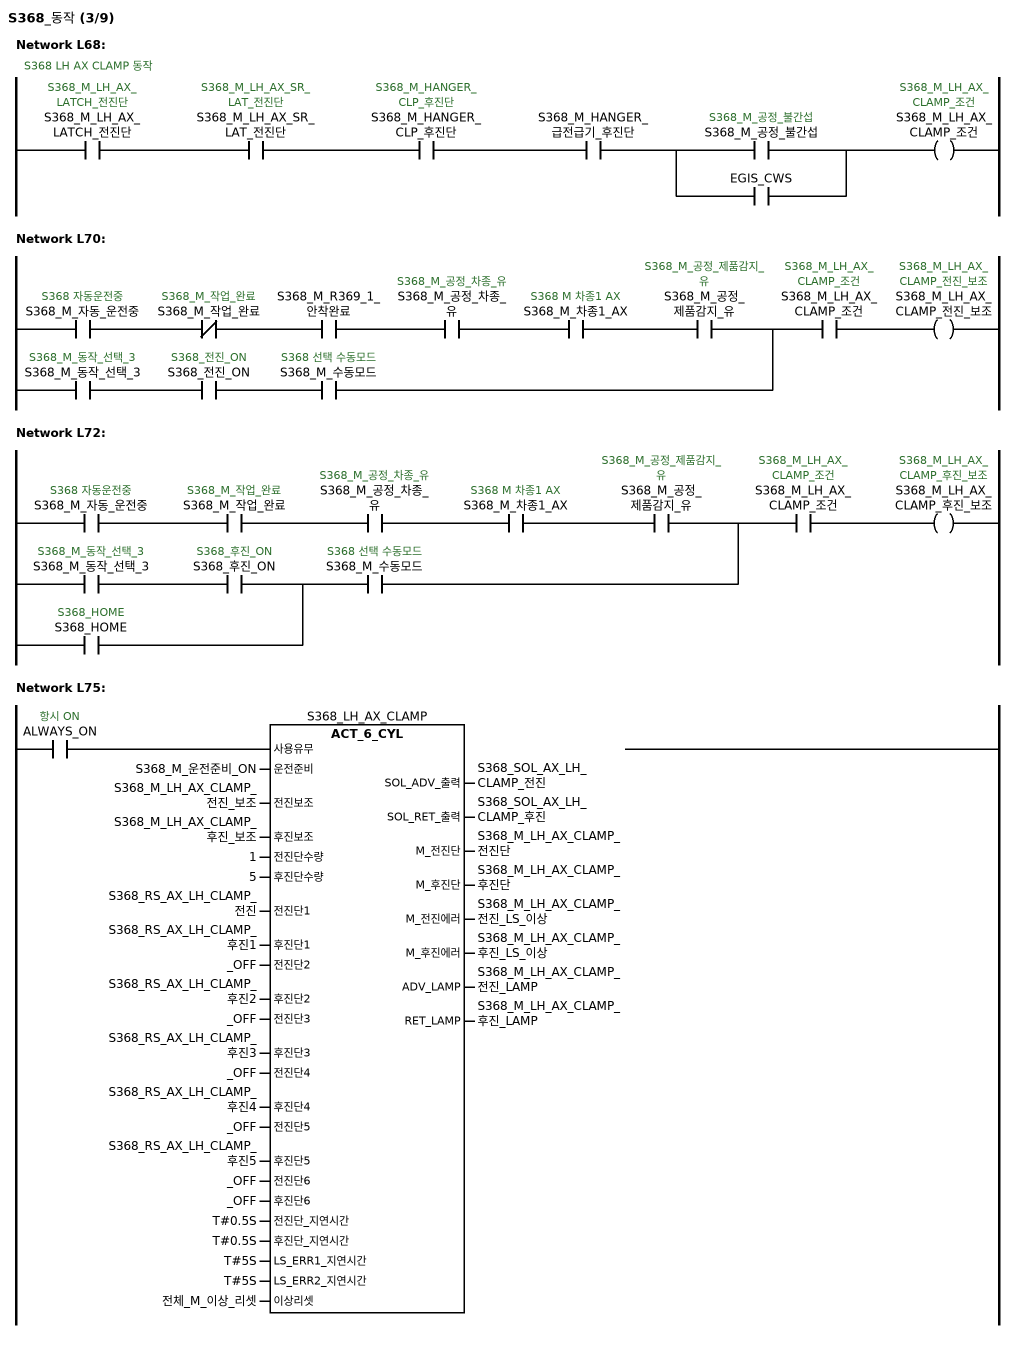
(* [picture p240: S368_동작 rungs L68-L75] *)
(* S368 LH AX CLAMP 동작 *)
(* Rung L68 *)
S368_M_LH_AX_CLAMP_조건 := S368_M_LH_AX_LATCH_전진단 AND S368_M_LH_AX_SR_LAT_전진단 AND S368_M_HANGER_CLP_후진단 AND S368_M_HANGER_급전급기_후진단 AND (S368_M_공정_불간섭 OR EGIS_CWS);
(* Rung L70 *)
S368_M_LH_AX_CLAMP_전진_보조 := ((S368_M_자동_운전중 AND NOT S368_M_작업_완료 AND S368_M_R369_1_안착완료 AND S368_M_공정_차종_유 AND S368_M_차종1_AX AND S368_M_공정_제품감지_유) OR (S368_M_동작_선택_3 AND S368_전진_ON AND S368_M_수동모드)) AND S368_M_LH_AX_CLAMP_조건;
(* Rung L72 *)
S368_M_LH_AX_CLAMP_후진_보조 := ((S368_M_자동_운전중 AND S368_M_작업_완료 AND S368_M_공정_차종_유 AND S368_M_차종1_AX AND S368_M_공정_제품감지_유) OR (((S368_M_동작_선택_3 AND S368_후진_ON) OR S368_HOME) AND S368_M_수동모드)) AND S368_M_LH_AX_CLAMP_조건;
(* Rung L75 *)
S368_LH_AX_CLAMP(사용유무 := ALWAYS_ON, 운전준비 := S368_M_운전준비_ON, 전진보조 := S368_M_LH_AX_CLAMP_전진_보조, 후진보조 := S368_M_LH_AX_CLAMP_후진_보조, 전진단수량 := 1, 후진단수량 := 5, 전진단1 := S368_RS_AX_LH_CLAMP_전진, 후진단1 := S368_RS_AX_LH_CLAMP_후진1, 전진단2 := _OFF, 후진단2 := S368_RS_AX_LH_CLAMP_후진2, 전진단3 := _OFF, 후진단3 := S368_RS_AX_LH_CLAMP_후진3, 전진단4 := _OFF, 후진단4 := S368_RS_AX_LH_CLAMP_후진4, 전진단5 := _OFF, 후진단5 := S368_RS_AX_LH_CLAMP_후진5, 전진단6 := _OFF, 후진단6 := _OFF, 전진단_지연시간 := T#0.5S, 후진단_지연시간 := T#0.5S, LS_ERR1_지연시간 := T#5S, LS_ERR2_지연시간 := T#5S, 이상리셋 := 전체_M_이상_리셋, SOL_ADV_출력 => S368_SOL_AX_LH_CLAMP_전진, SOL_RET_출력 => S368_SOL_AX_LH_CLAMP_후진, M_전진단 => S368_M_LH_AX_CLAMP_전진단, M_후진단 => S368_M_LH_AX_CLAMP_후진단, M_전진에러 => S368_M_LH_AX_CLAMP_전진_LS_이상, M_후진에러 => S368_M_LH_AX_CLAMP_후진_LS_이상, ADV_LAMP => S368_M_LH_AX_CLAMP_전진_LAMP, RET_LAMP => S368_M_LH_AX_CLAMP_후진_LAMP);

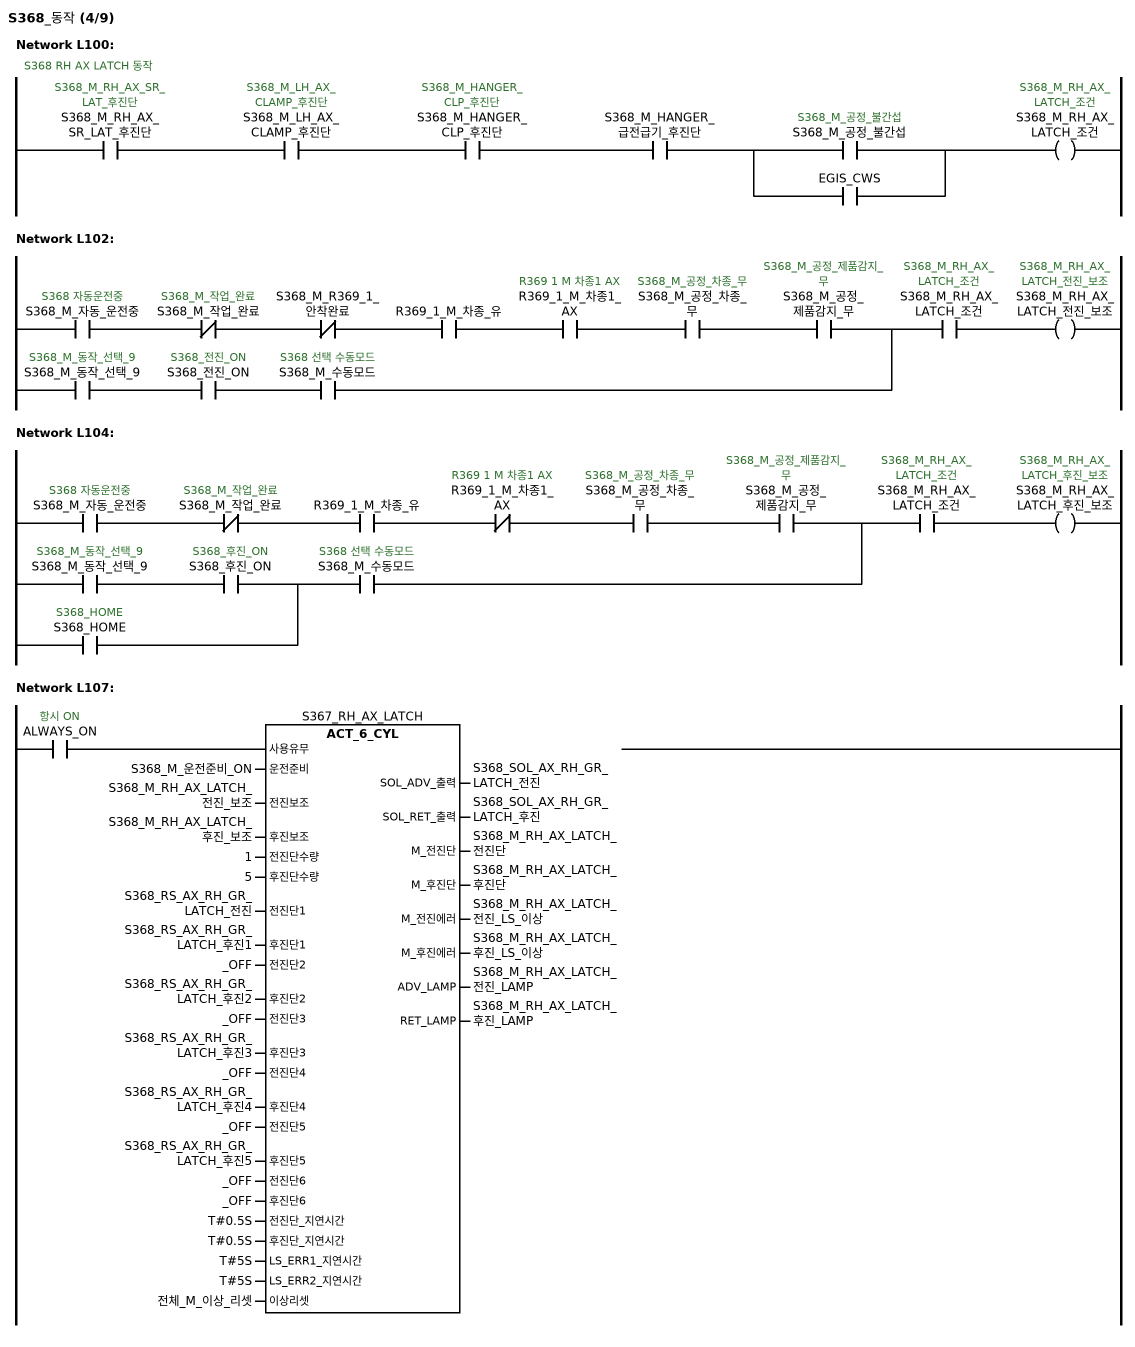
(* S368 RH AX LATCH 동작 *)
(* Rung L100 *)
S368_M_RH_AX_LATCH_조건 := S368_M_RH_AX_SR_LAT_후진단 AND S368_M_LH_AX_CLAMP_후진단 AND S368_M_HANGER_CLP_후진단 AND S368_M_HANGER_급전급기_후진단 AND (S368_M_공정_불간섭 OR EGIS_CWS);
(* Rung L102 *)
S368_M_RH_AX_LATCH_전진_보조 := ((S368_M_자동_운전중 AND NOT S368_M_작업_완료 AND NOT S368_M_R369_1_안착완료 AND R369_1_M_차종_유 AND R369_1_M_차종1_AX AND S368_M_공정_차종_무 AND S368_M_공정_제품감지_무) OR (S368_M_동작_선택_9 AND S368_전진_ON AND S368_M_수동모드)) AND S368_M_RH_AX_LATCH_조건;
(* Rung L104 *)
S368_M_RH_AX_LATCH_후진_보조 := ((S368_M_자동_운전중 AND NOT S368_M_작업_완료 AND R369_1_M_차종_유 AND NOT R369_1_M_차종1_AX AND S368_M_공정_차종_무 AND S368_M_공정_제품감지_무) OR (((S368_M_동작_선택_9 AND S368_후진_ON) OR S368_HOME) AND S368_M_수동모드)) AND S368_M_RH_AX_LATCH_조건;
(* Rung L107 *)
S367_RH_AX_LATCH(사용유무 := ALWAYS_ON, 운전준비 := S368_M_운전준비_ON, 전진보조 := S368_M_RH_AX_LATCH_전진_보조, 후진보조 := S368_M_RH_AX_LATCH_후진_보조, 전진단수량 := 1, 후진단수량 := 5, 전진단1 := S368_RS_AX_RH_GR_LATCH_전진, 후진단1 := S368_RS_AX_RH_GR_LATCH_후진1, 전진단2 := _OFF, 후진단2 := S368_RS_AX_RH_GR_LATCH_후진2, 전진단3 := _OFF, 후진단3 := S368_RS_AX_RH_GR_LATCH_후진3, 전진단4 := _OFF, 후진단4 := S368_RS_AX_RH_GR_LATCH_후진4, 전진단5 := _OFF, 후진단5 := S368_RS_AX_RH_GR_LATCH_후진5, 전진단6 := _OFF, 후진단6 := _OFF, 전진단_지연시간 := T#0.5S, 후진단_지연시간 := T#0.5S, LS_ERR1_지연시간 := T#5S, LS_ERR2_지연시간 := T#5S, 이상리셋 := 전체_M_이상_리셋, SOL_ADV_출력 => S368_SOL_AX_RH_GR_LATCH_전진, SOL_RET_출력 => S368_SOL_AX_RH_GR_LATCH_후진, M_전진단 => S368_M_RH_AX_LATCH_전진단, M_후진단 => S368_M_RH_AX_LATCH_후진단, M_전진에러 => S368_M_RH_AX_LATCH_전진_LS_이상, M_후진에러 => S368_M_RH_AX_LATCH_후진_LS_이상, ADV_LAMP => S368_M_RH_AX_LATCH_전진_LAMP, RET_LAMP => S368_M_RH_AX_LATCH_후진_LAMP);

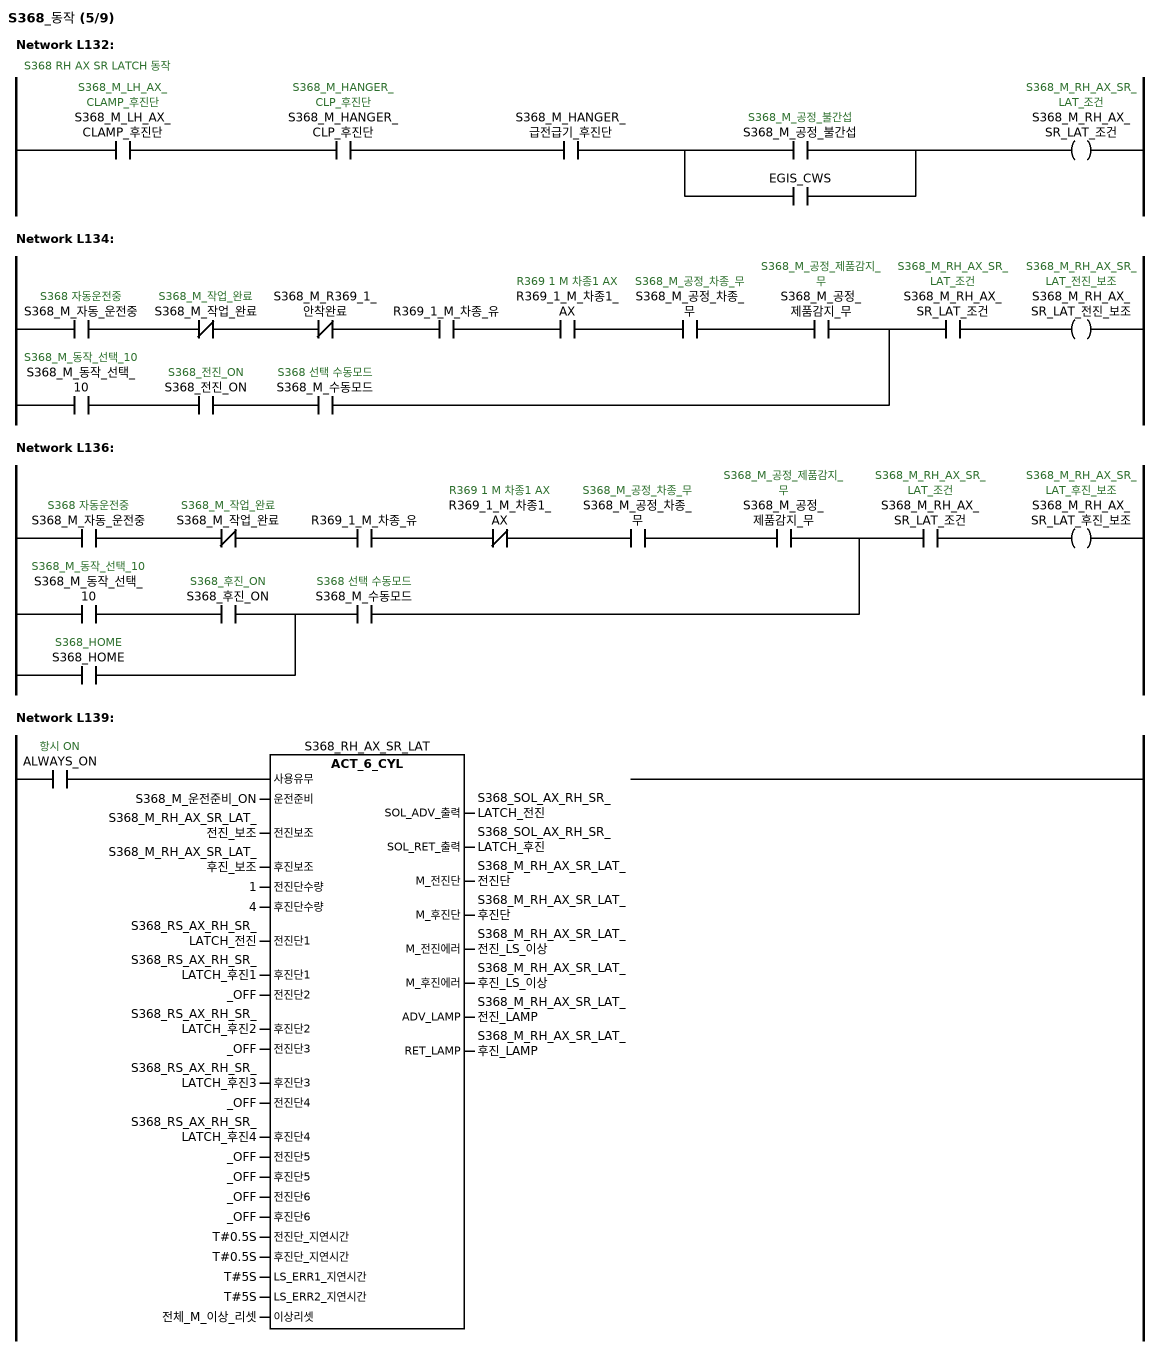
(* S368 RH AX SR LATCH 동작 *)
(* Rung L132 *)
S368_M_RH_AX_SR_LAT_조건 := S368_M_LH_AX_CLAMP_후진단 AND S368_M_HANGER_CLP_후진단 AND S368_M_HANGER_급전급기_후진단 AND (S368_M_공정_불간섭 OR EGIS_CWS);
(* Rung L134 *)
S368_M_RH_AX_SR_LAT_전진_보조 := ((S368_M_자동_운전중 AND NOT S368_M_작업_완료 AND NOT S368_M_R369_1_안착완료 AND R369_1_M_차종_유 AND R369_1_M_차종1_AX AND S368_M_공정_차종_무 AND S368_M_공정_제품감지_무) OR (S368_M_동작_선택_10 AND S368_전진_ON AND S368_M_수동모드)) AND S368_M_RH_AX_SR_LAT_조건;
(* Rung L136 *)
S368_M_RH_AX_SR_LAT_후진_보조 := ((S368_M_자동_운전중 AND NOT S368_M_작업_완료 AND R369_1_M_차종_유 AND NOT R369_1_M_차종1_AX AND S368_M_공정_차종_무 AND S368_M_공정_제품감지_무) OR (((S368_M_동작_선택_10 AND S368_후진_ON) OR S368_HOME) AND S368_M_수동모드)) AND S368_M_RH_AX_SR_LAT_조건;
(* Rung L139 *)
S368_RH_AX_SR_LAT(사용유무 := ALWAYS_ON, 운전준비 := S368_M_운전준비_ON, 전진보조 := S368_M_RH_AX_SR_LAT_전진_보조, 후진보조 := S368_M_RH_AX_SR_LAT_후진_보조, 전진단수량 := 1, 후진단수량 := 4, 전진단1 := S368_RS_AX_RH_SR_LATCH_전진, 후진단1 := S368_RS_AX_RH_SR_LATCH_후진1, 전진단2 := _OFF, 후진단2 := S368_RS_AX_RH_SR_LATCH_후진2, 전진단3 := _OFF, 후진단3 := S368_RS_AX_RH_SR_LATCH_후진3, 전진단4 := _OFF, 후진단4 := S368_RS_AX_RH_SR_LATCH_후진4, 전진단5 := _OFF, 후진단5 := _OFF, 전진단6 := _OFF, 후진단6 := _OFF, 전진단_지연시간 := T#0.5S, 후진단_지연시간 := T#0.5S, LS_ERR1_지연시간 := T#5S, LS_ERR2_지연시간 := T#5S, 이상리셋 := 전체_M_이상_리셋, SOL_ADV_출력 => S368_SOL_AX_RH_SR_LATCH_전진, SOL_RET_출력 => S368_SOL_AX_RH_SR_LATCH_후진, M_전진단 => S368_M_RH_AX_SR_LAT_전진단, M_후진단 => S368_M_RH_AX_SR_LAT_후진단, M_전진에러 => S368_M_RH_AX_SR_LAT_전진_LS_이상, M_후진에러 => S368_M_RH_AX_SR_LAT_후진_LS_이상, ADV_LAMP => S368_M_RH_AX_SR_LAT_전진_LAMP, RET_LAMP => S368_M_RH_AX_SR_LAT_후진_LAMP);

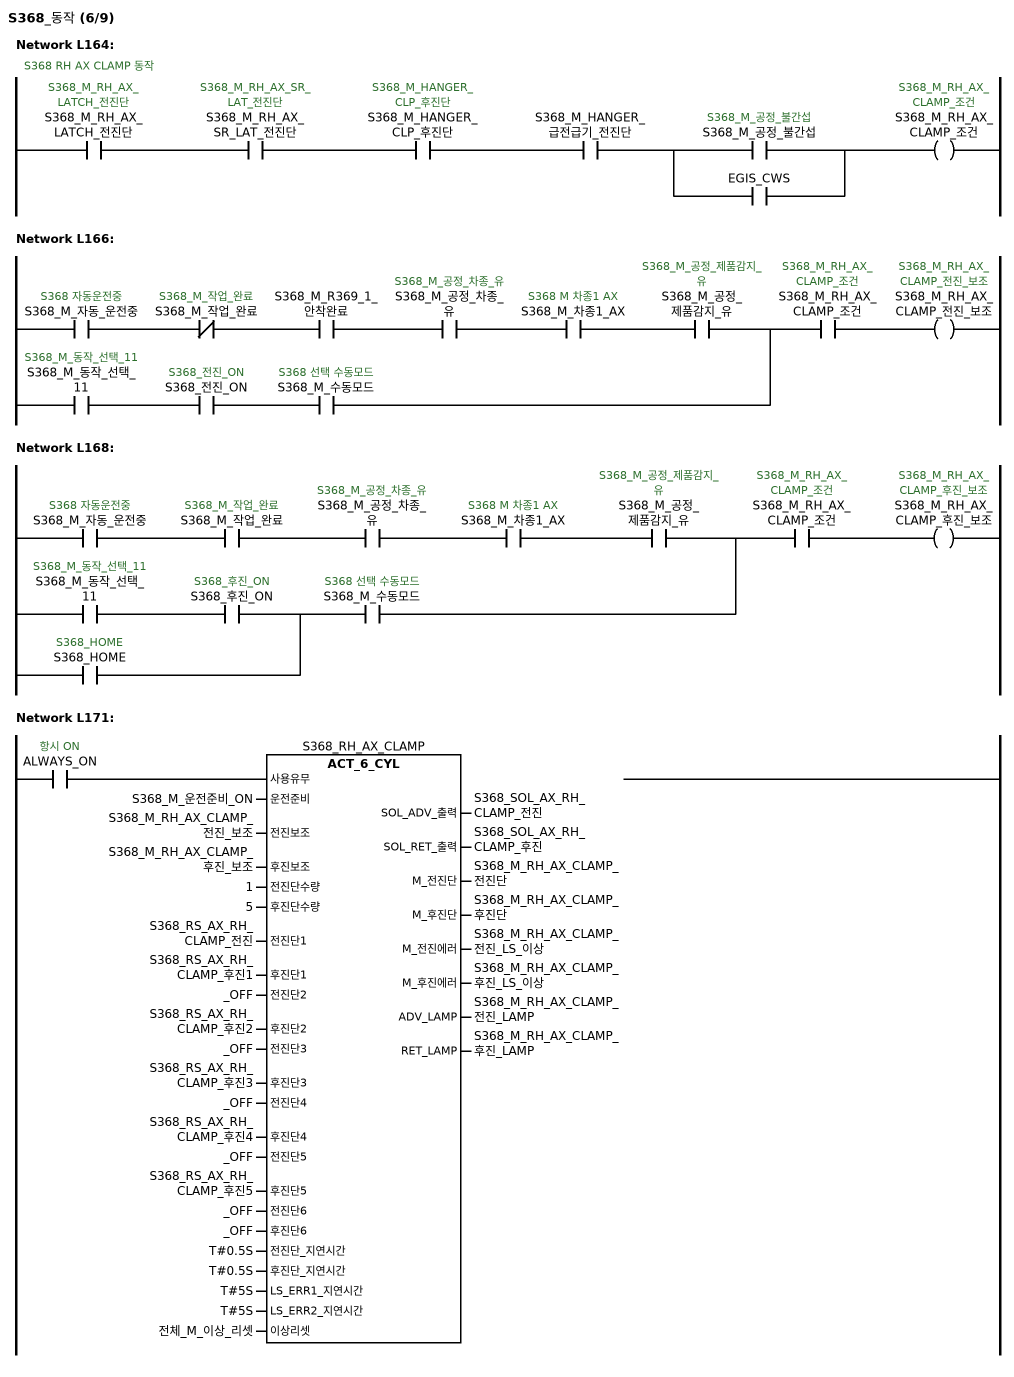
(* S368 RH AX CLAMP 동작 *)
(* Rung L164 *)
S368_M_RH_AX_CLAMP_조건 := S368_M_RH_AX_LATCH_전진단 AND S368_M_RH_AX_SR_LAT_전진단 AND S368_M_HANGER_CLP_후진단 AND S368_M_HANGER_급전급기_전진단 AND (S368_M_공정_불간섭 OR EGIS_CWS);
(* Rung L166 *)
S368_M_RH_AX_CLAMP_전진_보조 := ((S368_M_자동_운전중 AND NOT S368_M_작업_완료 AND S368_M_R369_1_안착완료 AND S368_M_공정_차종_유 AND S368_M_차종1_AX AND S368_M_공정_제품감지_유) OR (S368_M_동작_선택_11 AND S368_전진_ON AND S368_M_수동모드)) AND S368_M_RH_AX_CLAMP_조건;
(* Rung L168 *)
S368_M_RH_AX_CLAMP_후진_보조 := ((S368_M_자동_운전중 AND S368_M_작업_완료 AND S368_M_공정_차종_유 AND S368_M_차종1_AX AND S368_M_공정_제품감지_유) OR (((S368_M_동작_선택_11 AND S368_후진_ON) OR S368_HOME) AND S368_M_수동모드)) AND S368_M_RH_AX_CLAMP_조건;
(* Rung L171 *)
S368_RH_AX_CLAMP(사용유무 := ALWAYS_ON, 운전준비 := S368_M_운전준비_ON, 전진보조 := S368_M_RH_AX_CLAMP_전진_보조, 후진보조 := S368_M_RH_AX_CLAMP_후진_보조, 전진단수량 := 1, 후진단수량 := 5, 전진단1 := S368_RS_AX_RH_CLAMP_전진, 후진단1 := S368_RS_AX_RH_CLAMP_후진1, 전진단2 := _OFF, 후진단2 := S368_RS_AX_RH_CLAMP_후진2, 전진단3 := _OFF, 후진단3 := S368_RS_AX_RH_CLAMP_후진3, 전진단4 := _OFF, 후진단4 := S368_RS_AX_RH_CLAMP_후진4, 전진단5 := _OFF, 후진단5 := S368_RS_AX_RH_CLAMP_후진5, 전진단6 := _OFF, 후진단6 := _OFF, 전진단_지연시간 := T#0.5S, 후진단_지연시간 := T#0.5S, LS_ERR1_지연시간 := T#5S, LS_ERR2_지연시간 := T#5S, 이상리셋 := 전체_M_이상_리셋, SOL_ADV_출력 => S368_SOL_AX_RH_CLAMP_전진, SOL_RET_출력 => S368_SOL_AX_RH_CLAMP_후진, M_전진단 => S368_M_RH_AX_CLAMP_전진단, M_후진단 => S368_M_RH_AX_CLAMP_후진단, M_전진에러 => S368_M_RH_AX_CLAMP_전진_LS_이상, M_후진에러 => S368_M_RH_AX_CLAMP_후진_LS_이상, ADV_LAMP => S368_M_RH_AX_CLAMP_전진_LAMP, RET_LAMP => S368_M_RH_AX_CLAMP_후진_LAMP);

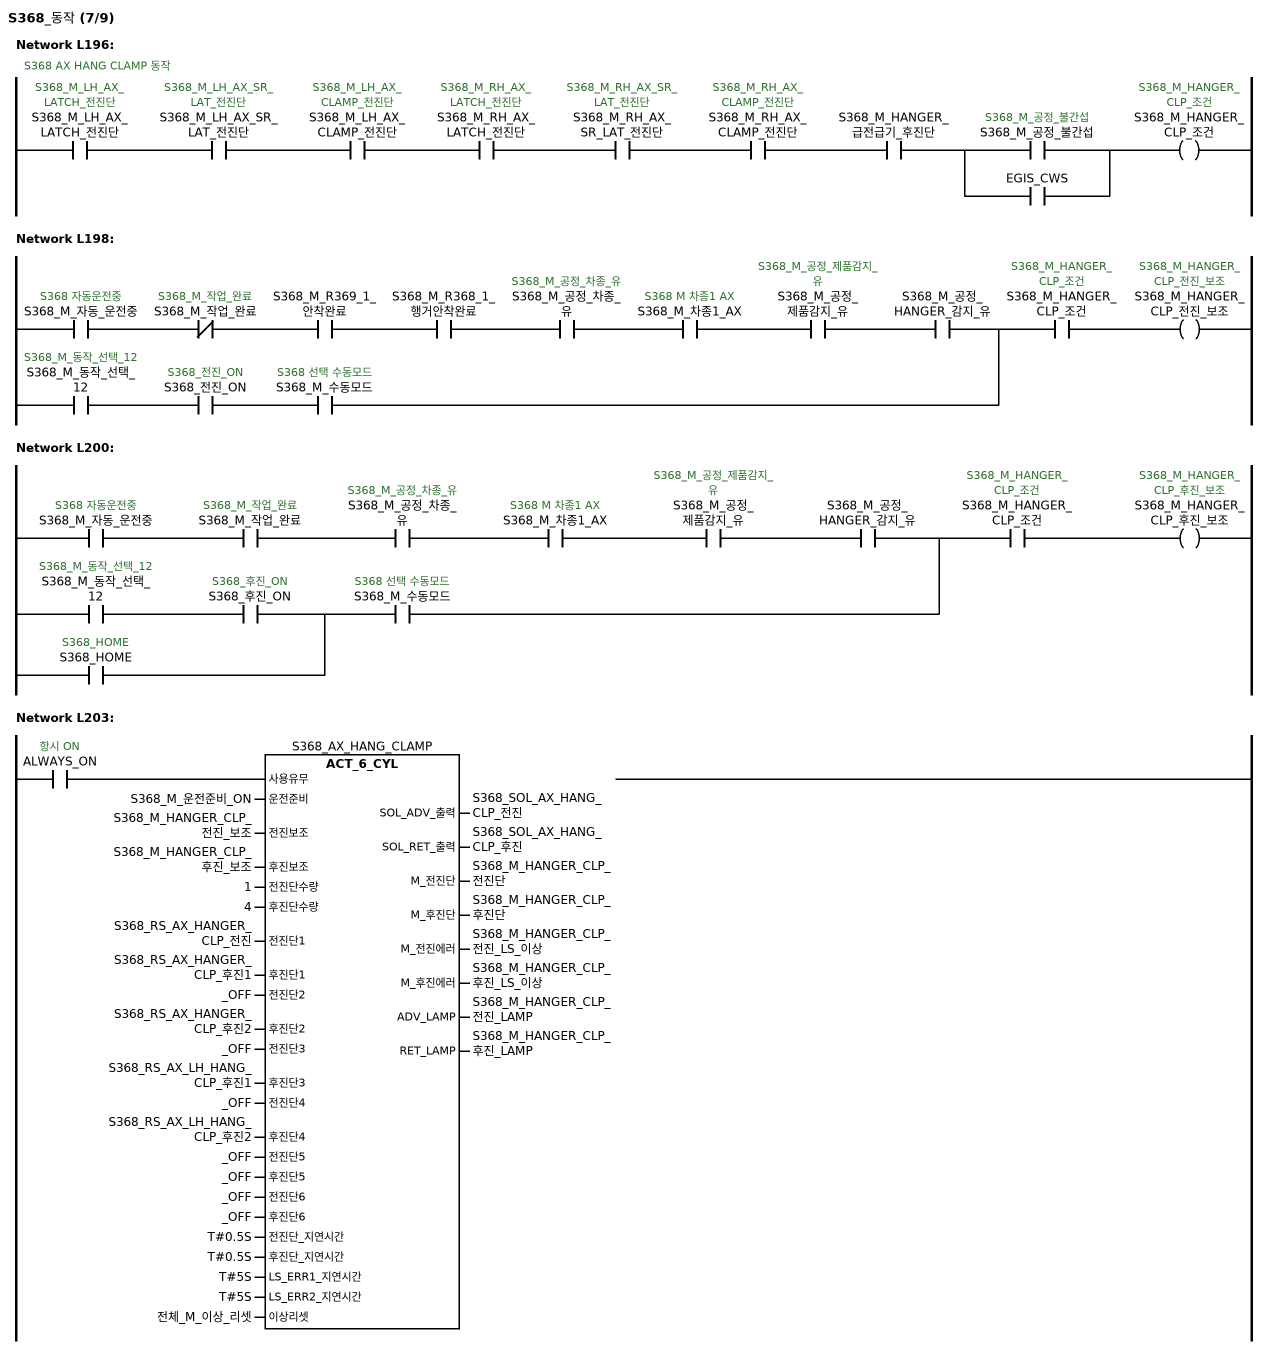
(* S368 AX HANG CLAMP 동작 *)
(* Rung L196 *)
S368_M_HANGER_CLP_조건 := S368_M_LH_AX_LATCH_전진단 AND S368_M_LH_AX_SR_LAT_전진단 AND S368_M_LH_AX_CLAMP_전진단 AND S368_M_RH_AX_LATCH_전진단 AND S368_M_RH_AX_SR_LAT_전진단 AND S368_M_RH_AX_CLAMP_전진단 AND S368_M_HANGER_급전급기_후진단 AND (S368_M_공정_불간섭 OR EGIS_CWS);
(* Rung L198 *)
S368_M_HANGER_CLP_전진_보조 := ((S368_M_자동_운전중 AND NOT S368_M_작업_완료 AND S368_M_R369_1_안착완료 AND S368_M_R368_1_행거안착완료 AND S368_M_공정_차종_유 AND S368_M_차종1_AX AND S368_M_공정_제품감지_유 AND S368_M_공정_HANGER_감지_유) OR (S368_M_동작_선택_12 AND S368_전진_ON AND S368_M_수동모드)) AND S368_M_HANGER_CLP_조건;
(* Rung L200 *)
S368_M_HANGER_CLP_후진_보조 := ((S368_M_자동_운전중 AND S368_M_작업_완료 AND S368_M_공정_차종_유 AND S368_M_차종1_AX AND S368_M_공정_제품감지_유 AND S368_M_공정_HANGER_감지_유) OR (((S368_M_동작_선택_12 AND S368_후진_ON) OR S368_HOME) AND S368_M_수동모드)) AND S368_M_HANGER_CLP_조건;
(* Rung L203 *)
S368_AX_HANG_CLAMP(사용유무 := ALWAYS_ON, 운전준비 := S368_M_운전준비_ON, 전진보조 := S368_M_HANGER_CLP_전진_보조, 후진보조 := S368_M_HANGER_CLP_후진_보조, 전진단수량 := 1, 후진단수량 := 4, 전진단1 := S368_RS_AX_HANGER_CLP_전진, 후진단1 := S368_RS_AX_HANGER_CLP_후진1, 전진단2 := _OFF, 후진단2 := S368_RS_AX_HANGER_CLP_후진2, 전진단3 := _OFF, 후진단3 := S368_RS_AX_LH_HANG_CLP_후진1, 전진단4 := _OFF, 후진단4 := S368_RS_AX_LH_HANG_CLP_후진2, 전진단5 := _OFF, 후진단5 := _OFF, 전진단6 := _OFF, 후진단6 := _OFF, 전진단_지연시간 := T#0.5S, 후진단_지연시간 := T#0.5S, LS_ERR1_지연시간 := T#5S, LS_ERR2_지연시간 := T#5S, 이상리셋 := 전체_M_이상_리셋, SOL_ADV_출력 => S368_SOL_AX_HANG_CLP_전진, SOL_RET_출력 => S368_SOL_AX_HANG_CLP_후진, M_전진단 => S368_M_HANGER_CLP_전진단, M_후진단 => S368_M_HANGER_CLP_후진단, M_전진에러 => S368_M_HANGER_CLP_전진_LS_이상, M_후진에러 => S368_M_HANGER_CLP_후진_LS_이상, ADV_LAMP => S368_M_HANGER_CLP_전진_LAMP, RET_LAMP => S368_M_HANGER_CLP_후진_LAMP);

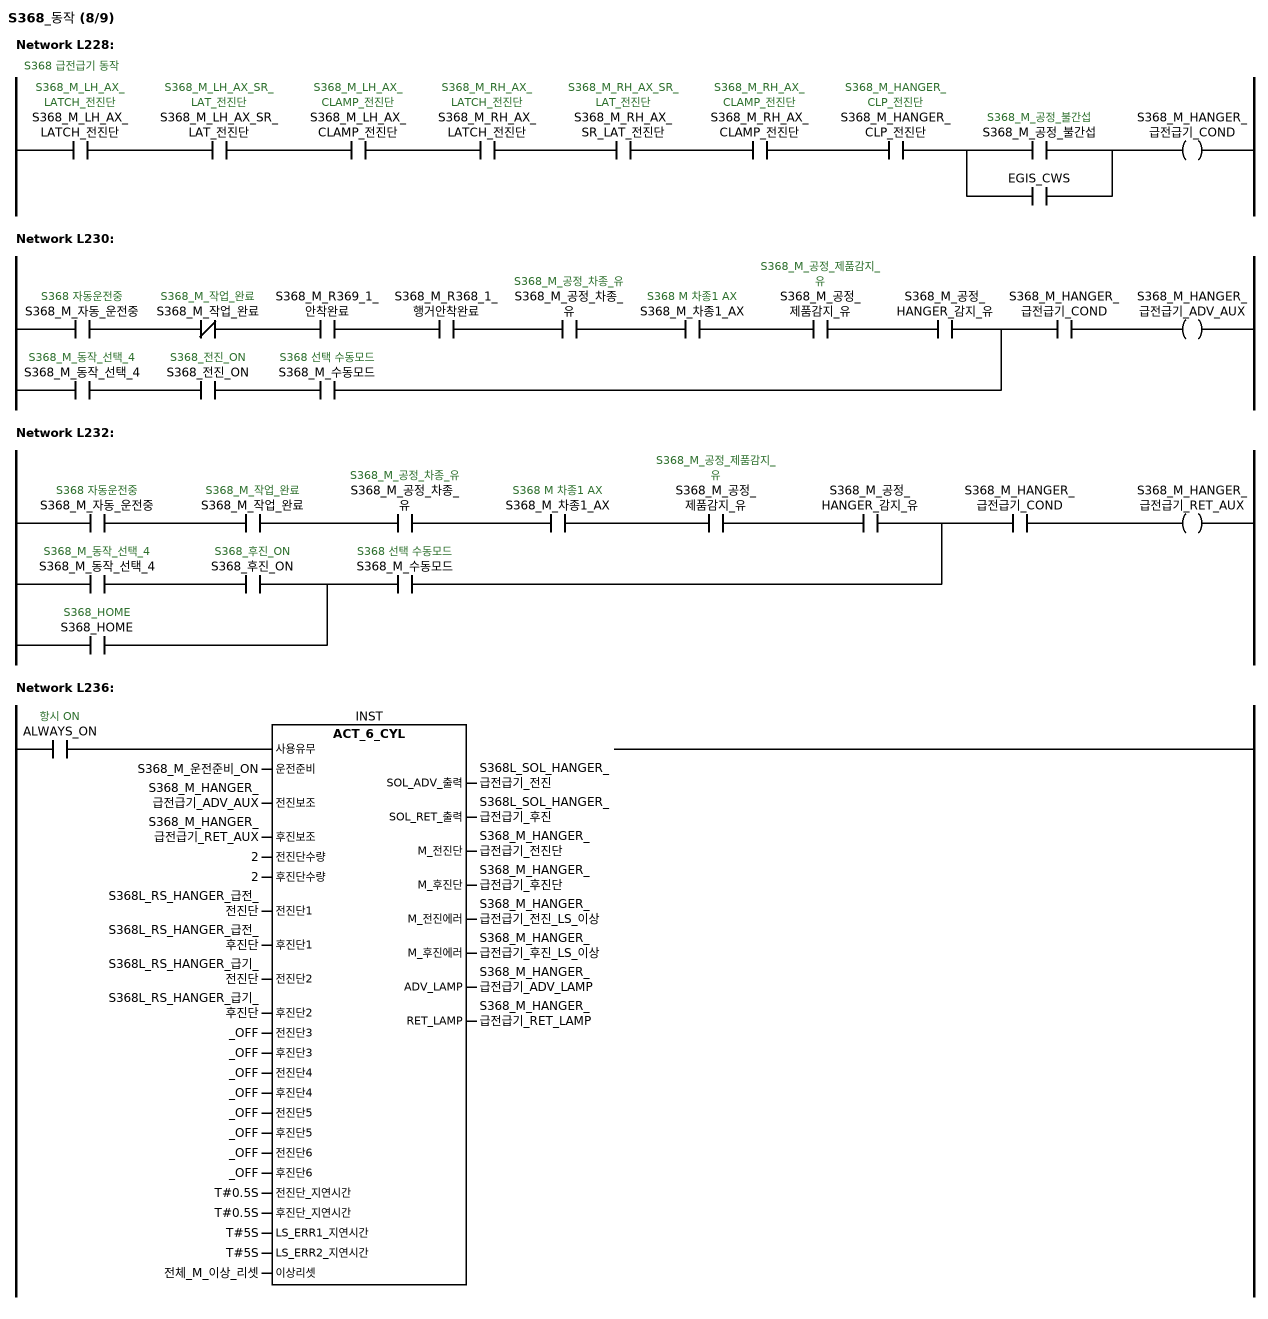
(* S368 급전급기 동작 *)
(* Rung L228 *)
S368_M_HANGER_급전급기_COND := S368_M_LH_AX_LATCH_전진단 AND S368_M_LH_AX_SR_LAT_전진단 AND S368_M_LH_AX_CLAMP_전진단 AND S368_M_RH_AX_LATCH_전진단 AND S368_M_RH_AX_SR_LAT_전진단 AND S368_M_RH_AX_CLAMP_전진단 AND S368_M_HANGER_CLP_전진단 AND (S368_M_공정_불간섭 OR EGIS_CWS);
(* Rung L230 *)
S368_M_HANGER_급전급기_ADV_AUX := ((S368_M_자동_운전중 AND NOT S368_M_작업_완료 AND S368_M_R369_1_안착완료 AND S368_M_R368_1_행거안착완료 AND S368_M_공정_차종_유 AND S368_M_차종1_AX AND S368_M_공정_제품감지_유 AND S368_M_공정_HANGER_감지_유) OR (S368_M_동작_선택_4 AND S368_전진_ON AND S368_M_수동모드)) AND S368_M_HANGER_급전급기_COND;
(* Rung L232 *)
S368_M_HANGER_급전급기_RET_AUX := ((S368_M_자동_운전중 AND S368_M_작업_완료 AND S368_M_공정_차종_유 AND S368_M_차종1_AX AND S368_M_공정_제품감지_유 AND S368_M_공정_HANGER_감지_유) OR (((S368_M_동작_선택_4 AND S368_후진_ON) OR S368_HOME) AND S368_M_수동모드)) AND S368_M_HANGER_급전급기_COND;
(* Rung L236 *)
INST(사용유무 := ALWAYS_ON, 운전준비 := S368_M_운전준비_ON, 전진보조 := S368_M_HANGER_급전급기_ADV_AUX, 후진보조 := S368_M_HANGER_급전급기_RET_AUX, 전진단수량 := 2, 후진단수량 := 2, 전진단1 := S368L_RS_HANGER_급전_전진단, 후진단1 := S368L_RS_HANGER_급전_후진단, 전진단2 := S368L_RS_HANGER_급기_전진단, 후진단2 := S368L_RS_HANGER_급기_후진단, 전진단3 := _OFF, 후진단3 := _OFF, 전진단4 := _OFF, 후진단4 := _OFF, 전진단5 := _OFF, 후진단5 := _OFF, 전진단6 := _OFF, 후진단6 := _OFF, 전진단_지연시간 := T#0.5S, 후진단_지연시간 := T#0.5S, LS_ERR1_지연시간 := T#5S, LS_ERR2_지연시간 := T#5S, 이상리셋 := 전체_M_이상_리셋, SOL_ADV_출력 => S368L_SOL_HANGER_급전급기_전진, SOL_RET_출력 => S368L_SOL_HANGER_급전급기_후진, M_전진단 => S368_M_HANGER_급전급기_전진단, M_후진단 => S368_M_HANGER_급전급기_후진단, M_전진에러 => S368_M_HANGER_급전급기_전진_LS_이상, M_후진에러 => S368_M_HANGER_급전급기_후진_LS_이상, ADV_LAMP => S368_M_HANGER_급전급기_ADV_LAMP, RET_LAMP => S368_M_HANGER_급전급기_RET_LAMP);

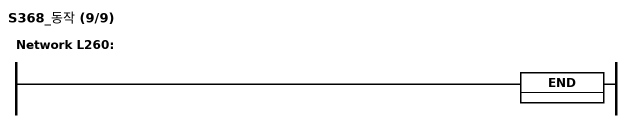
(* Rung L260 *)
END();
END_PROGRAM

PROGRAM S368_로보트 (* task: 스캔 프로그램 *)
VAR_EXTERNAL RETAIN
    ALWAYS_ON : BOOL; (* AT %MW3.1 *) (* 항시 ON *)
    MCP_M_부저_정지 : BOOL; (* AT %MW350.5 *) (* MCP 부저정지 *)
    MCP_M_비상정지 : BOOL; (* AT %MW350.7 *) (* MCP 비상정지 이상 *)
    S366_M_수동모드 : BOOL; (* AT %MW3000.3 *) (* S366 선택 수동모드 *)
    S366_M_자동_운전중 : BOOL; (* AT %MW3000.4 *) (* S366 자동운전중 *)
    S366_M_작업완료_SET_PLS : BOOL; (* AT %MW3000.8 *) (* S366 M 작업완료 SET PLS *)
    S366_M_작업완료_리셋_PLS : BOOL; (* AT %MW3000.9 *) (* S366 M 작업완료 리셋 PLS *)
    S368_M_R368_1_해밍가능 : BOOL; (* AT %MW4004.10 *)
    S368_M_R368_1_행거안착가능 : BOOL; (* AT %MW4004.9 *)
    S368_M_R368_1_행거안착완료 : BOOL; (* AT %MW4001.2 *)
    S368_M_R368_1_헤밍완료 : BOOL; (* AT %MW4001.3 *)
    S368_M_공정_HANGER_감지_무 : BOOL; (* AT %MW4001.12 *)
    S368_M_공정_HANGER_감지_유 : BOOL; (* AT %MW4001.11 *)
    S368_M_공정_제품감지_유 : BOOL; (* AT %MW4001.5 *) (* S368_M_공정_제품감지_유 *)
    S368_M_공정_차종_유 : BOOL; (* AT %MW4002.0 *) (* S368_M_공정_차종_유 *)
    S368_M_수동모드 : BOOL; (* AT %MW4000.3 *) (* S368 선택 수동모드 *)
    S368_M_자동_START : BOOL; (* AT %MW4000.5 *) (* S368 자동운전중 *)
    S368_M_자동_운전중 : BOOL; (* AT %MW4000.4 *) (* S368 자동운전중 *)
    S368_M_작업_완료 : BOOL; (* AT %MW4001.0 *) (* S368_M_작업_완료 *)
    S368_M_작업완료_SET_PLS : BOOL; (* AT %MW4000.8 *) (* S368 M 작업완료 SET PLS *)
    S368_M_작업완료_리셋_PLS : BOOL; (* AT %MW4000.9 *) (* S368 M 작업완료 리셋 PLS *)
    S368_M_차종1_AX : BOOL; (* AT %MW10201.0 *) (* S368 M 차종1 AX *)
    S368_M_총괄_이상 : BOOL; (* AT %MW4009.0 *) (* S368_M_총괄_이상 *)
    전체_M_GATE_비상정지_정상 : BOOL; (* AT %MW308.4 *) (* 전체 M GATE 비상정지 정상 *)
    전체_M_GATE_자동기동 : BOOL; (* AT %MW308.1 *) (* 전체_M_자동_운전 *)
    전체_M_운전준비_보조 : BOOL; (* AT %MW308.5 *)
    전체_M_이상_리셋 : BOOL; (* AT %MW308.2 *) (* ALL공정 PB 이상리셋 *)
    전체_공정_M_총괄_비상정지_정상 : BOOL; (* AT %MW304.1 *)
END_VAR
VAR
    INST1 : FB494_Robot_Hyundai_HMMI_v1;
    R368_1_M_RB_PROG_NO : INT;
    로보트제외 : BOOL;
END_VAR
VAR_EXTERNAL
    MCP_PBL_운전준비_ON : BOOL; (* AT %MW87630.0 *) (* MCP_PBL_운전준비_ON *)
    R366_1_M_I_RB_원위치 : BOOL; (* AT %MW20060.3 *) (* R366_1_M_I_RB_원위치 *)
    R366_1_M_O_RB_1_CYCLE_SET : BOOL; (* AT %MW21060.3 *) (* R366_1_M_O_RB_1_CYCLE_SET *)
    R366_1_M_O_RB_1차_작업완료_리셋 : BOOL; (* AT %MW21062.0 *) (* R366_1_M_O_RB_1차_작업완료_리셋 *)
    R366_1_M_O_RB_2차_작업완료_리셋 : BOOL; (* AT %MW21062.1 *) (* R366_1_M_O_RB_2차_작업완료_리셋 *)
    R366_1_M_O_RB_3차_작업완료_리셋 : BOOL; (* AT %MW21062.2 *) (* R366_1_M_O_RB_3차_작업완료_리셋 *)
    R366_1_M_O_RB_최종_작업완료_리셋 : BOOL; (* AT %MW21060.5 *) (* R366_1_M_O_RB_최종_작업완료_리셋 *)
    R368_1_I_RB_INPUT : ARRAY[0..3] OF WORD; (* AT %MW84070 *) (* R368_1_I_RB_INPUT *)
    R368_1_M_I_RB_1차_작업완료 : BOOL; (* AT %MW20071.2 *) (* R368_1_M_I_RB_1차_작업완료 *)
    R368_1_M_I_RB_2차_작업완료 : BOOL; (* AT %MW20071.3 *) (* R368_1_M_I_RB_2차_작업완료 *)
    R368_1_M_I_RB_3차_작업완료 : BOOL; (* AT %MW20071.4 *) (* R368_1_M_I_RB_3차_작업완료 *)
    R368_1_M_I_RB_4차_작업완료 : BOOL; (* AT %MW20071.5 *) (* R368_1_M_I_RB_4차_작업완료 *)
    R368_1_M_I_RB_5차_작업완료 : BOOL; (* AT %MW20071.6 *) (* R368_1_M_I_RB_5차_작업완료 *)
    R368_1_M_I_RB_6차_작업완료 : BOOL; (* AT %MW20071.7 *) (* R368_1_M_I_RB_6차_작업완료 *)
    R368_1_M_I_RB_7차_작업완료 : BOOL; (* AT %MW20071.8 *) (* R368_1_M_I_RB_7차_작업완료 *)
    R368_1_M_I_RB_PAUSE_보조 : BOOL; (* AT %MW20070.5 *) (* R368_1_M_I_RB_PAUSE_보조 *)
    R368_1_M_I_RB_PLC_RUN_CHK_이상 : BOOL; (* AT %MW20070.7 *) (* R368_1_M_I_RB_PLC_RUN_CHK_이상 *)
    R368_1_M_I_RB_간섭무_1 : BOOL; (* AT %MW20072.0 *) (* R368_1_M_I_RB_간섭무_1 *)
    R368_1_M_I_RB_간섭무_10 : BOOL; (* AT %MW20072.9 *) (* R368_1_M_I_RB_간섭무_10 *)
    R368_1_M_I_RB_간섭무_11 : BOOL; (* AT %MW20072.10 *) (* R368_1_M_I_RB_간섭무_11 *)
    R368_1_M_I_RB_간섭무_12 : BOOL; (* AT %MW20072.11 *) (* R368_1_M_I_RB_간섭무_12 *)
    R368_1_M_I_RB_간섭무_2 : BOOL; (* AT %MW20072.1 *) (* R368_1_M_I_RB_간섭무_2 *)
    R368_1_M_I_RB_간섭무_3 : BOOL; (* AT %MW20072.2 *) (* R368_1_M_I_RB_간섭무_3 *)
    R368_1_M_I_RB_간섭무_4 : BOOL; (* AT %MW20072.3 *) (* R368_1_M_I_RB_간섭무_4 *)
    R368_1_M_I_RB_간섭무_5 : BOOL; (* AT %MW20072.4 *) (* R368_1_M_I_RB_간섭무_5 *)
    R368_1_M_I_RB_간섭무_6 : BOOL; (* AT %MW20072.5 *) (* R368_1_M_I_RB_간섭무_6 *)
    R368_1_M_I_RB_간섭무_7 : BOOL; (* AT %MW20072.6 *) (* R368_1_M_I_RB_간섭무_7 *)
    R368_1_M_I_RB_간섭무_8 : BOOL; (* AT %MW20072.7 *) (* R368_1_M_I_RB_간섭무_8 *)
    R368_1_M_I_RB_간섭무_9 : BOOL; (* AT %MW20072.8 *) (* R368_1_M_I_RB_간섭무_9 *)
    R368_1_M_I_RB_비상정지 : BOOL; (* AT %MW20070.4 *) (* R368_1_M_I_RB_비상정지 *)
    R368_1_M_I_RB_운전준비 : BOOL; (* AT %MW20070.0 *) (* R368_1_M_I_RB_운전준비 *)
    R368_1_M_I_RB_원위치 : BOOL; (* AT %MW20070.3 *) (* R368_1_M_I_RB_원위치 *)
    R368_1_M_I_RB_이상 : BOOL; (* AT %MW20070.2 *) (* R368_1_M_I_RB_이상 *)
    R368_1_M_I_RB_자동 : BOOL; (* AT %MW20070.1 *) (* R368_1_M_I_RB_자동 *)
    R368_1_M_I_RB_최종작업완료 : BOOL; (* AT %MW20071.0 *) (* R368_1_M_I_RB_최종작업완료 *)
    R368_1_M_I_RB_프로그램_이상 : BOOL; (* AT %MW20070.6 *) (* R368_1_M_I_RB_프로그램_이상 *)
    R368_1_M_O_RB_1_CYCLE_SET : BOOL; (* AT %MW21070.3 *) (* R368_1_M_O_RB_1_CYCLE_SET *)
    R368_1_M_O_RB_1차_작업완료_리셋 : BOOL; (* AT %MW21072.0 *) (* R368_1_M_O_RB_1차_작업완료_리셋 *)
    R368_1_M_O_RB_2차_작업완료_리셋 : BOOL; (* AT %MW21072.1 *) (* R368_1_M_O_RB_2차_작업완료_리셋 *)
    R368_1_M_O_RB_2차_진입OK : BOOL; (* AT %MW21071.8 *) (* R368_1_M_O_RB_2차_진입OK *)
    R368_1_M_O_RB_3차_작업완료_리셋 : BOOL; (* AT %MW21072.2 *) (* R368_1_M_O_RB_3차_작업완료_리셋 *)
    R368_1_M_O_RB_3차_진입OK : BOOL; (* AT %MW21071.9 *) (* R368_1_M_O_RB_3차_진입OK *)
    R368_1_M_O_RB_4차_작업완료_리셋 : BOOL; (* AT %MW21072.3 *) (* R368_1_M_O_RB_4차_작업완료_리셋 *)
    R368_1_M_O_RB_4차_진입OK : BOOL; (* AT %MW21071.10 *) (* R368_1_M_O_RB_4차_진입OK *)
    R368_1_M_O_RB_5차_작업완료_리셋 : BOOL; (* AT %MW21072.4 *) (* R368_1_M_O_RB_5차_작업완료_리셋 *)
    R368_1_M_O_RB_5차_진입OK : BOOL; (* AT %MW21071.11 *) (* R368_1_M_O_RB_5차_진입OK *)
    R368_1_M_O_RB_6차_작업완료_리셋 : BOOL; (* AT %MW21072.5 *) (* R368_1_M_O_RB_6차_작업완료_리셋 *)
    R368_1_M_O_RB_6차_진입OK : BOOL; (* AT %MW21071.12 *) (* R368_1_M_O_RB_6차_진입OK *)
    R368_1_M_O_RB_7차_작업완료_리셋 : BOOL; (* AT %MW21072.6 *) (* R368_1_M_O_RB_7차_작업완료_리셋 *)
    R368_1_M_O_RB_7차_진입OK : BOOL; (* AT %MW21071.13 *) (* R368_1_M_O_RB_7차_진입OK *)
    R368_1_M_O_RB_ATD_OK : BOOL; (* AT %MW21070.6 *) (* R368_1_M_O_RB_ATD_OK *)
    R368_1_M_O_RB_PLT_10_진입OK : BOOL; (* AT %MW21073.10 *) (* R368_1_M_O_RB_PLT_10_진입OK *)
    R368_1_M_O_RB_PLT_11_진입OK : BOOL; (* AT %MW21073.11 *) (* R368_1_M_O_RB_PLT_11_진입OK *)
    R368_1_M_O_RB_PLT_12_진입OK : BOOL; (* AT %MW21073.12 *) (* R368_1_M_O_RB_PLT_12_진입OK *)
    R368_1_M_O_RB_PLT_1_진입OK : BOOL; (* AT %MW21073.1 *) (* R368_1_M_O_RB_PLT_1_진입OK *)
    R368_1_M_O_RB_PLT_2_진입OK : BOOL; (* AT %MW21073.2 *) (* R368_1_M_O_RB_PLT_2_진입OK *)
    R368_1_M_O_RB_PLT_3_진입OK : BOOL; (* AT %MW21073.3 *) (* R368_1_M_O_RB_PLT_3_진입OK *)
    R368_1_M_O_RB_PLT_4_진입OK : BOOL; (* AT %MW21073.4 *) (* R368_1_M_O_RB_PLT_4_진입OK *)
    R368_1_M_O_RB_PLT_5_진입OK : BOOL; (* AT %MW21073.5 *) (* R368_1_M_O_RB_PLT_5_진입OK *)
    R368_1_M_O_RB_PLT_6_진입OK : BOOL; (* AT %MW21073.6 *) (* R368_1_M_O_RB_PLT_6_진입OK *)
    R368_1_M_O_RB_PLT_7_진입OK : BOOL; (* AT %MW21073.7 *) (* R368_1_M_O_RB_PLT_7_진입OK *)
    R368_1_M_O_RB_PLT_8_진입OK : BOOL; (* AT %MW21073.8 *) (* R368_1_M_O_RB_PLT_8_진입OK *)
    R368_1_M_O_RB_PLT_9_진입OK : BOOL; (* AT %MW21073.9 *) (* R368_1_M_O_RB_PLT_9_진입OK *)
    R368_1_M_O_RB_PLT_카운터리셋_보조 : BOOL; (* AT %MW21070.10 *) (* R368_1_M_O_RB_PLT_카운터리셋_보조 *)
    R368_1_M_O_RB_PROG_NO : WORD; (* AT %MW21074 *)
    R368_1_M_O_RB_RESTART_OK : BOOL; (* AT %MW21070.2 *) (* R368_1_M_O_RB_RESTART_OK *)
    R368_1_M_O_RB_START_OK : BOOL; (* AT %MW21070.0 *) (* R368_1_M_O_RB_START_OK *)
    R368_1_M_O_RB_TEST_MODE_5000회 : BOOL; (* AT %MW21070.12 *) (* R368_1_M_O_RB_TEST_MODE_5000회 *)
    R368_1_M_O_RB_TIP_교체_시작 : BOOL; (* AT %MW21070.7 *) (* R368_1_M_O_RB_TIP_교체_시작 *)
    R368_1_M_O_RB_TIP_교체_완료 : BOOL; (* AT %MW21070.8 *) (* R368_1_M_O_RB_TIP_교체_완료 *)
    R368_1_M_O_RB_VIP_MODE : BOOL; (* AT %MW21070.11 *) (* R368_1_M_O_RB_VIP_MODE *)
    R368_1_M_O_RB_냉각수_차단_요청 : BOOL; (* AT %MW21070.9 *) (* R368_1_M_O_RB_냉각수_차단_요청 *)
    R368_1_M_O_RB_진입OK_AX차종 : BOOL; (* AT %MW21071.0 *) (* R368_1_M_O_RB_진입OK_AX차종 *)
    R368_1_M_O_RB_진입OK_B차종 : BOOL; (* AT %MW21071.1 *) (* R368_1_M_O_RB_진입OK_B차종 *)
    R368_1_M_O_RB_진입OK_C차종 : BOOL; (* AT %MW21071.2 *) (* R368_1_M_O_RB_진입OK_C차종 *)
    R368_1_M_O_RB_진입OK_D차종 : BOOL; (* AT %MW21071.3 *) (* R368_1_M_O_RB_진입OK_D차종 *)
    R368_1_M_O_RB_진입OK_E차종 : BOOL; (* AT %MW21071.4 *) (* R368_1_M_O_RB_진입OK_E차종 *)
    R368_1_M_O_RB_진입OK_F차종 : BOOL; (* AT %MW21071.5 *) (* R368_1_M_O_RB_진입OK_F차종 *)
    R368_1_M_O_RB_진입OK_G차종 : BOOL; (* AT %MW21071.6 *) (* R368_1_M_O_RB_진입OK_G차종 *)
    R368_1_M_O_RB_진입OK_H차종 : BOOL; (* AT %MW21071.7 *) (* R368_1_M_O_RB_진입OK_H차종 *)
    R368_1_M_O_RB_최종_작업완료_리셋 : BOOL; (* AT %MW21070.5 *) (* R368_1_M_O_RB_최종_작업완료_리셋 *)
    R368_1_M_O_RB_프로그램_OK : BOOL; (* AT %MW21070.1 *) (* R368_1_M_O_RB_프로그램_OK *)
    R368_1_O_RB_OUTPUT : ARRAY[0..3] OF WORD; (* AT %MW94070 *) (* R368_1_O_RB_OUTPUT *)
    R369_1_I_RB_상호인터록_INT1 : BOOL; (* AT %MW84083.0 *) (* R369_1_I_RB_상호인터록_INT1 *)
END_VAR
(* ladder body could not be read *)
END_PROGRAM

PROGRAM S368_이상 (* task: 스캔 프로그램 *)
VAR
    INST10 : TON;
    INST11 : TON;
    INST12 : TON;
    INST13 : TON;
    INST14 : TON;
    INST15 : TON;
    INST16 : TON;
    INST17 : TON;
    INST18 : TON;
    INST19 : TON;
    INST20 : TON;
    INST21 : TON;
    INST22 : TON;
    INST23 : TON;
    INST24 : TON;
    INST25 : TON;
    INST26 : TON;
    INST27 : TON;
    INST28 : TON;
    INST29 : TON;
    INST30 : TON;
    INST31 : TON;
    INST32 : TON;
    INST8 : TON;
    INST9 : TON;
END_VAR
VAR_EXTERNAL
    R366_1_M_I_RB_이상 : BOOL; (* AT %MW20060.2 *) (* R366_1_M_I_RB_이상 *)
    R366_1_M_I_RB_프로그램_이상 : BOOL; (* AT %MW20060.6 *) (* R366_1_M_I_RB_프로그램_이상 *)
    R368_1_M_I_RB_이상 : BOOL; (* AT %MW20070.2 *) (* R368_1_M_I_RB_이상 *)
    R368_1_M_I_RB_프로그램_이상 : BOOL; (* AT %MW20070.6 *) (* R368_1_M_I_RB_프로그램_이상 *)
    S368_6_30_PLC_BOX_CP_TRIP : BOOL; (* AT %MW86302.15 *) (* S368_6_30_PLC_BOX_CP_TRIP *)
    S368_6_31_PLC_BOX_CP_TRIP : BOOL; (* AT %MW86312.15 *) (* S368_6_31_PLC_BOX_CP_TRIP *)
    S368_PRS_AX_LH_HANGER_CHECK : BOOL; (* AT %MW86312.2 *) (* S368_PRS_AX_LH_HANGER_CHECK *)
    S368_PRS_AX_LH_ROOF_FRT_CHECK : BOOL; (* AT %MW86312.0 *) (* S368_PRS_AX_LH_ROOF_FRT_CHECK *)
    S368_PRS_AX_LH_ROOF_RR_CHECK : BOOL; (* AT %MW86312.1 *) (* S368_PRS_AX_LH_ROOF_RR_CHECK *)
    S368_PRS_AX_RH_HANGER_CHECK : BOOL; (* AT %MW86302.2 *) (* S368_PRS_AX_RH_HANGER_CHECK *)
    S368_PRS_AX_RH_ROOF_FRT_CHECK : BOOL; (* AT %MW86302.0 *) (* S368_PRS_AX_RH_ROOF_FRT_CHECK *)
    S368_PRS_AX_RH_ROOF_RR_CHECK : BOOL; (* AT %MW86302.1 *) (* S368_PRS_AX_RH_ROOF_RR_CHECK *)
    S368_공기압_AIR_CHECK : BOOL; (* AT %MW86302.14 *) (* S368_공기압_AIR_CHECK *)
    _0004_EB06_CFG_ER : BOOL; (* AT %MW184034.8 *) (* EB 구성 에러 *)
    _0004_EB06_DEER : BOOL; (* AT %MW184034.9 *) (* EB 운전 중 탈락 *)
    _0004_EB07_CFG_ER : BOOL; (* AT %MW184037.0 *) (* EB 구성 에러 *)
    _0004_EB07_DEER : BOOL; (* AT %MW184037.1 *) (* EB 운전 중 탈락 *)
    _0006_EB10_CFG_ER : BOOL; (* AT %MW186028.0 *) (* EB 구성 에러 *)
    _0006_EB10_DEER : BOOL; (* AT %MW186028.1 *) (* EB 운전 중 탈락 *)
    _0006_EB10_IO_DEER : BOOL; (* AT %MW186029.2 *) (* EB IO 탈락 에러 *)
    _0006_EB10_IO_TYER : BOOL; (* AT %MW186029.1 *) (* EB IO 타입 에러 *)
    _0006_EB30_CFG_ER : BOOL; (* AT %MW186046.0 *) (* EB 구성 에러 *)
    _0006_EB30_DEER : BOOL; (* AT %MW186046.1 *) (* EB 운전 중 탈락 *)
    _0006_EB30_IO_DEER : BOOL; (* AT %MW186047.2 *) (* EB IO 탈락 에러 *)
    _0006_EB30_IO_TYER : BOOL; (* AT %MW186047.1 *) (* EB IO 타입 에러 *)
    _0006_EB31_CFG_ER : BOOL; (* AT %MW186052.0 *) (* EB 구성 에러 *)
    _0006_EB31_DEER : BOOL; (* AT %MW186052.1 *) (* EB 운전 중 탈락 *)
    _0006_EB31_IO_DEER : BOOL; (* AT %MW186053.2 *) (* EB IO 탈락 에러 *)
    _0006_EB31_IO_TYER : BOOL; (* AT %MW186053.1 *) (* EB IO 타입 에러 *)
END_VAR
VAR_EXTERNAL RETAIN
    R368_1_M_NODE_4_07_통신_이상 : BOOL; (* AT %MW4024.8 *)
    S366_M_공정_불간섭 : BOOL; (* AT %MW3004.1 *) (* S366_M_공정_불간섭 *)
    S366_M_공정_제품감지_무 : BOOL; (* AT %MW3001.7 *) (* S366_M_공정_제품감지_무 *)
    S366_M_공정_차종_유 : BOOL; (* AT %MW3002.0 *) (* S366_M_공정_차종_유 *)
    S366_M_자동_운전중 : BOOL; (* AT %MW3000.4 *) (* S366 자동운전중 *)
    S368_LH_M_NODE_6_31_통신_이상 : BOOL; (* AT %MW4024.0 *)
    S368_M_HANGER_CLP_전진_LS_이상 : BOOL; (* AT %MW4111.5 *) (* S368_M_HANGER_CLP_전진_LS_이상 *)
    S368_M_HANGER_CLP_후진_LS_이상 : BOOL; (* AT %MW4111.6 *) (* S368_M_HANGER_CLP_후진_LS_이상 *)
    S368_M_HANGER_급전급기_전진_LS_이상 : BOOL; (* AT %MW4103.5 *)
    S368_M_HANGER_급전급기_후진_LS_이상 : BOOL; (* AT %MW4103.6 *)
    S368_M_LH_AX_CLAMP_전진_LS_이상 : BOOL; (* AT %MW4102.5 *) (* S368_M_LH_AX_CLAMP_전진_LS_이상 *)
    S368_M_LH_AX_CLAMP_후진_LS_이상 : BOOL; (* AT %MW4102.6 *) (* S368_M_LH_AX_CLAMP_후진_LS_이상 *)
    S368_M_LH_AX_LATCH_전진_LS_이상 : BOOL; (* AT %MW4100.5 *) (* S368_M_LH_AX_LATCH_전진_LS_이상 *)
    S368_M_LH_AX_LATCH_후진_LS_이상 : BOOL; (* AT %MW4100.6 *) (* S368_M_LH_AX_LATCH_후진_LS_이상 *)
    S368_M_LH_AX_SR_LAT_전진_LS_이상 : BOOL; (* AT %MW4101.5 *) (* S368_M_LH_AX_SR_LAT_전진_LS_이상 *)
    S368_M_LH_AX_SR_LAT_후진_LS_이상 : BOOL; (* AT %MW4101.6 *) (* S368_M_LH_AX_SR_LAT_후진_LS_이상 *)
    S368_M_LH_CP_OFF : BOOL; (* AT %MW4017.0 *) (* S368_M_LH_CP_OFF *)
    S368_M_R368_1_행거안착완료 : BOOL; (* AT %MW4001.2 *)
    S368_M_R369_1_안착완료 : BOOL; (* AT %MW4001.1 *)
    S368_M_RH_AX_CLAMP_전진_LS_이상 : BOOL; (* AT %MW4110.5 *) (* S368_M_RH_AX_CLAMP_전진_LS_이상 *)
    S368_M_RH_AX_CLAMP_후진_LS_이상 : BOOL; (* AT %MW4110.6 *) (* S368_M_RH_AX_CLAMP_후진_LS_이상 *)
    S368_M_RH_AX_LATCH_전진_LS_이상 : BOOL; (* AT %MW4108.5 *) (* S368_M_RH_AX_LATCH_전진_LS_이상 *)
    S368_M_RH_AX_LATCH_후진_LS_이상 : BOOL; (* AT %MW4108.6 *) (* S368_M_RH_AX_LATCH_후진_LS_이상 *)
    S368_M_RH_AX_SR_LAT_전진_LS_이상 : BOOL; (* AT %MW4109.5 *) (* S368_M_RH_AX_SR_LAT_전진_LS_이상 *)
    S368_M_RH_AX_SR_LAT_후진_LS_이상 : BOOL; (* AT %MW4109.6 *) (* S368_M_RH_AX_SR_LAT_후진_LS_이상 *)
    S368_M_RH_CP_OFF : BOOL; (* AT %MW4017.1 *) (* S368_M_RH_CP_OFF *)
    S368_M_공정_FRT_제품감지_무 : BOOL; (* AT %MW4001.8 *)
    S368_M_공정_FRT_제품감지_유 : BOOL; (* AT %MW4001.7 *)
    S368_M_공정_FRT_제품감지_이상 : BOOL; (* AT %MW4014.0 *)
    S368_M_공정_HANGER_감지_무 : BOOL; (* AT %MW4001.12 *)
    S368_M_공정_HANGER_감지_유 : BOOL; (* AT %MW4001.11 *)
    S368_M_공정_HANGER_감지_이상 : BOOL; (* AT %MW4014.2 *)
    S368_M_공정_RR_제품감지_무 : BOOL; (* AT %MW4001.10 *)
    S368_M_공정_RR_제품감지_유 : BOOL; (* AT %MW4001.9 *)
    S368_M_공정_RR_제품감지_이상 : BOOL; (* AT %MW4014.1 *)
    S368_M_공정_불간섭 : BOOL; (* AT %MW4004.1 *) (* S368_M_공정_불간섭 *)
    S368_M_공정_제품감지_무 : BOOL; (* AT %MW4001.6 *) (* S368_M_공정_제품감지_무 *)
    S368_M_공정_차종_유 : BOOL; (* AT %MW4002.0 *) (* S368_M_공정_차종_유 *)
    S368_M_자동_운전중 : BOOL; (* AT %MW4000.4 *) (* S368 자동운전중 *)
    S368_M_총괄_CP_이상 : BOOL; (* AT %MW4009.7 *) (* S368 CP OFF 이상 *)
    S368_M_총괄_CT_이상 : BOOL; (* AT %MW4010.4 *) (* S368   TACK TIME 이상 *)
    S368_M_총괄_EOCR_이상 : BOOL; (* AT %MW4009.8 *) (* S368_M_총괄_EOCR_이상 *)
    S368_M_총괄_INV_이상 : BOOL; (* AT %MW4009.9 *) (* S368_M_총괄_INV_이상 *)
    S368_M_총괄_LS_이상 : BOOL; (* AT %MW4009.15 *) (* S368 LS 이상 *)
    S368_M_총괄_MATCH_이상 : BOOL; (* AT %MW4010.0 *) (* S368 매트SW 이상 *)
    S368_M_총괄_MC_이상 : BOOL; (* AT %MW4009.13 *) (* S368_M_총괄_MC_이상 *)
    S368_M_총괄_NFB_이상 : BOOL; (* AT %MW4009.11 *) (* S368_M_총괄_NFB_이상 *)
    S368_M_총괄_ROBOT_이상 : BOOL; (* AT %MW4010.1 *) (* S368 ROBOT 이상 *)
    S368_M_총괄_SAFETY_이상 : BOOL; (* AT %MW4009.2 *) (* S368_M_총괄_SAFETY_이상 *)
    S368_M_총괄_공기압_이상 : BOOL; (* AT %MW4009.3 *) (* S368 공기압 이상 *)
    S368_M_총괄_사양_이상 : BOOL; (* AT %MW4009.6 *) (* S368 사양 이상 *)
    S368_M_총괄_오버런_이상 : BOOL; (* AT %MW4009.12 *) (* S368_M_총괄_오버런_이상 *)
    S368_M_총괄_용접타점수_이상 : BOOL; (* AT %MW4010.2 *) (* S368 용접타점수 이상 *)
    S368_M_총괄_이상 : BOOL; (* AT %MW4009.0 *) (* S368_M_총괄_이상 *)
    S368_M_총괄_제품감지_이상 : BOOL; (* AT %MW4009.4 *) (* S368 제품감지 이상 *)
    S368_M_총괄_차종_이상 : BOOL; (* AT %MW4009.5 *) (* S368 차종 이상 *)
    S368_M_총괄_통신_이상 : BOOL; (* AT %MW4009.14 *) (* S368 통신이상 *)
    S368_RH_M_NODE_6_30_통신_이상 : BOOL; (* AT %MW4024.1 *)
    전체_M_이상_리셋 : BOOL; (* AT %MW308.2 *) (* ALL공정 PB 이상리셋 *)
END_VAR

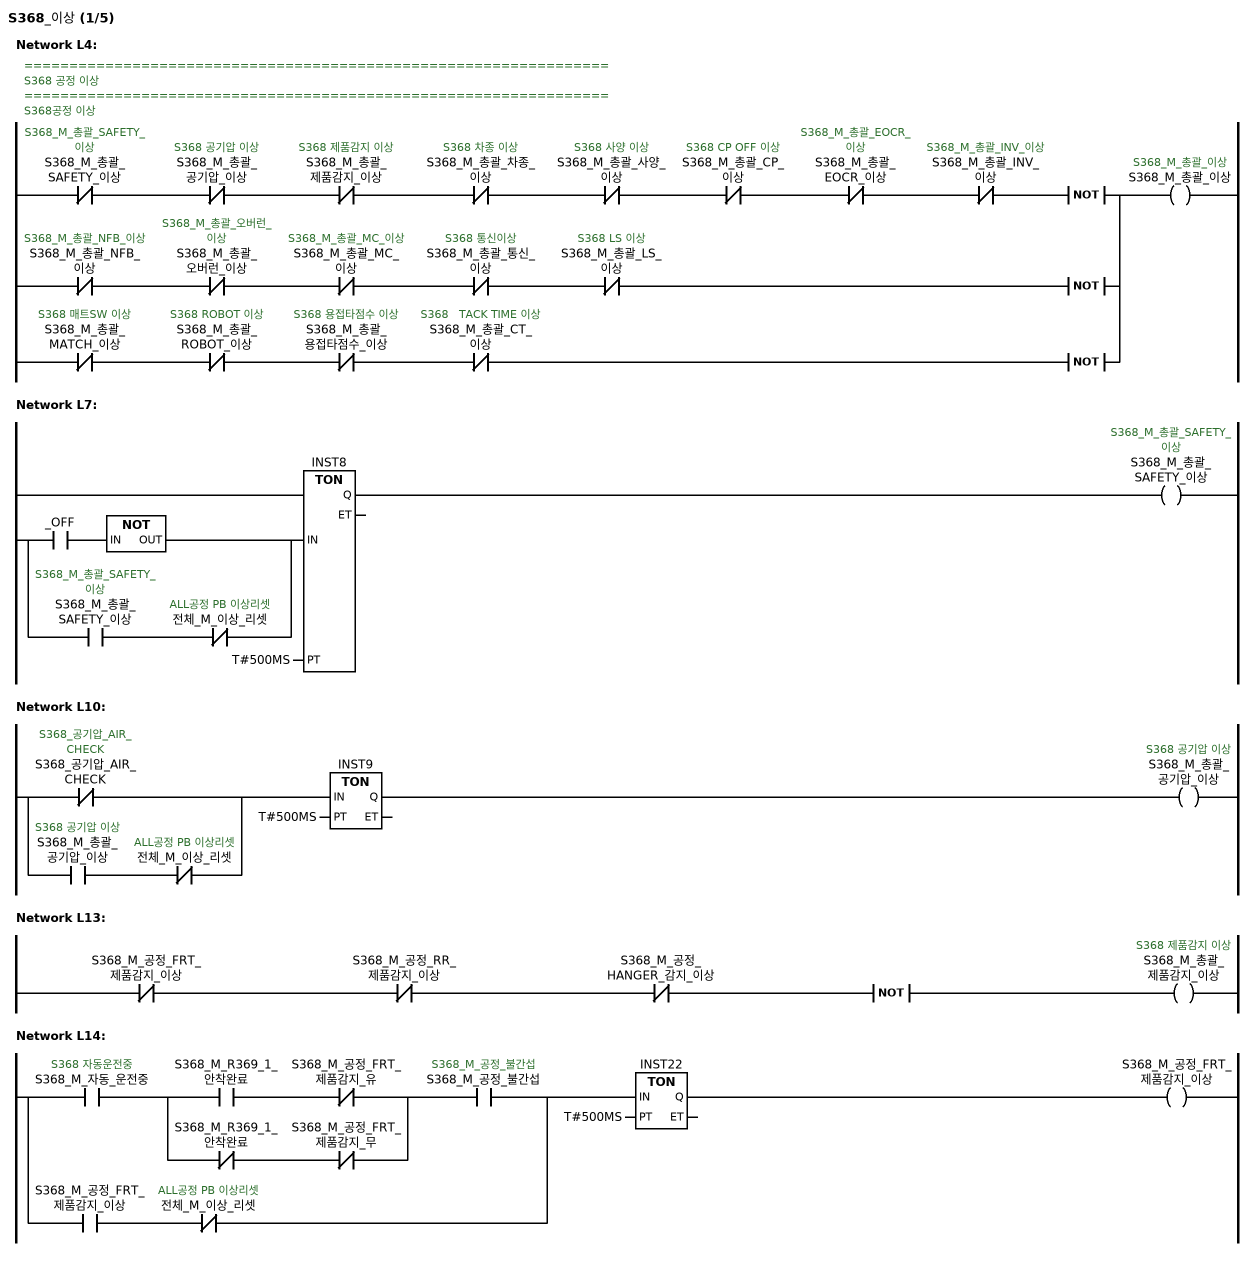
(* ================================================================= *)
(* S368 공정 이상 *)
(* ================================================================= *)
(* S368공정 이상 *)
(* Rung L4 *)
S368_M_총괄_이상 := NOT (NOT S368_M_총괄_SAFETY_이상 AND NOT S368_M_총괄_공기압_이상 AND NOT S368_M_총괄_제품감지_이상 AND NOT S368_M_총괄_차종_이상 AND NOT S368_M_총괄_사양_이상 AND NOT S368_M_총괄_CP_이상 AND NOT S368_M_총괄_EOCR_이상 AND NOT S368_M_총괄_INV_이상) OR NOT (NOT S368_M_총괄_NFB_이상 AND NOT S368_M_총괄_오버런_이상 AND NOT S368_M_총괄_MC_이상 AND NOT S368_M_총괄_통신_이상 AND NOT S368_M_총괄_LS_이상) OR NOT (NOT S368_M_총괄_MATCH_이상 AND NOT S368_M_총괄_ROBOT_이상 AND NOT S368_M_총괄_용접타점수_이상 AND NOT S368_M_총괄_CT_이상);
(* Rung L7 *)
INST8(IN := (NOT _OFF) OR (S368_M_총괄_SAFETY_이상 AND NOT 전체_M_이상_리셋), PT := T#500MS);
S368_M_총괄_SAFETY_이상 := INST8.Q;
(* Rung L10 *)
INST9(IN := NOT S368_공기압_AIR_CHECK OR (S368_M_총괄_공기압_이상 AND NOT 전체_M_이상_리셋), PT := T#500MS);
S368_M_총괄_공기압_이상 := INST9.Q;
(* Rung L13 *)
S368_M_총괄_제품감지_이상 := NOT (NOT S368_M_공정_FRT_제품감지_이상 AND NOT S368_M_공정_RR_제품감지_이상 AND NOT S368_M_공정_HANGER_감지_이상);
(* Rung L14 *)
INST22(IN := (S368_M_자동_운전중 AND ((S368_M_R369_1_안착완료 AND NOT S368_M_공정_FRT_제품감지_유) OR (NOT S368_M_R369_1_안착완료 AND NOT S368_M_공정_FRT_제품감지_무)) AND S368_M_공정_불간섭) OR (S368_M_공정_FRT_제품감지_이상 AND NOT 전체_M_이상_리셋), PT := T#500MS);
S368_M_공정_FRT_제품감지_이상 := INST22.Q;

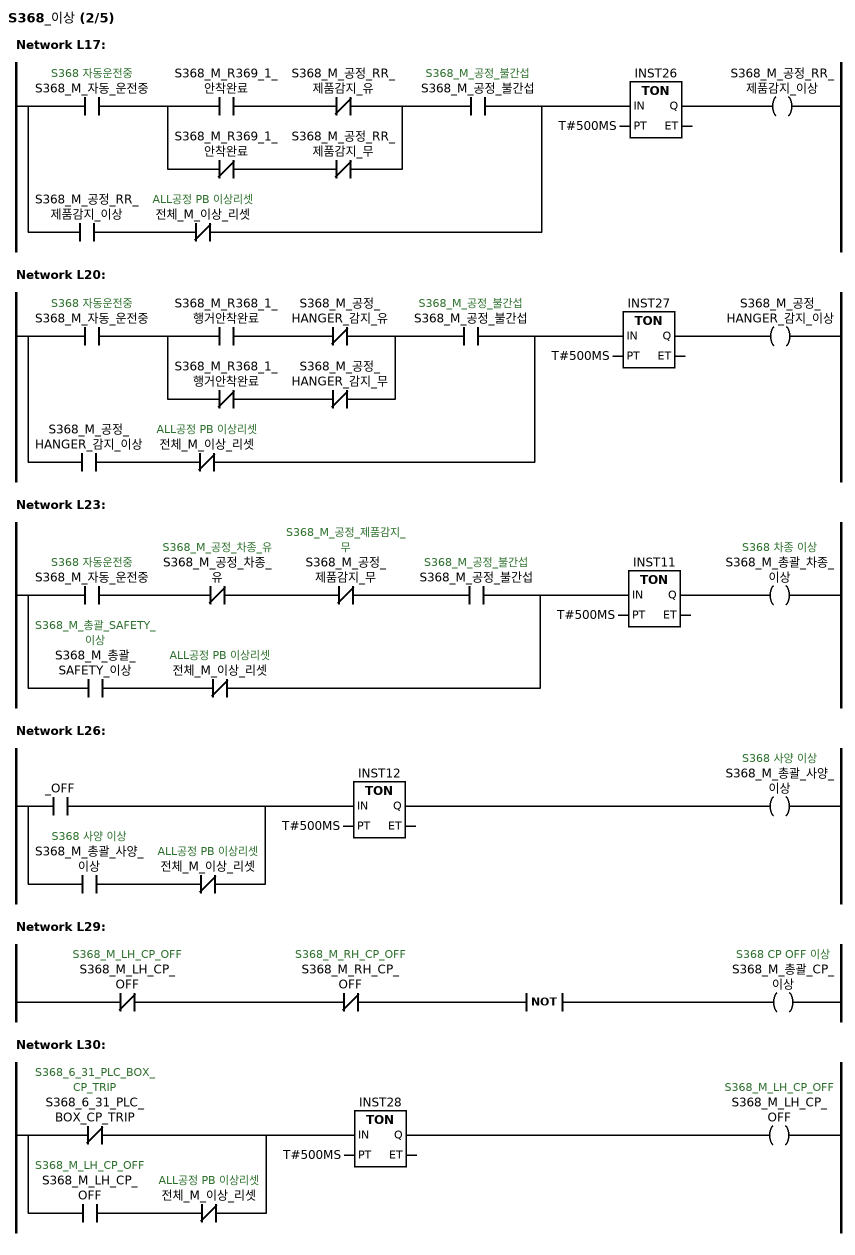
(* Rung L17 *)
INST26(IN := (S368_M_자동_운전중 AND ((S368_M_R369_1_안착완료 AND NOT S368_M_공정_RR_제품감지_유) OR (NOT S368_M_R369_1_안착완료 AND NOT S368_M_공정_RR_제품감지_무)) AND S368_M_공정_불간섭) OR (S368_M_공정_RR_제품감지_이상 AND NOT 전체_M_이상_리셋), PT := T#500MS);
S368_M_공정_RR_제품감지_이상 := INST26.Q;
(* Rung L20 *)
INST27(IN := (S368_M_자동_운전중 AND ((S368_M_R368_1_행거안착완료 AND NOT S368_M_공정_HANGER_감지_유) OR (NOT S368_M_R368_1_행거안착완료 AND NOT S368_M_공정_HANGER_감지_무)) AND S368_M_공정_불간섭) OR (S368_M_공정_HANGER_감지_이상 AND NOT 전체_M_이상_리셋), PT := T#500MS);
S368_M_공정_HANGER_감지_이상 := INST27.Q;
(* Rung L23 *)
INST11(IN := (S368_M_자동_운전중 AND NOT S368_M_공정_차종_유 AND NOT S368_M_공정_제품감지_무 AND S368_M_공정_불간섭) OR (S368_M_총괄_SAFETY_이상 AND NOT 전체_M_이상_리셋), PT := T#500MS);
S368_M_총괄_차종_이상 := INST11.Q;
(* Rung L26 *)
INST12(IN := _OFF OR (S368_M_총괄_사양_이상 AND NOT 전체_M_이상_리셋), PT := T#500MS);
S368_M_총괄_사양_이상 := INST12.Q;
(* Rung L29 *)
S368_M_총괄_CP_이상 := NOT (NOT S368_M_LH_CP_OFF AND NOT S368_M_RH_CP_OFF);
(* Rung L30 *)
INST28(IN := NOT S368_6_31_PLC_BOX_CP_TRIP OR (S368_M_LH_CP_OFF AND NOT 전체_M_이상_리셋), PT := T#500MS);
S368_M_LH_CP_OFF := INST28.Q;

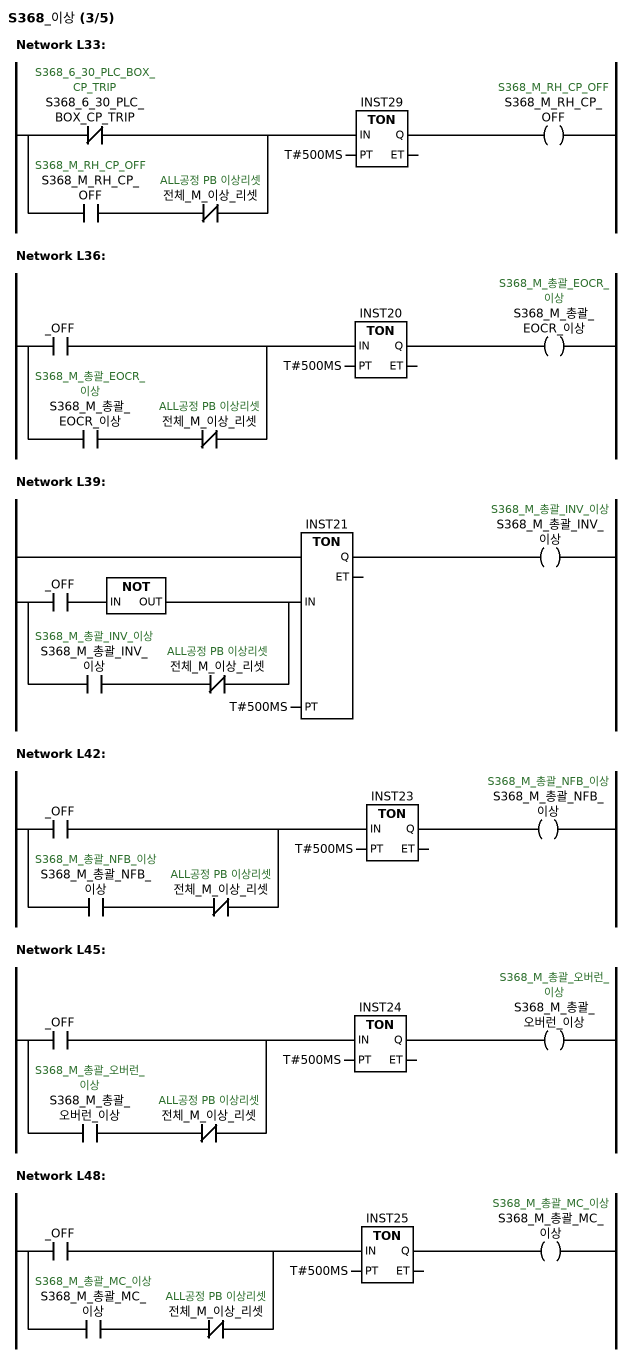
(* Rung L33 *)
INST29(IN := NOT S368_6_30_PLC_BOX_CP_TRIP OR (S368_M_RH_CP_OFF AND NOT 전체_M_이상_리셋), PT := T#500MS);
S368_M_RH_CP_OFF := INST29.Q;
(* Rung L36 *)
INST20(IN := _OFF OR (S368_M_총괄_EOCR_이상 AND NOT 전체_M_이상_리셋), PT := T#500MS);
S368_M_총괄_EOCR_이상 := INST20.Q;
(* Rung L39 *)
INST21(IN := (NOT _OFF) OR (S368_M_총괄_INV_이상 AND NOT 전체_M_이상_리셋), PT := T#500MS);
S368_M_총괄_INV_이상 := INST21.Q;
(* Rung L42 *)
INST23(IN := _OFF OR (S368_M_총괄_NFB_이상 AND NOT 전체_M_이상_리셋), PT := T#500MS);
S368_M_총괄_NFB_이상 := INST23.Q;
(* Rung L45 *)
INST24(IN := _OFF OR (S368_M_총괄_오버런_이상 AND NOT 전체_M_이상_리셋), PT := T#500MS);
S368_M_총괄_오버런_이상 := INST24.Q;
(* Rung L48 *)
INST25(IN := _OFF OR (S368_M_총괄_MC_이상 AND NOT 전체_M_이상_리셋), PT := T#500MS);
S368_M_총괄_MC_이상 := INST25.Q;

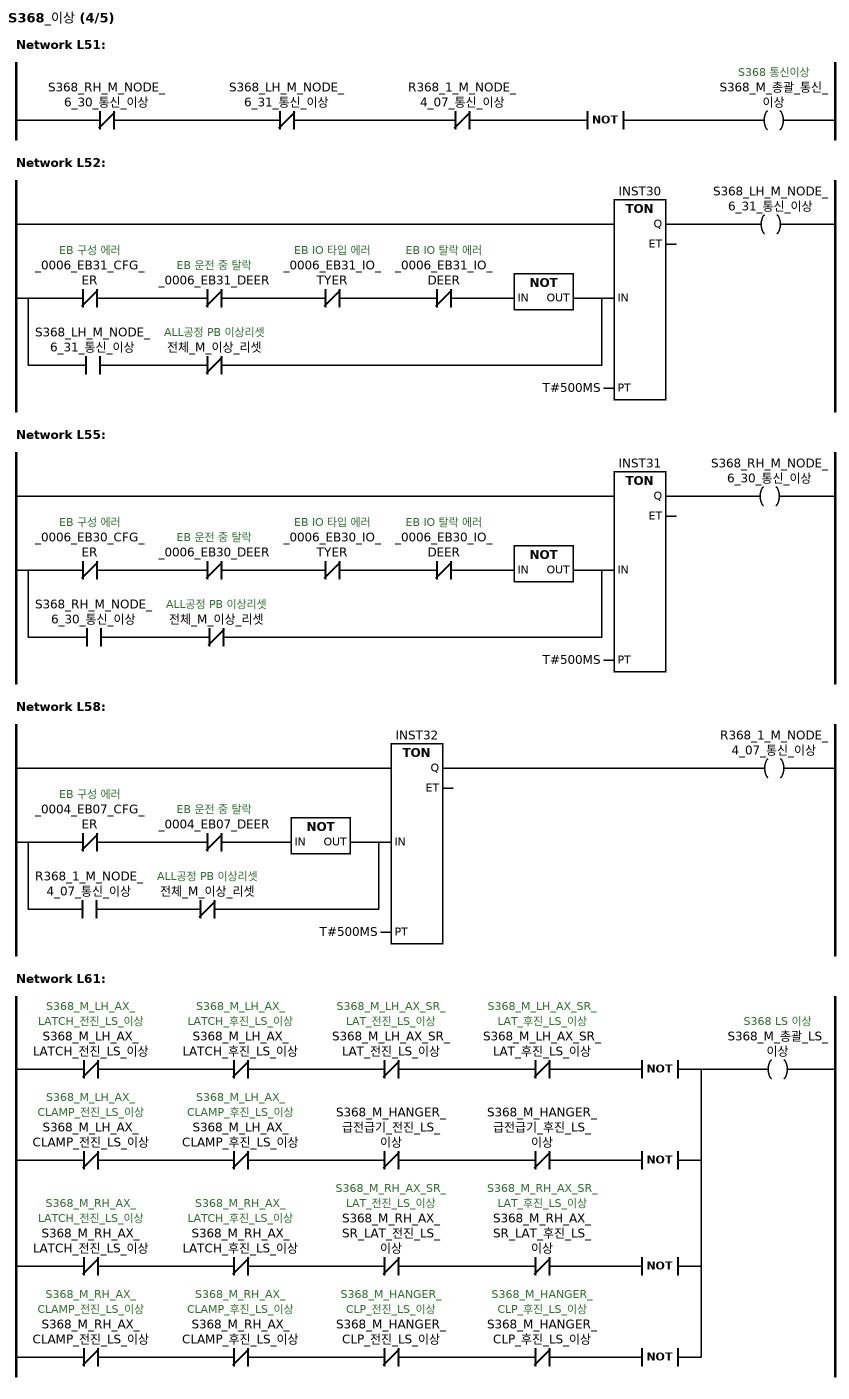
(* Rung L51 *)
S368_M_총괄_통신_이상 := NOT (NOT S368_RH_M_NODE_6_30_통신_이상 AND NOT S368_LH_M_NODE_6_31_통신_이상 AND NOT R368_1_M_NODE_4_07_통신_이상);
(* Rung L52 *)
INST30(IN := (NOT (NOT _0006_EB31_CFG_ER AND NOT _0006_EB31_DEER AND NOT _0006_EB31_IO_TYER AND NOT _0006_EB31_IO_DEER)) OR (S368_LH_M_NODE_6_31_통신_이상 AND NOT 전체_M_이상_리셋), PT := T#500MS);
S368_LH_M_NODE_6_31_통신_이상 := INST30.Q;
(* Rung L55 *)
INST31(IN := (NOT (NOT _0006_EB30_CFG_ER AND NOT _0006_EB30_DEER AND NOT _0006_EB30_IO_TYER AND NOT _0006_EB30_IO_DEER)) OR (S368_RH_M_NODE_6_30_통신_이상 AND NOT 전체_M_이상_리셋), PT := T#500MS);
S368_RH_M_NODE_6_30_통신_이상 := INST31.Q;
(* Rung L58 *)
INST32(IN := (NOT (NOT _0004_EB07_CFG_ER AND NOT _0004_EB07_DEER)) OR (R368_1_M_NODE_4_07_통신_이상 AND NOT 전체_M_이상_리셋), PT := T#500MS);
R368_1_M_NODE_4_07_통신_이상 := INST32.Q;
(* Rung L61 *)
S368_M_총괄_LS_이상 := NOT (NOT S368_M_LH_AX_LATCH_전진_LS_이상 AND NOT S368_M_LH_AX_LATCH_후진_LS_이상 AND NOT S368_M_LH_AX_SR_LAT_전진_LS_이상 AND NOT S368_M_LH_AX_SR_LAT_후진_LS_이상) OR NOT (NOT S368_M_LH_AX_CLAMP_전진_LS_이상 AND NOT S368_M_LH_AX_CLAMP_후진_LS_이상 AND NOT S368_M_HANGER_급전급기_전진_LS_이상 AND NOT S368_M_HANGER_급전급기_후진_LS_이상) OR NOT (NOT S368_M_RH_AX_LATCH_전진_LS_이상 AND NOT S368_M_RH_AX_LATCH_후진_LS_이상 AND NOT S368_M_RH_AX_SR_LAT_전진_LS_이상 AND NOT S368_M_RH_AX_SR_LAT_후진_LS_이상) OR NOT (NOT S368_M_RH_AX_CLAMP_전진_LS_이상 AND NOT S368_M_RH_AX_CLAMP_후진_LS_이상 AND NOT S368_M_HANGER_CLP_전진_LS_이상 AND NOT S368_M_HANGER_CLP_후진_LS_이상);

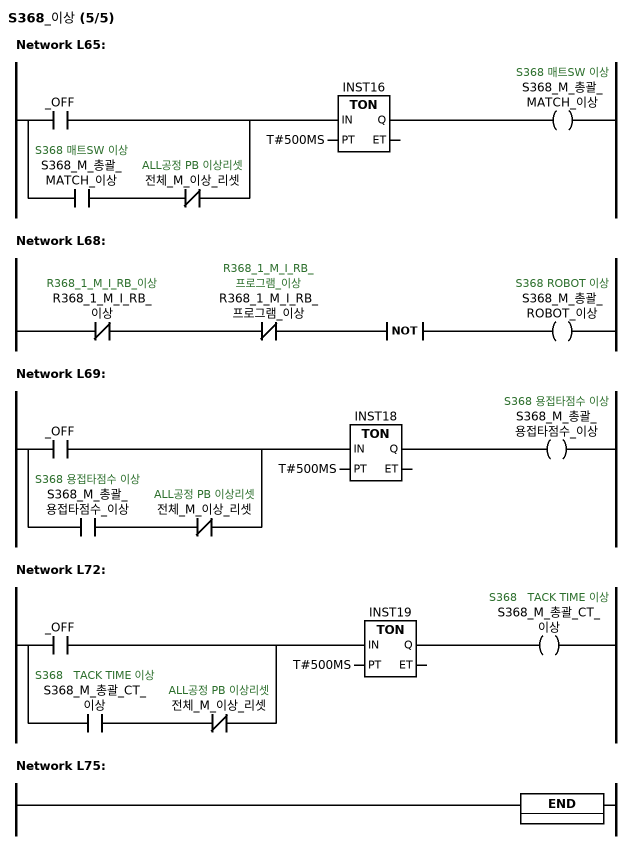
(* Rung L65 *)
INST16(IN := _OFF OR (S368_M_총괄_MATCH_이상 AND NOT 전체_M_이상_리셋), PT := T#500MS);
S368_M_총괄_MATCH_이상 := INST16.Q;
(* Rung L68 *)
S368_M_총괄_ROBOT_이상 := NOT (NOT R368_1_M_I_RB_이상 AND NOT R368_1_M_I_RB_프로그램_이상);
(* Rung L69 *)
INST18(IN := _OFF OR (S368_M_총괄_용접타점수_이상 AND NOT 전체_M_이상_리셋), PT := T#500MS);
S368_M_총괄_용접타점수_이상 := INST18.Q;
(* Rung L72 *)
INST19(IN := _OFF OR (S368_M_총괄_CT_이상 AND NOT 전체_M_이상_리셋), PT := T#500MS);
S368_M_총괄_CT_이상 := INST19.Q;
(* Rung L75 *)
END();
END_PROGRAM

PROGRAM S369_1_유틸리티 (* task: 스캔 프로그램 *)
VAR_EXTERNAL RETAIN
    ALWAYS_ON : BOOL; (* AT %MW3.1 *) (* 항시 ON *)
    HMI_M_선택_MOD_S368 : BOOL; (* AT %MW6.6 *) (* HMI M 선택 MOD S368 *)
    HMI_M_선택_MOD_S369_1 : BOOL; (* AT %MW6.7 *) (* HMI M 선택 MOD S369_1 *)
    R369_1_M_SEQ : WORD; (* AT %MW10060 *) (* R369 1 M SEQ *)
    R369_1_M_차종1_AX : BOOL; (* AT %MW10061.0 *) (* R369 1 M 차종1 AX *)
    R369_1_M_차종1_B : BOOL; (* AT %MW10061.1 *) (* R369 1 M 차종1 B *)
    R369_1_M_차종1_C : BOOL; (* AT %MW10061.2 *) (* R369 1 M 차종1 C *)
    R369_1_M_차종1_D : BOOL; (* AT %MW10061.3 *) (* R369 1 M 차종1 D *)
    R369_1_M_차종1_E : BOOL; (* AT %MW10061.4 *) (* R369 1 M 차종1 E *)
    R369_1_M_차종1_F : BOOL; (* AT %MW10061.5 *) (* R369 1 M 차종1 F *)
    R369_1_M_차종1_G : BOOL; (* AT %MW10061.6 *) (* R369 1 M 차종1 G *)
    R369_1_M_차종1_H : BOOL; (* AT %MW10061.7 *) (* R369 1 M 차종1 H *)
    R369_1_M_차종2_3DR : BOOL; (* AT %MW10061.8 *) (* R369 1 M 차종2 3DR *)
    R369_1_M_차종2_4DR : BOOL; (* AT %MW10061.9 *) (* R369 1 M 차종2 4DR *)
    R369_1_M_차종2_5DR : BOOL; (* AT %MW10061.10 *) (* R369 1 M 차종2 5DR *)
    R369_1_M_차종2_SP1 : BOOL; (* AT %MW10061.12 *) (* R369 1 M 차종2 SP1 *)
    R369_1_M_차종2_SP2 : BOOL; (* AT %MW10061.13 *) (* R369 1 M 차종2 SP2 *)
    R369_1_M_차종2_WGN : BOOL; (* AT %MW10061.11 *) (* R369 1 M 차종2 WGN *)
    R369_1_M_차종3_LHD : BOOL; (* AT %MW10061.14 *) (* R369 1 M 차종3 LHD *)
    R369_1_M_차종3_RHD : BOOL; (* AT %MW10061.15 *) (* R369 1 M 차종3 RHD *)
    R369_1_M_차종4_EEC : BOOL; (* AT %MW10062.3 *) (* R369 1 M 차종4 EEC *)
    R369_1_M_차종4_SP1 : BOOL; (* AT %MW10062.8 *) (* R369 1 M 차종4 SP1 *)
    R369_1_M_차종4_SP2 : BOOL; (* AT %MW10062.9 *) (* R369 1 M 차종4 SP2 *)
    R369_1_M_차종4_SP3 : BOOL; (* AT %MW10062.11 *) (* R369 1 M 차종4 SP3 *)
    R369_1_M_차종4_SP4 : BOOL; (* AT %MW10062.12 *) (* R369 1 M 차종4 SP4 *)
    R369_1_M_차종4_SP5 : BOOL; (* AT %MW10062.13 *) (* R369 1 M 차종4 SP5 *)
    R369_1_M_차종4_SP6 : BOOL; (* AT %MW10062.14 *) (* R369 1 M 차종4 SP6 *)
    R369_1_M_차종4_SP7 : BOOL; (* AT %MW10062.15 *) (* R369 1 M 차종4 SP7 *)
    R369_1_M_차종4_내수 : BOOL; (* AT %MW10062.0 *) (* R369 1 M 차종4 내수 *)
    R369_1_M_차종4_러시아 : BOOL; (* AT %MW10062.10 *) (* R369 1 M 차종4 러시아 *)
    R369_1_M_차종4_북미 : BOOL; (* AT %MW10062.2 *) (* R369 1 M 차종4 북미 *)
    R369_1_M_차종4_브라질 : BOOL; (* AT %MW10062.7 *) (* R369 1 M 차종4 브라질 *)
    R369_1_M_차종4_수출 : BOOL; (* AT %MW10062.1 *) (* R369 1 M 차종4 수출 *)
    R369_1_M_차종4_중국 : BOOL; (* AT %MW10062.6 *) (* R369 1 M 차종4 중국 *)
    R369_1_M_차종4_중동 : BOOL; (* AT %MW10062.5 *) (* R369 1 M 차종4 중동 *)
    R369_1_M_차종4_호주 : BOOL; (* AT %MW10062.4 *) (* R369 1 M 차종4 호주 *)
    R369_1_M_차종5_AT : BOOL; (* AT %MW10063.1 *) (* R369 1 M 차종5 AT *)
    R369_1_M_차종5_MT : BOOL; (* AT %MW10063.0 *) (* R369 1 M 차종5 MT *)
    R369_1_M_차종5_SP1 : BOOL; (* AT %MW10063.2 *) (* R369 1 M 차종5 SP1 *)
    R369_1_M_차종6_DSROOF : BOOL; (* AT %MW10063.6 *) (* R369 1 M 차종6 DSROOF *)
    R369_1_M_차종6_SP1 : BOOL; (* AT %MW10063.7 *) (* R369 1 M 차종6 SP1 *)
    R369_1_M_차종6_썬루프 : BOOL; (* AT %MW10063.4 *) (* R369 1 M 차종6 썬루프 *)
    R369_1_M_차종6_일반루프 : BOOL; (* AT %MW10063.3 *) (* R369 1 M 차종6 일반루프 *)
    R369_1_M_차종6_파노라마루프 : BOOL; (* AT %MW10063.5 *) (* R369 1 M 차종6 파노라마루프 *)
    R369_1_M_차종7_DSL : BOOL; (* AT %MW10063.9 *) (* R369 1 M 차종7 DSL *)
    R369_1_M_차종7_GSL : BOOL; (* AT %MW10063.8 *) (* R369 1 M 차종7 GSL *)
    R369_1_M_차종7_SP1 : BOOL; (* AT %MW10063.10 *) (* R369 1 M 차종7 SP1 *)
    R369_1_M_차종7_SP2 : BOOL; (* AT %MW10063.11 *) (* R369 1 M 차종7 SP2 *)
    R369_1_M_차종7_SP3 : BOOL; (* AT %MW10063.12 *) (* R369 1 M 차종7 SP3 *)
    R369_1_M_차종7_SP4 : BOOL; (* AT %MW10063.13 *) (* R369 1 M 차종7 SP4 *)
    R369_1_M_차종7_SP5 : BOOL; (* AT %MW10063.14 *) (* R369 1 M 차종7 SP5 *)
    R369_1_M_차종7_SP6 : BOOL; (* AT %MW10063.15 *) (* R369 1 M 차종7 SP6 *)
    R369_1_M_차종8_2WD : BOOL; (* AT %MW10064.0 *) (* R369 1 M 차종8 2WD *)
    R369_1_M_차종8_4WD : BOOL; (* AT %MW10064.1 *) (* R369 1 M 차종8 4WD *)
    R369_1_M_차종8_SP1 : BOOL; (* AT %MW10064.2 *) (* R369 1 M 차종8 SP1 *)
    R369_1_M_차종9_MPI : BOOL; (* AT %MW10064.3 *) (* R369 1 M 차종9 MPI *)
    R369_1_M_차종9_SP1 : BOOL; (* AT %MW10064.5 *) (* R369 1 M 차종9 SP1 *)
    R369_1_M_차종9_SP10 : BOOL; (* AT %MW10064.14 *) (* R369 1 M 차종9 SP10 *)
    R369_1_M_차종9_SP11 : BOOL; (* AT %MW10064.15 *) (* R369 1 M 차종9 SP11 *)
    R369_1_M_차종9_SP2 : BOOL; (* AT %MW10064.6 *) (* R369 1 M 차종9 SP2 *)
    R369_1_M_차종9_SP3 : BOOL; (* AT %MW10064.7 *) (* R369 1 M 차종9 SP3 *)
    R369_1_M_차종9_SP4 : BOOL; (* AT %MW10064.8 *) (* R369 1 M 차종9 SP4 *)
    R369_1_M_차종9_SP5 : BOOL; (* AT %MW10064.9 *) (* R369 1 M 차종9 SP5 *)
    R369_1_M_차종9_SP6 : BOOL; (* AT %MW10064.10 *) (* R369 1 M 차종9 SP6 *)
    R369_1_M_차종9_SP7 : BOOL; (* AT %MW10064.11 *) (* R369 1 M 차종9 SP7 *)
    R369_1_M_차종9_SP8 : BOOL; (* AT %MW10064.12 *) (* R369 1 M 차종9 SP8 *)
    R369_1_M_차종9_SP9 : BOOL; (* AT %MW10064.13 *) (* R369 1 M 차종9 SP9 *)
    R369_1_M_차종9_T_GDI : BOOL; (* AT %MW10064.4 *) (* R369 1 M 차종9 T GDI *)
    R369_1_M_차종_OPT1_R_RACK_무 : BOOL; (* AT %MW10065.3 *) (* R369 1 M 차종 OPT1 R RACK 무 *)
    R369_1_M_차종_OPT1_R_RACK_유 : BOOL; (* AT %MW10065.2 *) (* R369 1 M 차종 OPT1 R RACK 유 *)
    R369_1_M_차종_OPT1_S_REP_EATER_무 : BOOL; (* AT %MW10065.7 *) (* R369 1 M 차종 OPT1 S REP EATER 무 *)
    R369_1_M_차종_OPT1_S_REP_EATER_유 : BOOL; (* AT %MW10065.6 *) (* R369 1 M 차종 OPT1 S REP EATER 유 *)
    R369_1_M_차종_OPT1_VAN_무 : BOOL; (* AT %MW10065.9 *) (* R369 1 M 차종 OPT1 VAN 무 *)
    R369_1_M_차종_OPT1_VAN_유 : BOOL; (* AT %MW10065.8 *) (* R369 1 M 차종 OPT1 VAN 유 *)
    R369_1_M_차종_OPT1_슬라이딩_무 : BOOL; (* AT %MW10065.1 *) (* R369 1 M 차종 OPT1 슬라이딩 무 *)
    R369_1_M_차종_OPT1_슬라이딩_유 : BOOL; (* AT %MW10065.0 *) (* R369 1 M 차종 OPT1 슬라이딩 유 *)
    R369_1_M_차종_OPT1_폴딩_무 : BOOL; (* AT %MW10065.5 *) (* R369 1 M 차종 OPT1 폴딩 무 *)
    R369_1_M_차종_OPT1_폴딩_유 : BOOL; (* AT %MW10065.4 *) (* R369 1 M 차종 OPT1 폴딩 유 *)
    R369_1_M_차종_무 : BOOL; (* AT %MW4502.3 *)
    R369_1_M_차종_유 : BOOL; (* AT %MW4502.2 *)
    R369_2_M_SEQ : WORD; (* AT %MW10080 *) (* R369 2 M SEQ *)
    R369_2_M_차종1_AX : BOOL; (* AT %MW10081.0 *) (* R369 2 M 차종1 AX *)
    R369_2_M_차종1_B : BOOL; (* AT %MW10081.1 *) (* R369 2 M 차종1 B *)
    R369_2_M_차종1_C : BOOL; (* AT %MW10081.2 *) (* R369 2 M 차종1 C *)
    R369_2_M_차종1_D : BOOL; (* AT %MW10081.3 *) (* R369 2 M 차종1 D *)
    R369_2_M_차종1_E : BOOL; (* AT %MW10081.4 *) (* R369 2 M 차종1 E *)
    R369_2_M_차종1_F : BOOL; (* AT %MW10081.5 *) (* R369 2 M 차종1 F *)
    R369_2_M_차종1_G : BOOL; (* AT %MW10081.6 *) (* R369 2 M 차종1 G *)
    R369_2_M_차종1_H : BOOL; (* AT %MW10081.7 *) (* R369 2 M 차종1 H *)
    R369_2_M_차종2_3DR : BOOL; (* AT %MW10081.8 *) (* R369 2 M 차종2 3DR *)
    R369_2_M_차종2_4DR : BOOL; (* AT %MW10081.9 *) (* R369 2 M 차종2 4DR *)
    R369_2_M_차종2_5DR : BOOL; (* AT %MW10081.10 *) (* R369 2 M 차종2 5DR *)
    R369_2_M_차종2_SP1 : BOOL; (* AT %MW10081.12 *) (* R369 2 M 차종2 SP1 *)
    R369_2_M_차종2_SP2 : BOOL; (* AT %MW10081.13 *) (* R369 2 M 차종2 SP2 *)
    R369_2_M_차종2_WGN : BOOL; (* AT %MW10081.11 *) (* R369 2 M 차종2 WGN *)
    R369_2_M_차종3_LHD : BOOL; (* AT %MW10081.14 *) (* R369 2 M 차종3 LHD *)
    R369_2_M_차종3_RHD : BOOL; (* AT %MW10081.15 *) (* R369 2 M 차종3 RHD *)
    R369_2_M_차종4_EEC : BOOL; (* AT %MW10082.3 *) (* R369 2 M 차종4 EEC *)
    R369_2_M_차종4_SP1 : BOOL; (* AT %MW10082.8 *) (* R369 2 M 차종4 SP1 *)
    R369_2_M_차종4_SP2 : BOOL; (* AT %MW10082.9 *) (* R369 2 M 차종4 SP2 *)
    R369_2_M_차종4_SP3 : BOOL; (* AT %MW10082.11 *) (* R369 2 M 차종4 SP3 *)
    R369_2_M_차종4_SP4 : BOOL; (* AT %MW10082.12 *) (* R369 2 M 차종4 SP4 *)
    R369_2_M_차종4_SP5 : BOOL; (* AT %MW10082.13 *) (* R369 2 M 차종4 SP5 *)
    R369_2_M_차종4_SP6 : BOOL; (* AT %MW10082.14 *) (* R369 2 M 차종4 SP6 *)
    R369_2_M_차종4_SP7 : BOOL; (* AT %MW10082.15 *) (* R369 2 M 차종4 SP7 *)
    R369_2_M_차종4_내수 : BOOL; (* AT %MW10082.0 *) (* R369 2 M 차종4 내수 *)
    R369_2_M_차종4_러시아 : BOOL; (* AT %MW10082.10 *) (* R369 2 M 차종4 러시아 *)
    R369_2_M_차종4_북미 : BOOL; (* AT %MW10082.2 *) (* R369 2 M 차종4 북미 *)
    R369_2_M_차종4_브라질 : BOOL; (* AT %MW10082.7 *) (* R369 2 M 차종4 브라질 *)
    R369_2_M_차종4_수출 : BOOL; (* AT %MW10082.1 *) (* R369 2 M 차종4 수출 *)
    R369_2_M_차종4_중국 : BOOL; (* AT %MW10082.6 *) (* R369 2 M 차종4 중국 *)
    R369_2_M_차종4_중동 : BOOL; (* AT %MW10082.5 *) (* R369 2 M 차종4 중동 *)
    R369_2_M_차종4_호주 : BOOL; (* AT %MW10082.4 *) (* R369 2 M 차종4 호주 *)
    R369_2_M_차종5_AT : BOOL; (* AT %MW10083.1 *) (* R369 2 M 차종5 AT *)
    R369_2_M_차종5_MT : BOOL; (* AT %MW10083.0 *) (* R369 2 M 차종5 MT *)
    R369_2_M_차종5_SP1 : BOOL; (* AT %MW10083.2 *) (* R369 2 M 차종5 SP1 *)
    R369_2_M_차종6_DSROOF : BOOL; (* AT %MW10083.6 *) (* R369 2 M 차종6 DSROOF *)
    R369_2_M_차종6_SP1 : BOOL; (* AT %MW10083.7 *) (* R369 2 M 차종6 SP1 *)
    R369_2_M_차종6_썬루프 : BOOL; (* AT %MW10083.4 *) (* R369 2 M 차종6 썬루프 *)
    R369_2_M_차종6_일반루프 : BOOL; (* AT %MW10083.3 *) (* R369 2 M 차종6 일반루프 *)
    R369_2_M_차종6_파노라마루프 : BOOL; (* AT %MW10083.5 *) (* R369 2 M 차종6 파노라마루프 *)
    R369_2_M_차종7_DSL : BOOL; (* AT %MW10083.9 *) (* R369 2 M 차종7 DSL *)
    R369_2_M_차종7_GSL : BOOL; (* AT %MW10083.8 *) (* R369 2 M 차종7 GSL *)
    R369_2_M_차종7_SP1 : BOOL; (* AT %MW10083.10 *) (* R369 2 M 차종7 SP1 *)
    R369_2_M_차종7_SP2 : BOOL; (* AT %MW10083.11 *) (* R369 2 M 차종7 SP2 *)
    R369_2_M_차종7_SP3 : BOOL; (* AT %MW10083.12 *) (* R369 2 M 차종7 SP3 *)
    R369_2_M_차종7_SP4 : BOOL; (* AT %MW10083.13 *) (* R369 2 M 차종7 SP4 *)
    R369_2_M_차종7_SP5 : BOOL; (* AT %MW10083.14 *) (* R369 2 M 차종7 SP5 *)
    R369_2_M_차종7_SP6 : BOOL; (* AT %MW10083.15 *) (* R369 2 M 차종7 SP6 *)
    R369_2_M_차종8_2WD : BOOL; (* AT %MW10084.0 *) (* R369 2 M 차종8 2WD *)
    R369_2_M_차종8_4WD : BOOL; (* AT %MW10084.1 *) (* R369 2 M 차종8 4WD *)
    R369_2_M_차종8_SP1 : BOOL; (* AT %MW10084.2 *) (* R369 2 M 차종8 SP1 *)
    R369_2_M_차종9_MPI : BOOL; (* AT %MW10084.3 *) (* R369 2 M 차종9 MPI *)
    R369_2_M_차종9_SP1 : BOOL; (* AT %MW10084.5 *) (* R369 2 M 차종9 SP1 *)
    R369_2_M_차종9_SP10 : BOOL; (* AT %MW10084.14 *) (* R369 2 M 차종9 SP10 *)
    R369_2_M_차종9_SP11 : BOOL; (* AT %MW10084.15 *) (* R369 2 M 차종9 SP11 *)
    R369_2_M_차종9_SP2 : BOOL; (* AT %MW10084.6 *) (* R369 2 M 차종9 SP2 *)
    R369_2_M_차종9_SP3 : BOOL; (* AT %MW10084.7 *) (* R369 2 M 차종9 SP3 *)
    R369_2_M_차종9_SP4 : BOOL; (* AT %MW10084.8 *) (* R369 2 M 차종9 SP4 *)
    R369_2_M_차종9_SP5 : BOOL; (* AT %MW10084.9 *) (* R369 2 M 차종9 SP5 *)
    R369_2_M_차종9_SP6 : BOOL; (* AT %MW10084.10 *) (* R369 2 M 차종9 SP6 *)
    R369_2_M_차종9_SP7 : BOOL; (* AT %MW10084.11 *) (* R369 2 M 차종9 SP7 *)
    R369_2_M_차종9_SP8 : BOOL; (* AT %MW10084.12 *) (* R369 2 M 차종9 SP8 *)
    R369_2_M_차종9_SP9 : BOOL; (* AT %MW10084.13 *) (* R369 2 M 차종9 SP9 *)
    R369_2_M_차종9_T_GDI : BOOL; (* AT %MW10084.4 *) (* R369 2 M 차종9 T GDI *)
    R369_2_M_차종_OPT1_R_RACK_무 : BOOL; (* AT %MW10085.3 *) (* R369 2 M 차종 OPT1 R RACK 무 *)
    R369_2_M_차종_OPT1_R_RACK_유 : BOOL; (* AT %MW10085.2 *) (* R369 2 M 차종 OPT1 R RACK 유 *)
    R369_2_M_차종_OPT1_S_REP_EATER_무 : BOOL; (* AT %MW10085.7 *) (* R369 2 M 차종 OPT1 S REP EATER 무 *)
    R369_2_M_차종_OPT1_S_REP_EATER_유 : BOOL; (* AT %MW10085.6 *) (* R369 2 M 차종 OPT1 S REP EATER 유 *)
    R369_2_M_차종_OPT1_VAN_무 : BOOL; (* AT %MW10085.9 *) (* R369 2 M 차종 OPT1 VAN 무 *)
    R369_2_M_차종_OPT1_VAN_유 : BOOL; (* AT %MW10085.8 *) (* R369 2 M 차종 OPT1 VAN 유 *)
    R369_2_M_차종_OPT1_슬라이딩_무 : BOOL; (* AT %MW10085.1 *) (* R369 2 M 차종 OPT1 슬라이딩 무 *)
    R369_2_M_차종_OPT1_슬라이딩_유 : BOOL; (* AT %MW10085.0 *) (* R369 2 M 차종 OPT1 슬라이딩 유 *)
    R369_2_M_차종_OPT1_폴딩_무 : BOOL; (* AT %MW10085.5 *) (* R369 2 M 차종 OPT1 폴딩 무 *)
    R369_2_M_차종_OPT1_폴딩_유 : BOOL; (* AT %MW10085.4 *) (* R369 2 M 차종 OPT1 폴딩 유 *)
    R369_2_M_차종_무 : BOOL; (* AT %MW4502.5 *)
    R369_2_M_차종_유 : BOOL; (* AT %MW4502.4 *)
    S362_M_총괄_이상 : BOOL; (* AT %MW1009.0 *) (* S362_M_총괄_이상 *)
    S367_M_공정_차종_무 : BOOL; (* AT %MW3502.1 *) (* S367_M_공정_차종_무 *)
    S367_M_공정_차종_유 : BOOL; (* AT %MW3502.0 *) (* S367_M_공정_차종_유 *)
    S368_M_수동모드 : BOOL; (* AT %MW4000.3 *) (* S368 선택 수동모드 *)
    S368_M_작업완료_SET_PLS : BOOL; (* AT %MW4000.8 *) (* S368 M 작업완료 SET PLS *)
    S368_M_작업완료_리셋_PLS : BOOL; (* AT %MW4000.9 *) (* S368 M 작업완료 리셋 PLS *)
    S369_1_M_BYPASS_보조 : BOOL; (* AT %MW4503.15 *) (* S369 1 M BYPASS 보조 *)
    S369_1_M_R369_1_안착완료 : BOOL; (* AT %MW4501.1 *)
    S369_1_M_R369_2_ROOF_취출가능 : BOOL; (* AT %MW4504.9 *)
    S369_1_M_R369_2_언로딩완료 : BOOL; (* AT %MW4501.2 *)
    S369_1_M_ROOF_안착가능 : BOOL; (* AT %MW4504.8 *)
    S369_1_M_ROOF_제품감지_무 : BOOL; (* AT %MW4501.6 *)
    S369_1_M_ROOF_제품감지_유 : BOOL; (* AT %MW4501.5 *)
    S369_1_M_SEQ : WORD; (* AT %MW10220 *) (* S369 1 M SEQ *)
    S369_1_M_공정_불간섭 : BOOL; (* AT %MW4504.1 *) (* S369_1_M_공정_불간섭 *)
    S369_1_M_공정_원위치 : BOOL; (* AT %MW4504.0 *) (* S369_1_M_공정_원위치 *)
    S369_1_M_공정_제품감지_무 : BOOL; (* AT %MW4501.4 *) (* S369_1_M_공정_제품감지_무 *)
    S369_1_M_공정_제품감지_유 : BOOL; (* AT %MW4501.3 *) (* S369_1_M_공정_제품감지_유 *)
    S369_1_M_공정_차종_무 : BOOL; (* AT %MW4502.1 *) (* S369_1_M_공정_차종_무 *)
    S369_1_M_공정_차종_유 : BOOL; (* AT %MW4502.0 *) (* S369_1_M_공정_차종_유 *)
    S369_1_M_수동모드 : BOOL; (* AT %MW4500.3 *) (* S369-1 선택 수동모드 *)
    S369_1_M_썬루프_제품감지_무 : BOOL; (* AT %MW4501.8 *)
    S369_1_M_썬루프_제품감지_유 : BOOL; (* AT %MW4501.7 *)
    S369_1_M_운전준비_ON : BOOL; (* AT %MW4500.0 *) (* S369-1 운전준비 ON *)
    S369_1_M_자동_START : BOOL; (* AT %MW4500.5 *) (* S369-1 자동운전중 *)
    S369_1_M_자동_운전중 : BOOL; (* AT %MW4500.4 *) (* S369-1 자동운전중 *)
    S369_1_M_자동모드 : BOOL; (* AT %MW4500.1 *) (* S369-1 선택 자동모드 *)
    S369_1_M_작업_완료 : BOOL; (* AT %MW4501.0 *) (* S369_1_M_작업_완료 *)
    S369_1_M_작업완료_SET_PLS : BOOL; (* AT %MW4500.8 *) (* S369 1 M 작업완료 SET PLS *)
    S369_1_M_작업완료_리셋_PLS : BOOL; (* AT %MW4500.9 *) (* S369 1 M 작업완료 리셋 PLS *)
    S369_1_M_차종1_AX : BOOL; (* AT %MW10221.0 *) (* S369 1 M 차종1 AX *)
    S369_1_M_차종1_B : BOOL; (* AT %MW10221.1 *) (* S369 1 M 차종1 B *)
    S369_1_M_차종1_C : BOOL; (* AT %MW10221.2 *) (* S369 1 M 차종1 C *)
    S369_1_M_차종1_D : BOOL; (* AT %MW10221.3 *) (* S369 1 M 차종1 D *)
    S369_1_M_차종1_E : BOOL; (* AT %MW10221.4 *) (* S369 1 M 차종1 E *)
    S369_1_M_차종1_F : BOOL; (* AT %MW10221.5 *) (* S369 1 M 차종1 F *)
    S369_1_M_차종1_G : BOOL; (* AT %MW10221.6 *) (* S369 1 M 차종1 G *)
    S369_1_M_차종1_H : BOOL; (* AT %MW10221.7 *) (* S369 1 M 차종1 H *)
    S369_1_M_차종2_3DR : BOOL; (* AT %MW10221.8 *) (* S369 1 M 차종2 3DR *)
    S369_1_M_차종2_4DR : BOOL; (* AT %MW10221.9 *) (* S369 1 M 차종2 4DR *)
    S369_1_M_차종2_5DR : BOOL; (* AT %MW10221.10 *) (* S369 1 M 차종2 5DR *)
    S369_1_M_차종2_SP1 : BOOL; (* AT %MW10221.12 *) (* S369 1 M 차종2 SP1 *)
    S369_1_M_차종2_SP2 : BOOL; (* AT %MW10221.13 *) (* S369 1 M 차종2 SP2 *)
    S369_1_M_차종2_WGN : BOOL; (* AT %MW10221.11 *) (* S369 1 M 차종2 WGN *)
    S369_1_M_차종3_LHD : BOOL; (* AT %MW10221.14 *) (* S369 1 M 차종3 LHD *)
    S369_1_M_차종3_RHD : BOOL; (* AT %MW10221.15 *) (* S369 1 M 차종3 RHD *)
    S369_1_M_차종4_EEC : BOOL; (* AT %MW10222.3 *) (* S369 1 M 차종4 EEC *)
    S369_1_M_차종4_SP1 : BOOL; (* AT %MW10222.8 *) (* S369 1 M 차종4 SP1 *)
    S369_1_M_차종4_SP2 : BOOL; (* AT %MW10222.9 *) (* S369 1 M 차종4 SP2 *)
    S369_1_M_차종4_SP3 : BOOL; (* AT %MW10222.11 *) (* S369 1 M 차종4 SP3 *)
    S369_1_M_차종4_SP4 : BOOL; (* AT %MW10222.12 *) (* S369 1 M 차종4 SP4 *)
    S369_1_M_차종4_SP5 : BOOL; (* AT %MW10222.13 *) (* S369 1 M 차종4 SP5 *)
    S369_1_M_차종4_SP6 : BOOL; (* AT %MW10222.14 *) (* S369 1 M 차종4 SP6 *)
    S369_1_M_차종4_SP7 : BOOL; (* AT %MW10222.15 *) (* S369 1 M 차종4 SP7 *)
    S369_1_M_차종4_내수 : BOOL; (* AT %MW10222.0 *) (* S369 1 M 차종4 내수 *)
    S369_1_M_차종4_러시아 : BOOL; (* AT %MW10222.10 *) (* S369 1 M 차종4 러시아 *)
    S369_1_M_차종4_북미 : BOOL; (* AT %MW10222.2 *) (* S369 1 M 차종4 북미 *)
    S369_1_M_차종4_브라질 : BOOL; (* AT %MW10222.7 *) (* S369 1 M 차종4 브라질 *)
    S369_1_M_차종4_수출 : BOOL; (* AT %MW10222.1 *) (* S369 1 M 차종4 수출 *)
    S369_1_M_차종4_중국 : BOOL; (* AT %MW10222.6 *) (* S369 1 M 차종4 중국 *)
    S369_1_M_차종4_중동 : BOOL; (* AT %MW10222.5 *) (* S369 1 M 차종4 중동 *)
    S369_1_M_차종4_호주 : BOOL; (* AT %MW10222.4 *) (* S369 1 M 차종4 호주 *)
    S369_1_M_차종5_AT : BOOL; (* AT %MW10223.1 *) (* S369 1 M 차종5 AT *)
    S369_1_M_차종5_MT : BOOL; (* AT %MW10223.0 *) (* S369 1 M 차종5 MT *)
    S369_1_M_차종5_SP1 : BOOL; (* AT %MW10223.2 *) (* S369 1 M 차종5 SP1 *)
    S369_1_M_차종6_DSROOF : BOOL; (* AT %MW10223.6 *) (* S369 1 M 차종6 DSROOF *)
    S369_1_M_차종6_SP1 : BOOL; (* AT %MW10223.7 *) (* S369 1 M 차종6 SP1 *)
    S369_1_M_차종6_썬루프 : BOOL; (* AT %MW10223.4 *) (* S369 1 M 차종6 썬루프 *)
    S369_1_M_차종6_일반루프 : BOOL; (* AT %MW10223.3 *) (* S369 1 M 차종6 일반루프 *)
    S369_1_M_차종6_파노라마루프 : BOOL; (* AT %MW10223.5 *) (* S369 1 M 차종6 파노라마루프 *)
    S369_1_M_차종7_DSL : BOOL; (* AT %MW10223.9 *) (* S369 1 M 차종7 DSL *)
    S369_1_M_차종7_GSL : BOOL; (* AT %MW10223.8 *) (* S369 1 M 차종7 GSL *)
    S369_1_M_차종7_SP1 : BOOL; (* AT %MW10223.10 *) (* S369 1 M 차종7 SP1 *)
    S369_1_M_차종7_SP2 : BOOL; (* AT %MW10223.11 *) (* S369 1 M 차종7 SP2 *)
    S369_1_M_차종7_SP3 : BOOL; (* AT %MW10223.12 *) (* S369 1 M 차종7 SP3 *)
    S369_1_M_차종7_SP4 : BOOL; (* AT %MW10223.13 *) (* S369 1 M 차종7 SP4 *)
    S369_1_M_차종7_SP5 : BOOL; (* AT %MW10223.14 *) (* S369 1 M 차종7 SP5 *)
    S369_1_M_차종7_SP6 : BOOL; (* AT %MW10223.15 *) (* S369 1 M 차종7 SP6 *)
    S369_1_M_차종8_2WD : BOOL; (* AT %MW10224.0 *) (* S369 1 M 차종8 2WD *)
    S369_1_M_차종8_4WD : BOOL; (* AT %MW10224.1 *) (* S369 1 M 차종8 4WD *)
    S369_1_M_차종8_SP1 : BOOL; (* AT %MW10224.2 *) (* S369 1 M 차종8 SP1 *)
    S369_1_M_차종9_MPI : BOOL; (* AT %MW10224.3 *) (* S369 1 M 차종9 MPI *)
    S369_1_M_차종9_SP1 : BOOL; (* AT %MW10224.5 *) (* S369 1 M 차종9 SP1 *)
    S369_1_M_차종9_SP10 : BOOL; (* AT %MW10224.14 *) (* S369 1 M 차종9 SP10 *)
    S369_1_M_차종9_SP11 : BOOL; (* AT %MW10224.15 *) (* S369 1 M 차종9 SP11 *)
    S369_1_M_차종9_SP2 : BOOL; (* AT %MW10224.6 *) (* S369 1 M 차종9 SP2 *)
    S369_1_M_차종9_SP3 : BOOL; (* AT %MW10224.7 *) (* S369 1 M 차종9 SP3 *)
    S369_1_M_차종9_SP4 : BOOL; (* AT %MW10224.8 *) (* S369 1 M 차종9 SP4 *)
    S369_1_M_차종9_SP5 : BOOL; (* AT %MW10224.9 *) (* S369 1 M 차종9 SP5 *)
    S369_1_M_차종9_SP6 : BOOL; (* AT %MW10224.10 *) (* S369 1 M 차종9 SP6 *)
    S369_1_M_차종9_SP7 : BOOL; (* AT %MW10224.11 *) (* S369 1 M 차종9 SP7 *)
    S369_1_M_차종9_SP8 : BOOL; (* AT %MW10224.12 *) (* S369 1 M 차종9 SP8 *)
    S369_1_M_차종9_SP9 : BOOL; (* AT %MW10224.13 *) (* S369 1 M 차종9 SP9 *)
    S369_1_M_차종9_T_GDI : BOOL; (* AT %MW10224.4 *) (* S369 1 M 차종9 T GDI *)
    S369_1_M_차종_OPT1_R_RACK_무 : BOOL; (* AT %MW10225.3 *) (* S369 1 M 차종 OPT1 R RACK 무 *)
    S369_1_M_차종_OPT1_R_RACK_유 : BOOL; (* AT %MW10225.2 *) (* S369 1 M 차종 OPT1 R RACK 유 *)
    S369_1_M_차종_OPT1_S_REP_EATER_무 : BOOL; (* AT %MW10225.7 *) (* S369 1 M 차종 OPT1 S REP EATER 무 *)
    S369_1_M_차종_OPT1_S_REP_EATER_유 : BOOL; (* AT %MW10225.6 *) (* S369 1 M 차종 OPT1 S REP EATER 유 *)
    S369_1_M_차종_OPT1_VAN_무 : BOOL; (* AT %MW10225.9 *) (* S369 1 M 차종 OPT1 VAN 무 *)
    S369_1_M_차종_OPT1_VAN_유 : BOOL; (* AT %MW10225.8 *) (* S369 1 M 차종 OPT1 VAN 유 *)
    S369_1_M_차종_OPT1_슬라이딩_무 : BOOL; (* AT %MW10225.1 *) (* S369 1 M 차종 OPT1 슬라이딩 무 *)
    S369_1_M_차종_OPT1_슬라이딩_유 : BOOL; (* AT %MW10225.0 *) (* S369 1 M 차종 OPT1 슬라이딩 유 *)
    S369_1_M_차종_OPT1_폴딩_무 : BOOL; (* AT %MW10225.5 *) (* S369 1 M 차종 OPT1 폴딩 무 *)
    S369_1_M_차종_OPT1_폴딩_유 : BOOL; (* AT %MW10225.4 *) (* S369 1 M 차종 OPT1 폴딩 유 *)
    S369_1_M_차종_공대차 : BOOL; (* AT %MW10230.12 *) (* S369 1 M 차종 공대차 *)
    S369_1_M_차종_공차 : BOOL; (* AT %MW10230.10 *) (* S369 1 M 차종 공차 *)
    S369_1_M_차종_불량차 : BOOL; (* AT %MW10230.11 *) (* S369 1 M 차종 불량차 *)
    S369_1_M_총괄_이상 : BOOL; (* AT %MW4509.0 *) (* S369_1_M_총괄_이상 *)
    전체_M_GATE_자동기동 : BOOL; (* AT %MW308.1 *) (* 전체_M_자동_운전 *)
    전체_라인_M_총괄_SAFETY_이상 : BOOL; (* AT %MW300.2 *) (* ALL공정 SAFETY  이상총괄 *)
    전체_라인_M_총괄_공기압_이상 : BOOL; (* AT %MW300.3 *) (* ALL공정 공기압 이상총괄 *)
    전체_라인_M_총괄_비상정지_이상 : BOOL; (* AT %MW300.1 *) (* ALL공정 비상정지 이상총괄 *)
    전체_라인_M_총괄_이상 : BOOL; (* AT %MW300.0 *) (* ALL공정 총괄이상 *)
END_VAR
VAR_EXTERNAL
    HOP_PBL_369_자동_운전 : BOOL; (* AT %MW87500.10 *) (* HOP_PBL_369_자동_운전 *)
    HOP_PBL_운전준비_ON : BOOL; (* AT %MW87500.0 *) (* HOP_PBL_운전준비_ON *)
    HOP_SSP_369_수동_선택 : BOOL; (* AT %MW87500.9 *) (* HOP_SSP_369_수동_선택 *)
    HOP_SSP_369_자동_선택 : BOOL; (* AT %MW87500.8 *) (* HOP_SSP_369_자동_선택 *)
    MCP_PBL_369_자동_운전 : BOOL; (* AT %MW87630.10 *) (* MCP PBL 369~-1 자동기동 *)
    MCP_PBL_운전준비_ON : BOOL; (* AT %MW87630.0 *) (* MCP_PBL_운전준비_ON *)
    MCP_SPB_작업완료_RESET : BOOL; (* AT %MW87631.6 *) (* MCP_SPB_작업완료_RESET *)
    MCP_SPB_작업완료_SET : BOOL; (* AT %MW87631.7 *) (* MCP_SPB_작업완료_SET *)
    MCP_SSP_369_수동_선택 : BOOL; (* AT %MW87630.8 *) (* MCP_SSP_369_수동_선택 *)
    MCP_SSP_369_자동_선택 : BOOL; (* AT %MW87630.9 *) (* MCP_SSP_369_자동_선택 *)
    R368_1_M_I_RB_간섭무_1 : BOOL; (* AT %MW20072.0 *) (* R368_1_M_I_RB_간섭무_1 *)
    R368_1_M_I_RB_원위치 : BOOL; (* AT %MW20070.3 *) (* R368_1_M_I_RB_원위치 *)
    R369_1_M_I_RB_4차_작업완료 : BOOL; (* AT %MW20081.5 *) (* R369_1_M_I_RB_4차_작업완료 *)
    R369_1_M_I_RB_간섭무_1 : BOOL; (* AT %MW20082.0 *) (* R369_1_M_I_RB_간섭무_1 *)
    R369_1_M_I_RB_원위치 : BOOL; (* AT %MW20080.3 *) (* R369_1_M_I_RB_원위치 *)
    R369_2_M_I_RB_1차_작업완료 : BOOL; (* AT %MW20091.2 *) (* R369_2_M_I_RB_1차_작업완료 *)
    R369_2_M_I_RB_간섭무_1 : BOOL; (* AT %MW20092.0 *) (* R369_2_M_I_RB_간섭무_1 *)
    R369_2_M_I_RB_원위치 : BOOL; (* AT %MW20090.3 *) (* R369_2_M_I_RB_원위치 *)
    S369_1_PHS_ROOF_PNL_썬루프_감지 : BOOL; (* AT %MW86400.3 *)
    S369_1_PRS_ROOF_PNL_제품감지1 : BOOL; (* AT %MW86400.0 *)
    S369_1_PRS_ROOF_PNL_제품감지2 : BOOL; (* AT %MW86400.1 *)
    S369_1_PRS_ROOF_PNL_제품감지3 : BOOL; (* AT %MW86400.2 *)
END_VAR
VAR
    S369_1_READY : TON;
    T369_1_AUTO : TON;
END_VAR
VAR
    _t1 : BOOL;
    _t2 : BOOL;
    _t3 : BOOL;
END_VAR

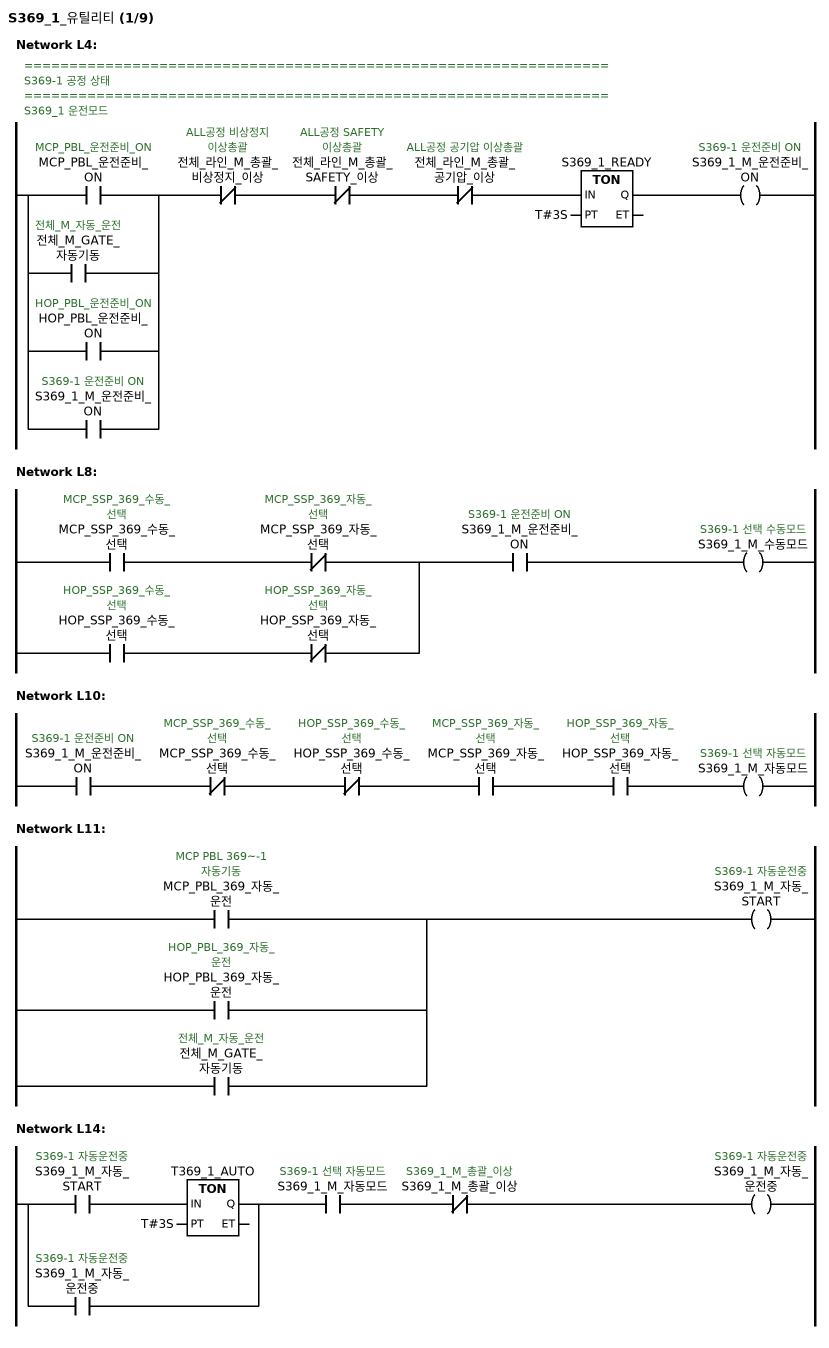
(* ================================================================= *)
(* S369-1 공정 상태 *)
(* ================================================================= *)
(* S369_1 운전모드 *)
(* Rung L4 *)
S369_1_READY(IN := (MCP_PBL_운전준비_ON OR 전체_M_GATE_자동기동 OR HOP_PBL_운전준비_ON OR S369_1_M_운전준비_ON) AND NOT 전체_라인_M_총괄_비상정지_이상 AND NOT 전체_라인_M_총괄_SAFETY_이상 AND NOT 전체_라인_M_총괄_공기압_이상, PT := T#3S);
S369_1_M_운전준비_ON := S369_1_READY.Q;
(* Rung L8 *)
S369_1_M_수동모드 := ((MCP_SSP_369_수동_선택 AND NOT MCP_SSP_369_자동_선택) OR (HOP_SSP_369_수동_선택 AND NOT HOP_SSP_369_자동_선택)) AND S369_1_M_운전준비_ON;
(* Rung L10 *)
S369_1_M_자동모드 := S369_1_M_운전준비_ON AND NOT MCP_SSP_369_수동_선택 AND NOT HOP_SSP_369_수동_선택 AND MCP_SSP_369_자동_선택 AND HOP_SSP_369_자동_선택;
(* Rung L11 *)
S369_1_M_자동_START := MCP_PBL_369_자동_운전 OR HOP_PBL_369_자동_운전 OR 전체_M_GATE_자동기동;
(* Rung L14 *)
T369_1_AUTO(IN := S369_1_M_자동_START, PT := T#3S);
S369_1_M_자동_운전중 := (T369_1_AUTO.Q OR S369_1_M_자동_운전중) AND S369_1_M_자동모드 AND NOT S369_1_M_총괄_이상;

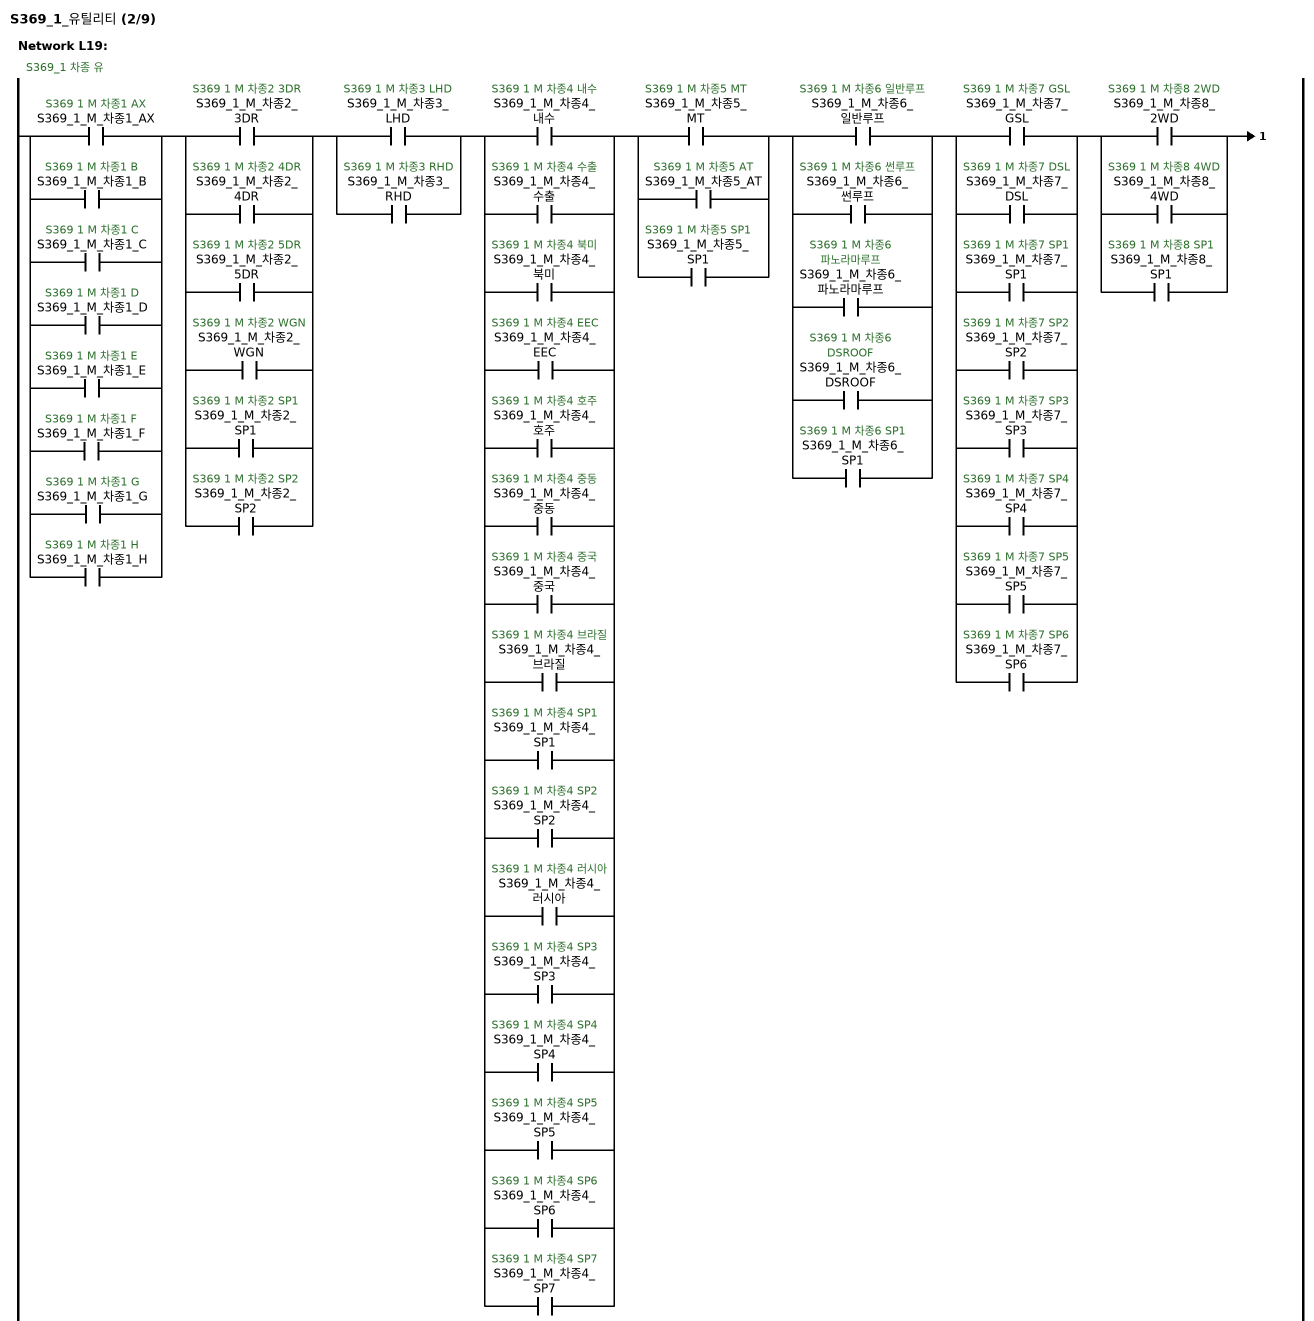

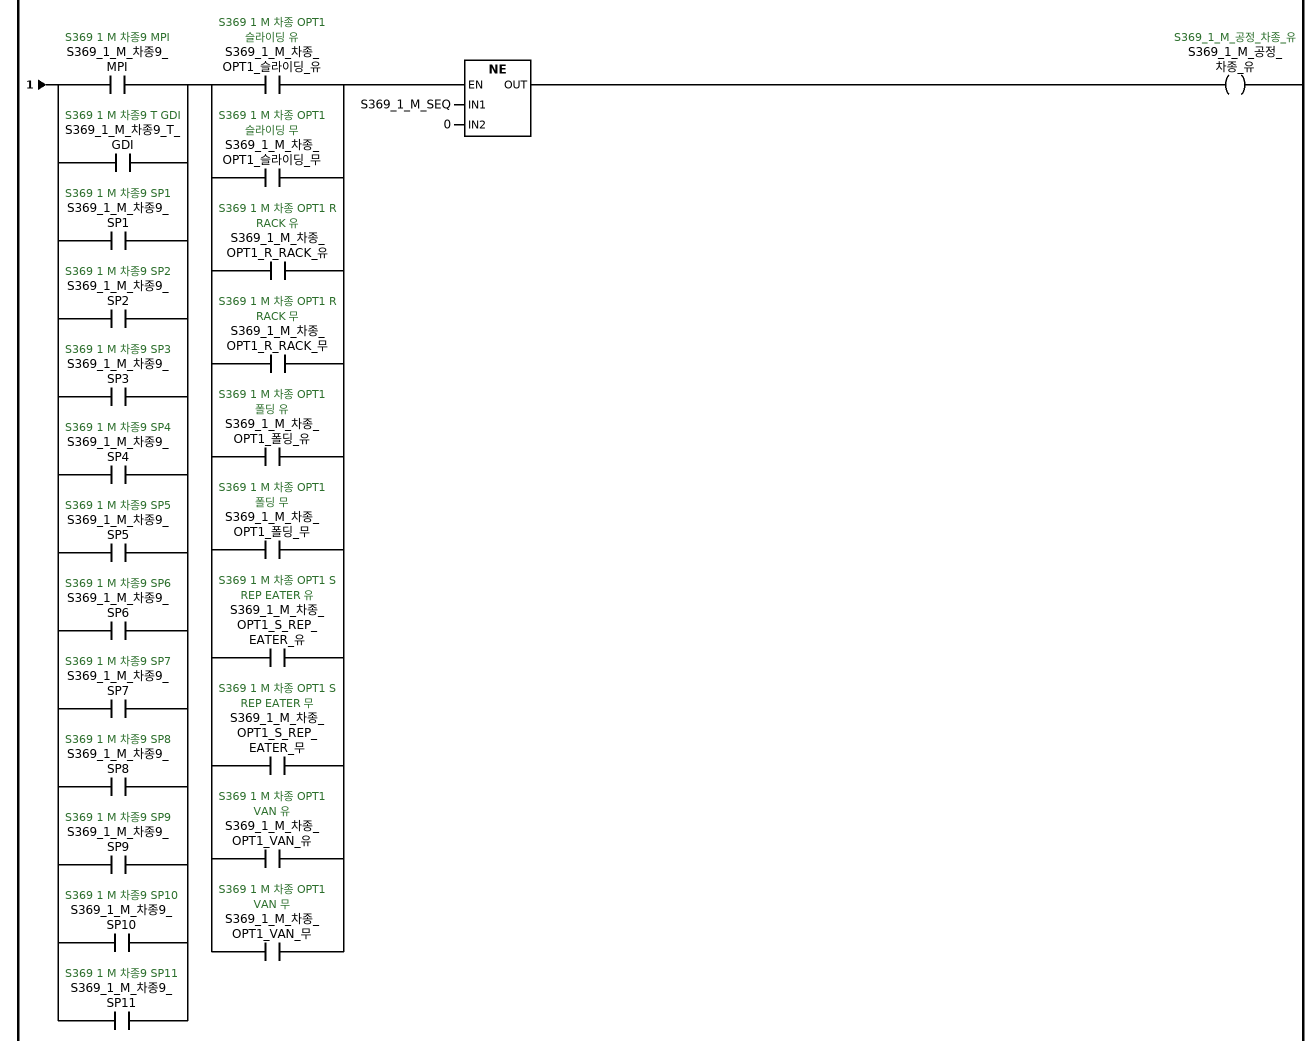
(* S369_1 차종 유 *)
(* Rung L19 *)
IF (S369_1_M_차종1_AX OR S369_1_M_차종1_B OR S369_1_M_차종1_C OR S369_1_M_차종1_D OR S369_1_M_차종1_E OR S369_1_M_차종1_F OR S369_1_M_차종1_G OR S369_1_M_차종1_H) AND (S369_1_M_차종2_3DR OR S369_1_M_차종2_4DR OR S369_1_M_차종2_5DR OR S369_1_M_차종2_WGN OR S369_1_M_차종2_SP1 OR S369_1_M_차종2_SP2) AND (S369_1_M_차종3_LHD OR S369_1_M_차종3_RHD) AND (S369_1_M_차종4_내수 OR S369_1_M_차종4_수출 OR S369_1_M_차종4_북미 OR S369_1_M_차종4_EEC OR S369_1_M_차종4_호주 OR S369_1_M_차종4_중동 OR S369_1_M_차종4_중국 OR S369_1_M_차종4_브라질 OR S369_1_M_차종4_SP1 OR S369_1_M_차종4_SP2 OR S369_1_M_차종4_러시아 OR S369_1_M_차종4_SP3 OR S369_1_M_차종4_SP4 OR S369_1_M_차종4_SP5 OR S369_1_M_차종4_SP6 OR S369_1_M_차종4_SP7) AND (S369_1_M_차종5_MT OR S369_1_M_차종5_AT OR S369_1_M_차종5_SP1) AND (S369_1_M_차종6_일반루프 OR S369_1_M_차종6_썬루프 OR S369_1_M_차종6_파노라마루프 OR S369_1_M_차종6_DSROOF OR S369_1_M_차종6_SP1) AND (S369_1_M_차종7_GSL OR S369_1_M_차종7_DSL OR S369_1_M_차종7_SP1 OR S369_1_M_차종7_SP2 OR S369_1_M_차종7_SP3 OR S369_1_M_차종7_SP4 OR S369_1_M_차종7_SP5 OR S369_1_M_차종7_SP6) AND (S369_1_M_차종8_2WD OR S369_1_M_차종8_4WD OR S369_1_M_차종8_SP1) AND (S369_1_M_차종9_MPI OR S369_1_M_차종9_T_GDI OR S369_1_M_차종9_SP1 OR S369_1_M_차종9_SP2 OR S369_1_M_차종9_SP3 OR S369_1_M_차종9_SP4 OR S369_1_M_차종9_SP5 OR S369_1_M_차종9_SP6 OR S369_1_M_차종9_SP7 OR S369_1_M_차종9_SP8 OR S369_1_M_차종9_SP9 OR S369_1_M_차종9_SP10 OR S369_1_M_차종9_SP11) AND (S369_1_M_차종_OPT1_슬라이딩_유 OR S369_1_M_차종_OPT1_슬라이딩_무 OR S369_1_M_차종_OPT1_R_RACK_유 OR S369_1_M_차종_OPT1_R_RACK_무 OR S369_1_M_차종_OPT1_폴딩_유 OR S369_1_M_차종_OPT1_폴딩_무 OR S369_1_M_차종_OPT1_S_REP_EATER_유 OR S369_1_M_차종_OPT1_S_REP_EATER_무 OR S369_1_M_차종_OPT1_VAN_유 OR S369_1_M_차종_OPT1_VAN_무) THEN
    _t1 := S369_1_M_SEQ <> 0;
END_IF;
S369_1_M_공정_차종_유 := _t1;

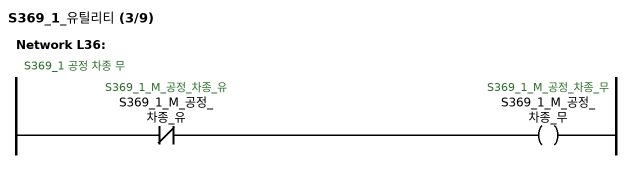
(* S369_1 공정 차종 무 *)
(* Rung L36 *)
S369_1_M_공정_차종_무 := NOT S369_1_M_공정_차종_유;

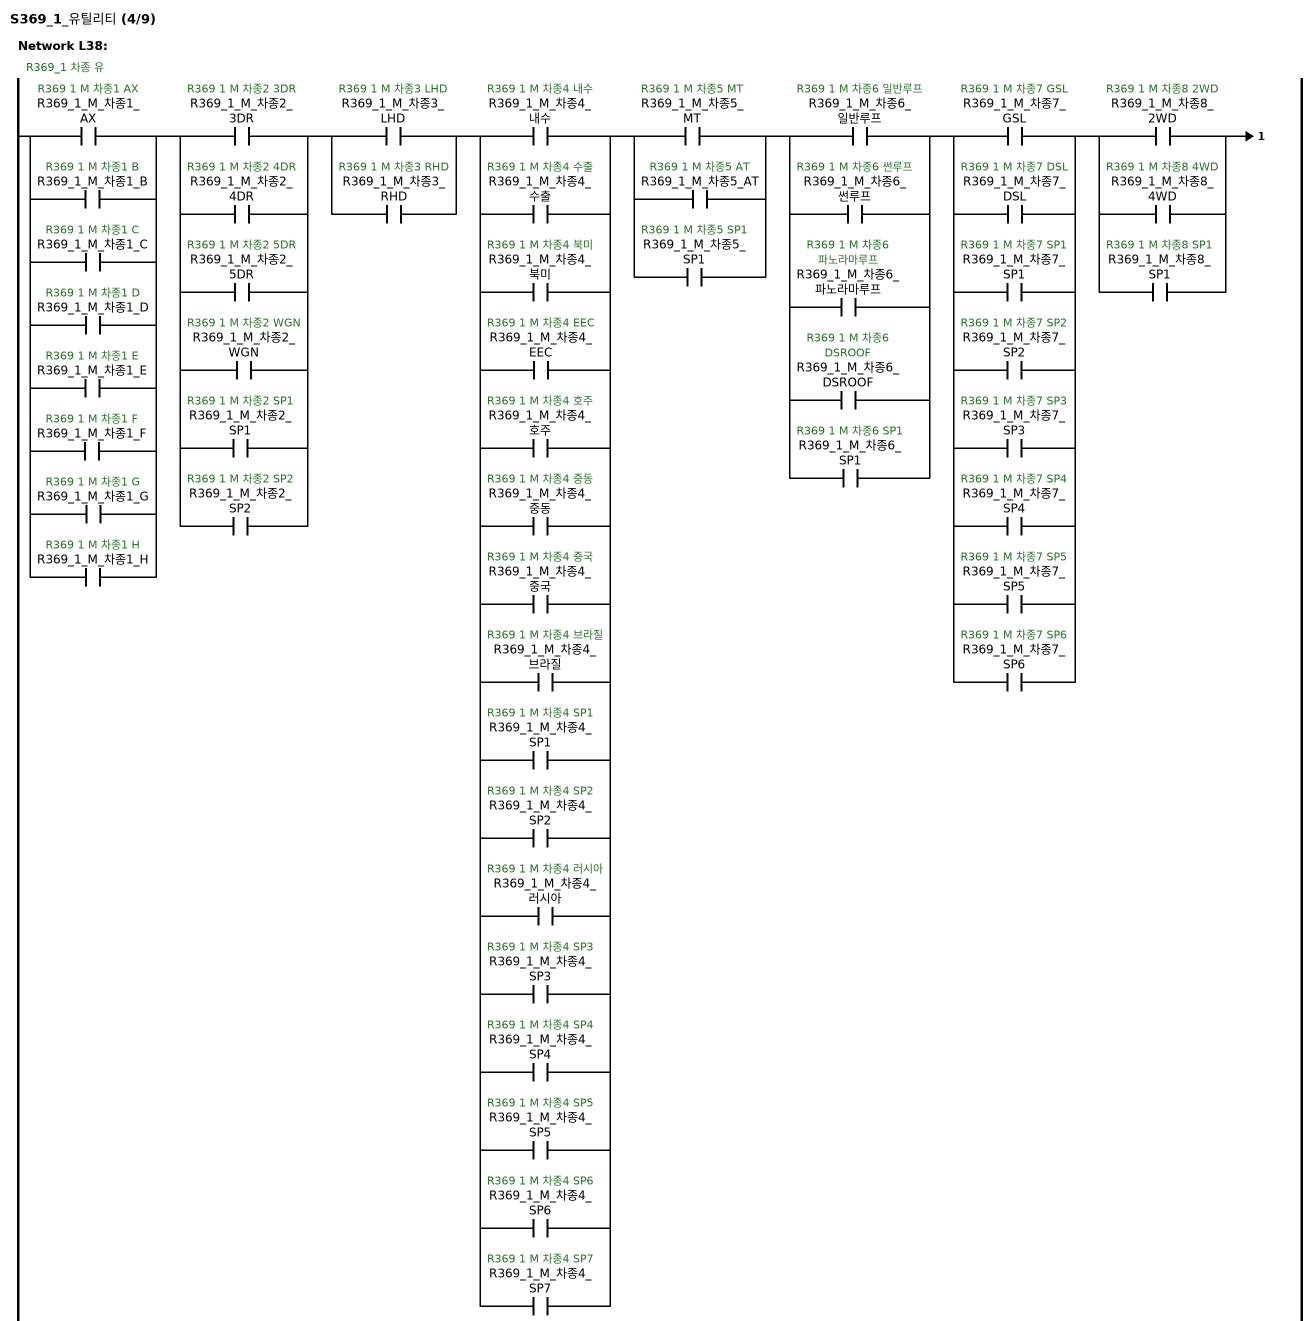

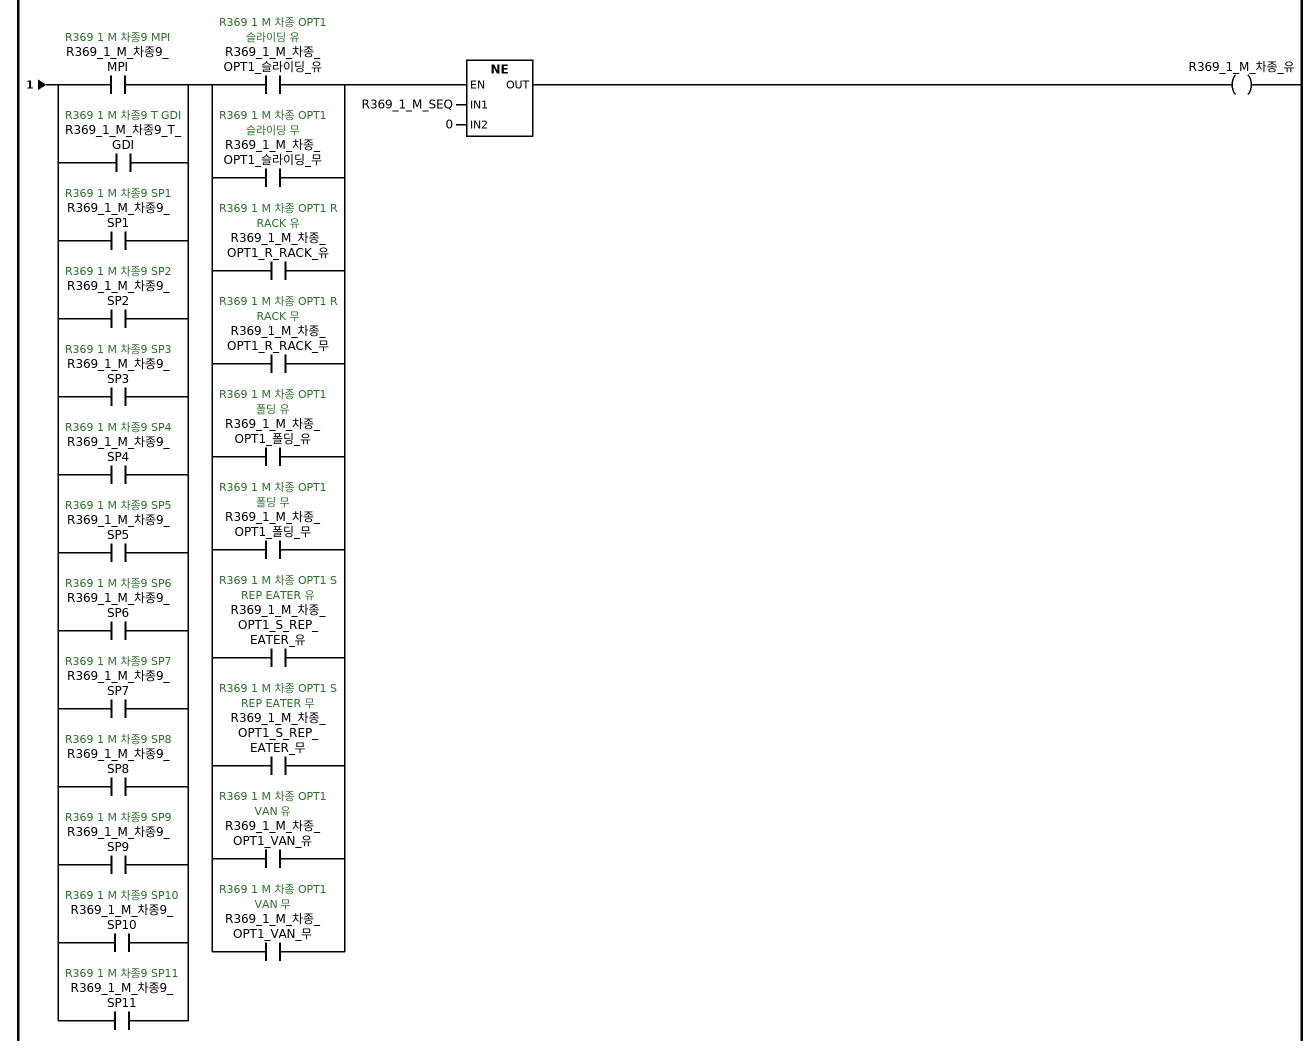
(* R369_1 차종 유 *)
(* Rung L38 *)
IF (R369_1_M_차종1_AX OR R369_1_M_차종1_B OR R369_1_M_차종1_C OR R369_1_M_차종1_D OR R369_1_M_차종1_E OR R369_1_M_차종1_F OR R369_1_M_차종1_G OR R369_1_M_차종1_H) AND (R369_1_M_차종2_3DR OR R369_1_M_차종2_4DR OR R369_1_M_차종2_5DR OR R369_1_M_차종2_WGN OR R369_1_M_차종2_SP1 OR R369_1_M_차종2_SP2) AND (R369_1_M_차종3_LHD OR R369_1_M_차종3_RHD) AND (R369_1_M_차종4_내수 OR R369_1_M_차종4_수출 OR R369_1_M_차종4_북미 OR R369_1_M_차종4_EEC OR R369_1_M_차종4_호주 OR R369_1_M_차종4_중동 OR R369_1_M_차종4_중국 OR R369_1_M_차종4_브라질 OR R369_1_M_차종4_SP1 OR R369_1_M_차종4_SP2 OR R369_1_M_차종4_러시아 OR R369_1_M_차종4_SP3 OR R369_1_M_차종4_SP4 OR R369_1_M_차종4_SP5 OR R369_1_M_차종4_SP6 OR R369_1_M_차종4_SP7) AND (R369_1_M_차종5_MT OR R369_1_M_차종5_AT OR R369_1_M_차종5_SP1) AND (R369_1_M_차종6_일반루프 OR R369_1_M_차종6_썬루프 OR R369_1_M_차종6_파노라마루프 OR R369_1_M_차종6_DSROOF OR R369_1_M_차종6_SP1) AND (R369_1_M_차종7_GSL OR R369_1_M_차종7_DSL OR R369_1_M_차종7_SP1 OR R369_1_M_차종7_SP2 OR R369_1_M_차종7_SP3 OR R369_1_M_차종7_SP4 OR R369_1_M_차종7_SP5 OR R369_1_M_차종7_SP6) AND (R369_1_M_차종8_2WD OR R369_1_M_차종8_4WD OR R369_1_M_차종8_SP1) AND (R369_1_M_차종9_MPI OR R369_1_M_차종9_T_GDI OR R369_1_M_차종9_SP1 OR R369_1_M_차종9_SP2 OR R369_1_M_차종9_SP3 OR R369_1_M_차종9_SP4 OR R369_1_M_차종9_SP5 OR R369_1_M_차종9_SP6 OR R369_1_M_차종9_SP7 OR R369_1_M_차종9_SP8 OR R369_1_M_차종9_SP9 OR R369_1_M_차종9_SP10 OR R369_1_M_차종9_SP11) AND (R369_1_M_차종_OPT1_슬라이딩_유 OR R369_1_M_차종_OPT1_슬라이딩_무 OR R369_1_M_차종_OPT1_R_RACK_유 OR R369_1_M_차종_OPT1_R_RACK_무 OR R369_1_M_차종_OPT1_폴딩_유 OR R369_1_M_차종_OPT1_폴딩_무 OR R369_1_M_차종_OPT1_S_REP_EATER_유 OR R369_1_M_차종_OPT1_S_REP_EATER_무 OR R369_1_M_차종_OPT1_VAN_유 OR R369_1_M_차종_OPT1_VAN_무) THEN
    _t2 := R369_1_M_SEQ <> 0;
END_IF;
R369_1_M_차종_유 := _t2;

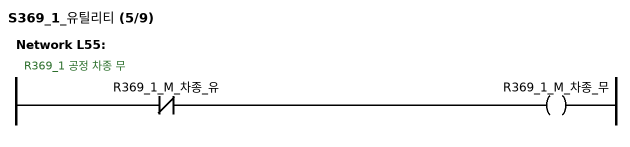
(* R369_1 공정 차종 무 *)
(* Rung L55 *)
R369_1_M_차종_무 := NOT R369_1_M_차종_유;

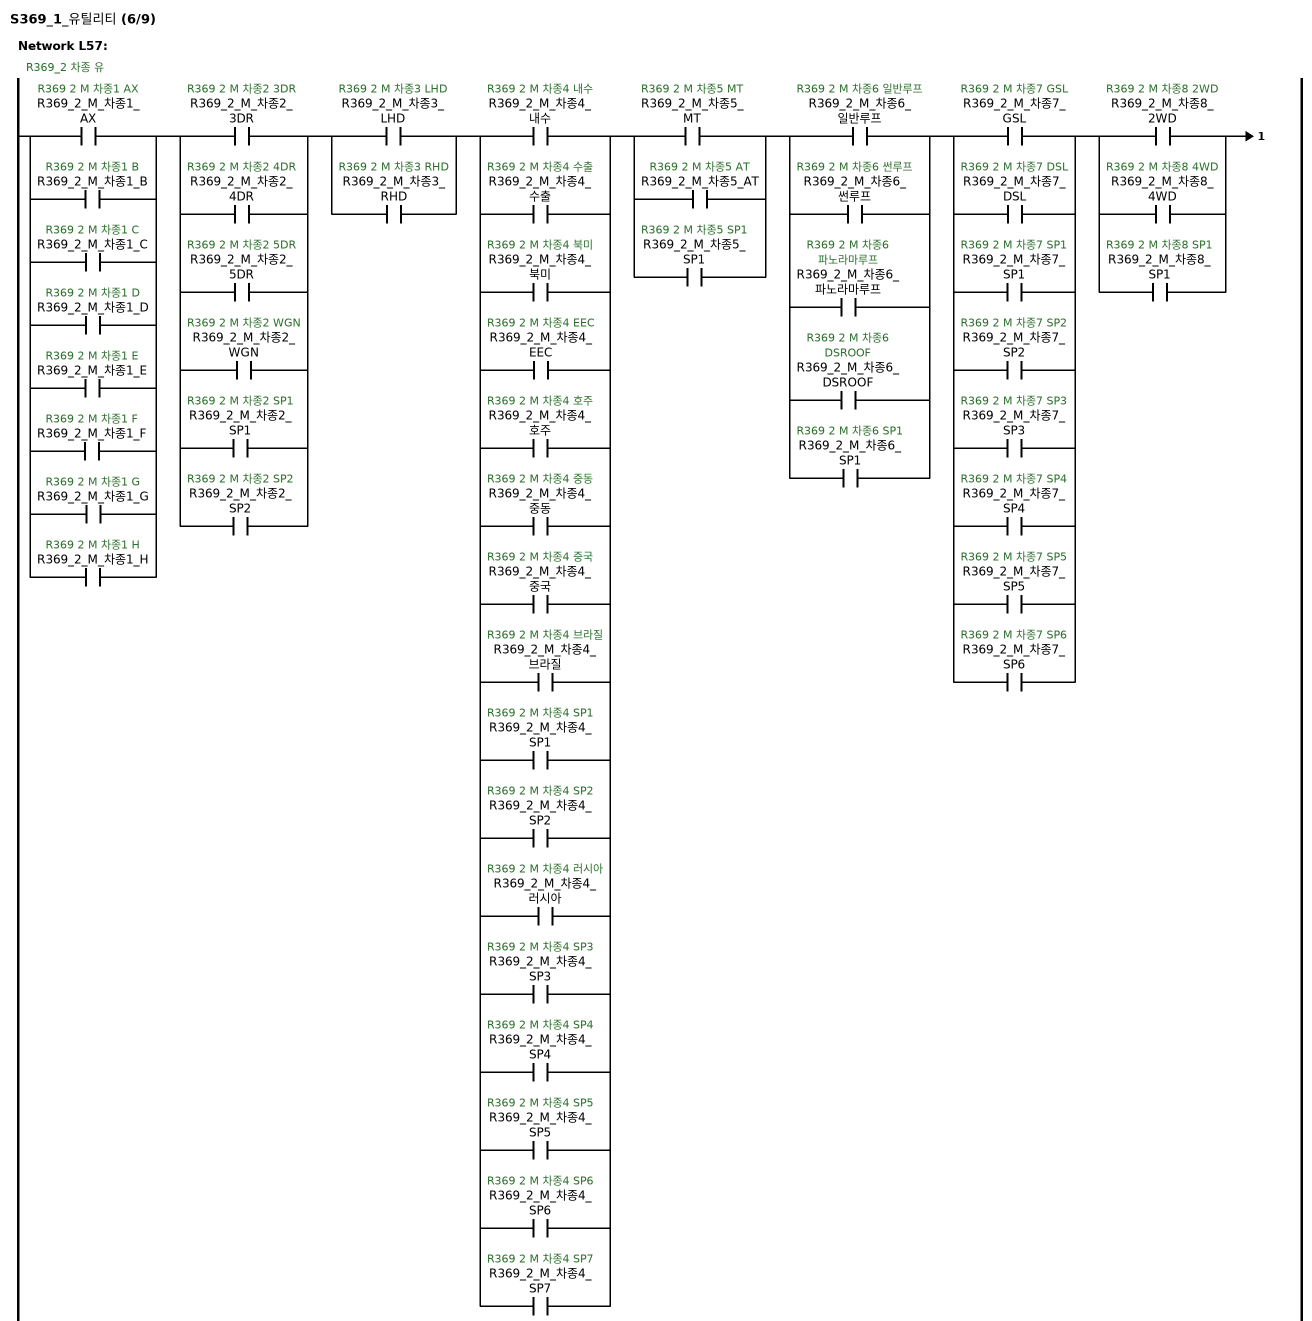

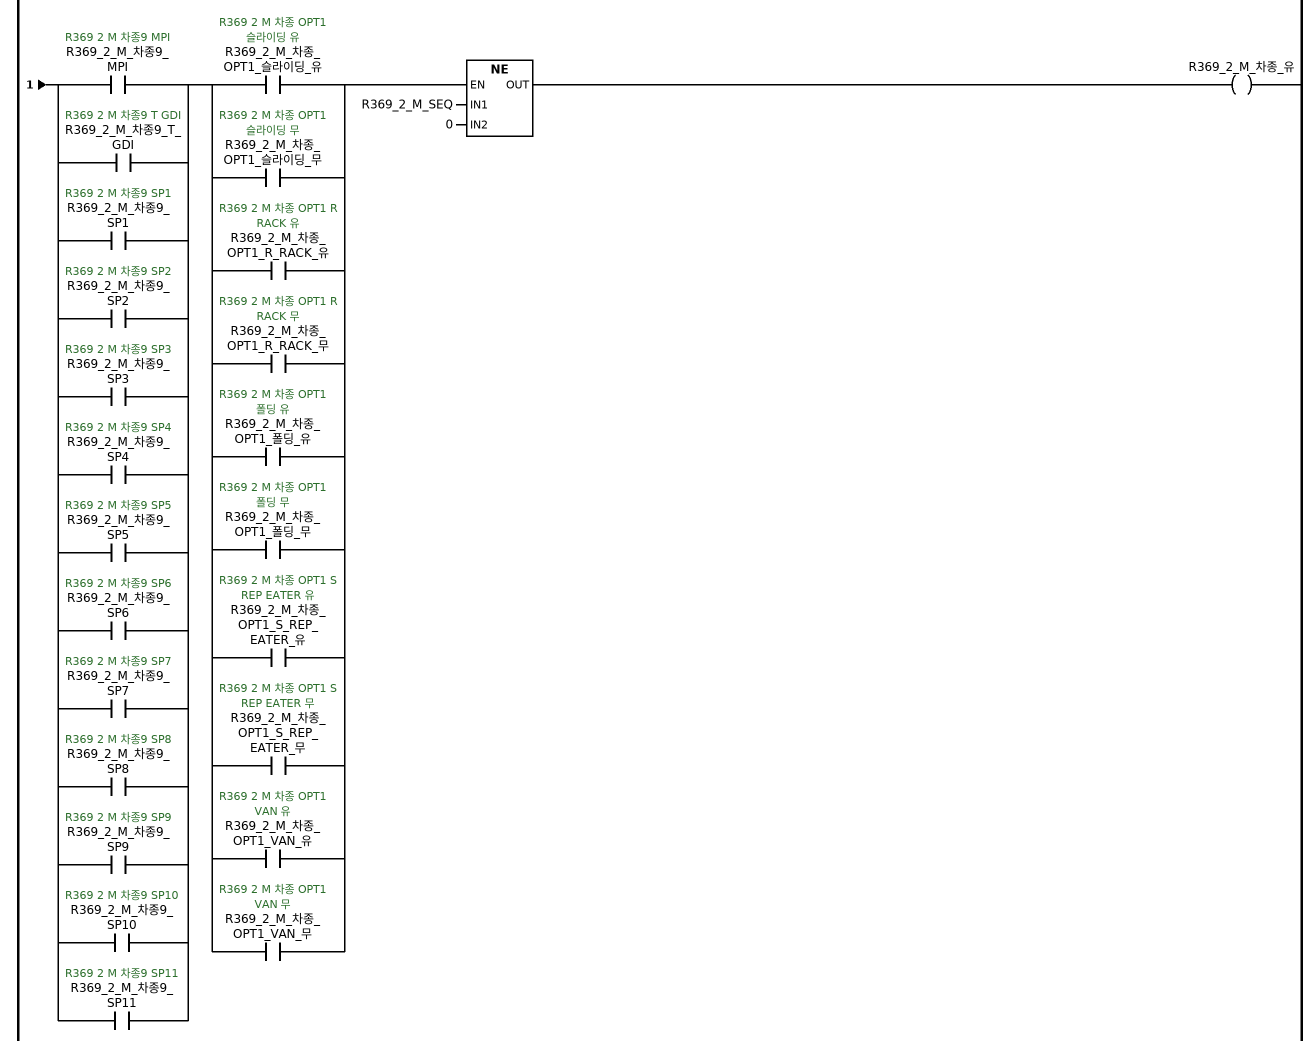
(* R369_2 차종 유 *)
(* Rung L57 *)
IF (R369_2_M_차종1_AX OR R369_2_M_차종1_B OR R369_2_M_차종1_C OR R369_2_M_차종1_D OR R369_2_M_차종1_E OR R369_2_M_차종1_F OR R369_2_M_차종1_G OR R369_2_M_차종1_H) AND (R369_2_M_차종2_3DR OR R369_2_M_차종2_4DR OR R369_2_M_차종2_5DR OR R369_2_M_차종2_WGN OR R369_2_M_차종2_SP1 OR R369_2_M_차종2_SP2) AND (R369_2_M_차종3_LHD OR R369_2_M_차종3_RHD) AND (R369_2_M_차종4_내수 OR R369_2_M_차종4_수출 OR R369_2_M_차종4_북미 OR R369_2_M_차종4_EEC OR R369_2_M_차종4_호주 OR R369_2_M_차종4_중동 OR R369_2_M_차종4_중국 OR R369_2_M_차종4_브라질 OR R369_2_M_차종4_SP1 OR R369_2_M_차종4_SP2 OR R369_2_M_차종4_러시아 OR R369_2_M_차종4_SP3 OR R369_2_M_차종4_SP4 OR R369_2_M_차종4_SP5 OR R369_2_M_차종4_SP6 OR R369_2_M_차종4_SP7) AND (R369_2_M_차종5_MT OR R369_2_M_차종5_AT OR R369_2_M_차종5_SP1) AND (R369_2_M_차종6_일반루프 OR R369_2_M_차종6_썬루프 OR R369_2_M_차종6_파노라마루프 OR R369_2_M_차종6_DSROOF OR R369_2_M_차종6_SP1) AND (R369_2_M_차종7_GSL OR R369_2_M_차종7_DSL OR R369_2_M_차종7_SP1 OR R369_2_M_차종7_SP2 OR R369_2_M_차종7_SP3 OR R369_2_M_차종7_SP4 OR R369_2_M_차종7_SP5 OR R369_2_M_차종7_SP6) AND (R369_2_M_차종8_2WD OR R369_2_M_차종8_4WD OR R369_2_M_차종8_SP1) AND (R369_2_M_차종9_MPI OR R369_2_M_차종9_T_GDI OR R369_2_M_차종9_SP1 OR R369_2_M_차종9_SP2 OR R369_2_M_차종9_SP3 OR R369_2_M_차종9_SP4 OR R369_2_M_차종9_SP5 OR R369_2_M_차종9_SP6 OR R369_2_M_차종9_SP7 OR R369_2_M_차종9_SP8 OR R369_2_M_차종9_SP9 OR R369_2_M_차종9_SP10 OR R369_2_M_차종9_SP11) AND (R369_2_M_차종_OPT1_슬라이딩_유 OR R369_2_M_차종_OPT1_슬라이딩_무 OR R369_2_M_차종_OPT1_R_RACK_유 OR R369_2_M_차종_OPT1_R_RACK_무 OR R369_2_M_차종_OPT1_폴딩_유 OR R369_2_M_차종_OPT1_폴딩_무 OR R369_2_M_차종_OPT1_S_REP_EATER_유 OR R369_2_M_차종_OPT1_S_REP_EATER_무 OR R369_2_M_차종_OPT1_VAN_유 OR R369_2_M_차종_OPT1_VAN_무) THEN
    _t3 := R369_2_M_SEQ <> 0;
END_IF;
R369_2_M_차종_유 := _t3;

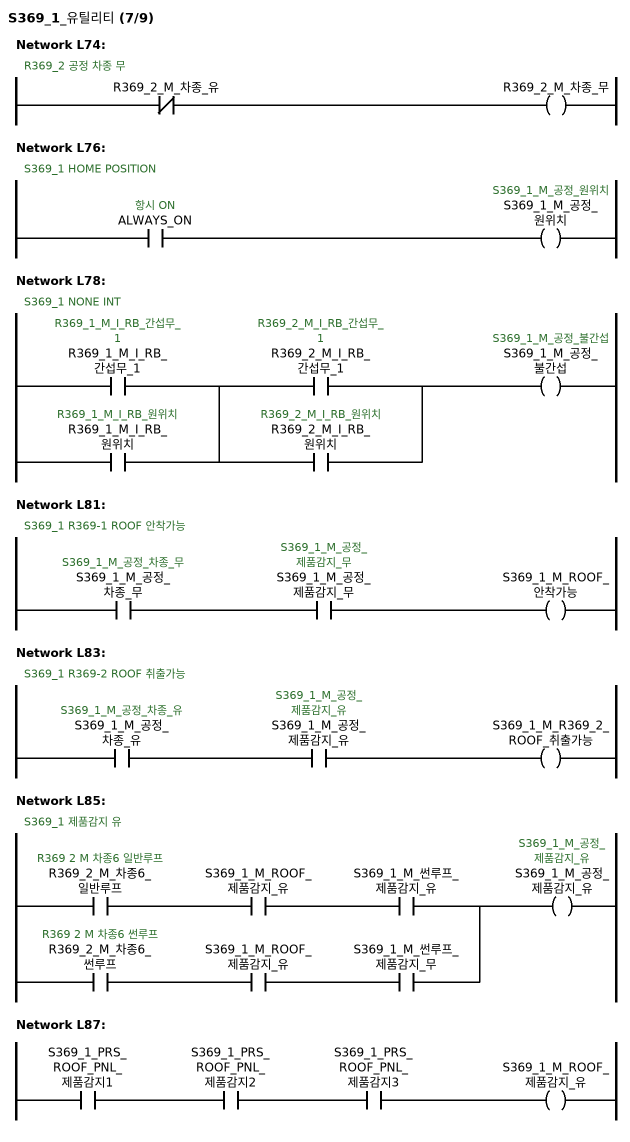
(* R369_2 공정 차종 무 *)
(* Rung L74 *)
R369_2_M_차종_무 := NOT R369_2_M_차종_유;
(* S369_1 HOME POSITION *)
(* Rung L76 *)
S369_1_M_공정_원위치 := ALWAYS_ON;
(* S369_1 NONE INT *)
(* Rung L78 *)
S369_1_M_공정_불간섭 := (R369_1_M_I_RB_간섭무_1 OR R369_1_M_I_RB_원위치) AND (R369_2_M_I_RB_간섭무_1 OR R369_2_M_I_RB_원위치);
(* S369_1 R369-1 ROOF 안착가능 *)
(* Rung L81 *)
S369_1_M_ROOF_안착가능 := S369_1_M_공정_차종_무 AND S369_1_M_공정_제품감지_무;
(* S369_1 R369-2 ROOF 취출가능 *)
(* Rung L83 *)
S369_1_M_R369_2_ROOF_취출가능 := S369_1_M_공정_차종_유 AND S369_1_M_공정_제품감지_유;
(* S369_1 제품감지 유 *)
(* Rung L85 *)
S369_1_M_공정_제품감지_유 := (R369_2_M_차종6_일반루프 AND S369_1_M_ROOF_제품감지_유 AND S369_1_M_썬루프_제품감지_유) OR (R369_2_M_차종6_썬루프 AND S369_1_M_ROOF_제품감지_유 AND S369_1_M_썬루프_제품감지_무);
(* Rung L87 *)
S369_1_M_ROOF_제품감지_유 := S369_1_PRS_ROOF_PNL_제품감지1 AND S369_1_PRS_ROOF_PNL_제품감지2 AND S369_1_PRS_ROOF_PNL_제품감지3;

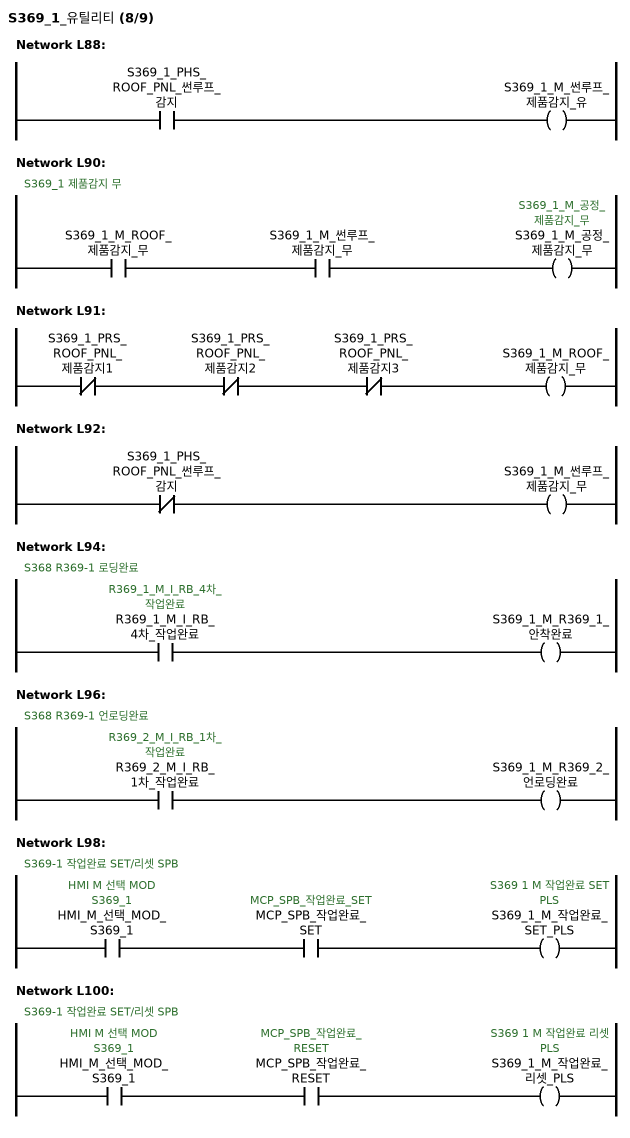
(* Rung L88 *)
S369_1_M_썬루프_제품감지_유 := S369_1_PHS_ROOF_PNL_썬루프_감지;
(* S369_1 제품감지 무 *)
(* Rung L90 *)
S369_1_M_공정_제품감지_무 := S369_1_M_ROOF_제품감지_무 AND S369_1_M_썬루프_제품감지_무;
(* Rung L91 *)
S369_1_M_ROOF_제품감지_무 := NOT S369_1_PRS_ROOF_PNL_제품감지1 AND NOT S369_1_PRS_ROOF_PNL_제품감지2 AND NOT S369_1_PRS_ROOF_PNL_제품감지3;
(* Rung L92 *)
S369_1_M_썬루프_제품감지_무 := NOT S369_1_PHS_ROOF_PNL_썬루프_감지;
(* S368 R369-1 로딩완료 *)
(* Rung L94 *)
S369_1_M_R369_1_안착완료 := R369_1_M_I_RB_4차_작업완료;
(* S368 R369-1 언로딩완료 *)
(* Rung L96 *)
S369_1_M_R369_2_언로딩완료 := R369_2_M_I_RB_1차_작업완료;
(* S369-1 작업완료 SET/리셋 SPB *)
(* Rung L98 *)
S369_1_M_작업완료_SET_PLS := HMI_M_선택_MOD_S369_1 AND MCP_SPB_작업완료_SET;
(* S369-1 작업완료 SET/리셋 SPB *)
(* Rung L100 *)
S369_1_M_작업완료_리셋_PLS := HMI_M_선택_MOD_S369_1 AND MCP_SPB_작업완료_RESET;

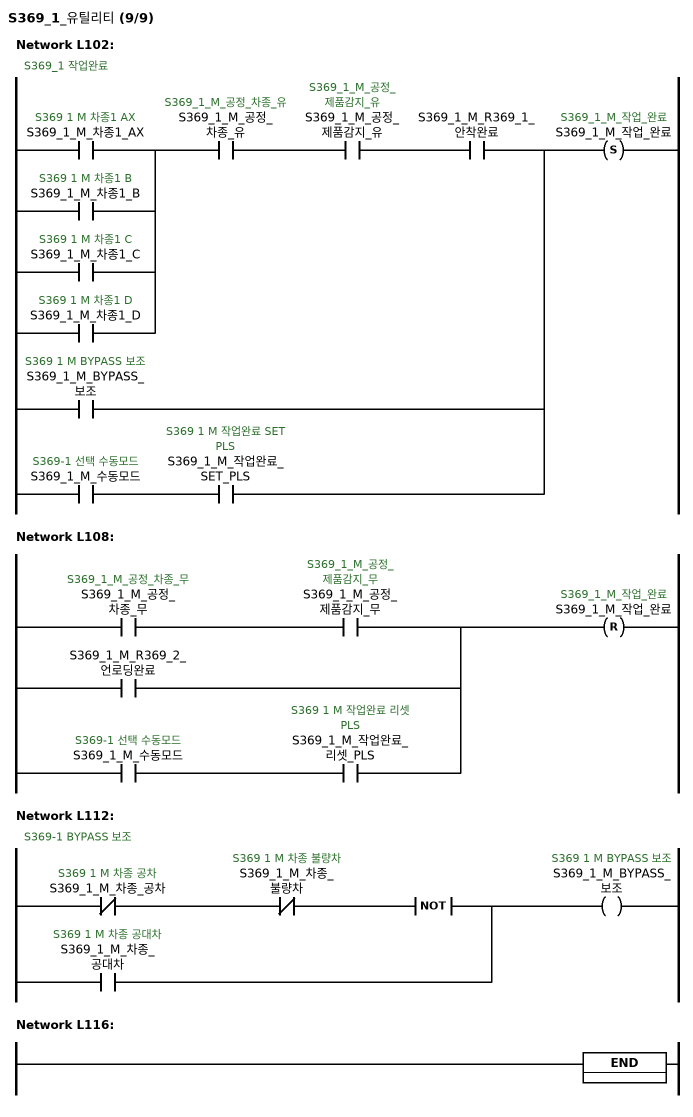
(* S369_1 작업완료 *)
(* Rung L102 *)
IF ((S369_1_M_차종1_AX OR S369_1_M_차종1_B OR S369_1_M_차종1_C OR S369_1_M_차종1_D) AND S369_1_M_공정_차종_유 AND S369_1_M_공정_제품감지_유 AND S369_1_M_R369_1_안착완료) OR S369_1_M_BYPASS_보조 OR (S369_1_M_수동모드 AND S369_1_M_작업완료_SET_PLS) THEN
    S369_1_M_작업_완료 := TRUE;
END_IF;
(* Rung L108 *)
IF (S369_1_M_공정_차종_무 AND S369_1_M_공정_제품감지_무) OR S369_1_M_R369_2_언로딩완료 OR (S369_1_M_수동모드 AND S369_1_M_작업완료_리셋_PLS) THEN
    S369_1_M_작업_완료 := FALSE;
END_IF;
(* S369-1 BYPASS 보조 *)
(* Rung L112 *)
S369_1_M_BYPASS_보조 := NOT (NOT S369_1_M_차종_공차 AND NOT S369_1_M_차종_불량차) OR S369_1_M_차종_공대차;
(* Rung L116 *)
END();
END_PROGRAM

PROGRAM S369_1_로보트(R369_1_&_R369_2) (* task: 스캔 프로그램 *)
VAR_EXTERNAL RETAIN
    ALWAYS_ON : BOOL; (* AT %MW3.1 *) (* 항시 ON *)
    MCP_M_부저_정지 : BOOL; (* AT %MW350.5 *) (* MCP 부저정지 *)
    MCP_M_비상정지 : BOOL; (* AT %MW350.7 *) (* MCP 비상정지 이상 *)
    R369_1_M_차종6_썬루프 : BOOL; (* AT %MW10063.4 *) (* R369 1 M 차종6 썬루프 *)
    R369_1_M_차종6_일반루프 : BOOL; (* AT %MW10063.3 *) (* R369 1 M 차종6 일반루프 *)
    R369_1_M_차종_유 : BOOL; (* AT %MW4502.2 *)
    S364_M_공정_차종_AX : BOOL; (* AT %MW2002.3 *) (* S364_M_공정_차종_AX *)
    S364_M_자동_START : BOOL; (* AT %MW2000.5 *) (* S364 자동운전중 *)
    S364_M_자동_운전중 : BOOL; (* AT %MW2000.4 *) (* S364 자동운전중 *)
    S364_M_작업_완료 : BOOL; (* AT %MW2001.0 *) (* S364_M_작업_완료 *)
    S364_M_총괄_이상 : BOOL; (* AT %MW2009.0 *) (* S364_M_총괄_이상 *)
    S367_M_369_1_언로딩가능 : BOOL; (* AT %MW3504.10 *)
    S367_M_공정_제품감지_유 : BOOL; (* AT %MW3501.5 *) (* S367_M_공정_제품감지_유 *)
    S367_M_공정_차종_유 : BOOL; (* AT %MW3502.0 *) (* S367_M_공정_차종_유 *)
    S367_M_작업_완료 : BOOL; (* AT %MW3501.0 *) (* S367_M_작업_완료 *)
    S367_M_차종1_AX : BOOL; (* AT %MW10181.0 *) (* S367 M 차종1 AX *)
    S367_M_차종6_썬루프 : BOOL; (* AT %MW10183.4 *) (* S367 M 차종6 썬루프 *)
    S367_M_차종6_일반루프 : BOOL; (* AT %MW10183.3 *) (* S367 M 차종6 일반루프 *)
    S368_M_R369_1_안착가능 : BOOL; (* AT %MW4004.8 *)
    S368_M_R369_1_안착완료 : BOOL; (* AT %MW4001.1 *)
    S368_M_공정_제품감지_무 : BOOL; (* AT %MW4001.6 *) (* S368_M_공정_제품감지_무 *)
    S368_M_공정_제품감지_유 : BOOL; (* AT %MW4001.5 *) (* S368_M_공정_제품감지_유 *)
    S368_M_공정_차종_무 : BOOL; (* AT %MW4002.1 *) (* S368_M_공정_차종_무 *)
    S368_M_공정_차종_유 : BOOL; (* AT %MW4002.0 *) (* S368_M_공정_차종_유 *)
    S368_M_작업_완료 : BOOL; (* AT %MW4001.0 *) (* S368_M_작업_완료 *)
    S369_1_M_R369_1_안착완료 : BOOL; (* AT %MW4501.1 *)
    S369_1_M_R369_2_ROOF_취출가능 : BOOL; (* AT %MW4504.9 *)
    S369_1_M_ROOF_안착가능 : BOOL; (* AT %MW4504.8 *)
    S369_1_M_공정_제품감지_무 : BOOL; (* AT %MW4501.4 *) (* S369_1_M_공정_제품감지_무 *)
    S369_1_M_공정_제품감지_유 : BOOL; (* AT %MW4501.3 *) (* S369_1_M_공정_제품감지_유 *)
    S369_1_M_공정_차종_무 : BOOL; (* AT %MW4502.1 *) (* S369_1_M_공정_차종_무 *)
    S369_1_M_공정_차종_유 : BOOL; (* AT %MW4502.0 *) (* S369_1_M_공정_차종_유 *)
    S369_1_M_수동모드 : BOOL; (* AT %MW4500.3 *) (* S369-1 선택 수동모드 *)
    S369_1_M_자동_운전중 : BOOL; (* AT %MW4500.4 *) (* S369-1 자동운전중 *)
    S369_1_M_작업_완료 : BOOL; (* AT %MW4501.0 *) (* S369_1_M_작업_완료 *)
    S369_1_M_작업완료_SET_PLS : BOOL; (* AT %MW4500.8 *) (* S369 1 M 작업완료 SET PLS *)
    S369_1_M_작업완료_리셋_PLS : BOOL; (* AT %MW4500.9 *) (* S369 1 M 작업완료 리셋 PLS *)
    S369_1_M_차종1_AX : BOOL; (* AT %MW10221.0 *) (* S369 1 M 차종1 AX *)
    S369_1_M_총괄_이상 : BOOL; (* AT %MW4509.0 *) (* S369_1_M_총괄_이상 *)
    S369_M_R369_2_로딩가능 : BOOL; (* AT %MW5004.8 *)
    S369_M_로딩_이젝터_제품감지_무 : BOOL; (* AT %MW5001.9 *)
    S369_M_로딩_작업_완료 : BOOL; (* AT %MW5001.0 *) (* S369_M_작업_완료 *)
    S369_M_로딩버퍼_제품감지_무 : BOOL; (* AT %MW5005.1 *) (* S369_로딩버퍼_제품감지_무 *)
    S369_M_로딩버퍼_차종_무 : BOOL; (* AT %MW5002.1 *)
    S369_M_자동_START : BOOL; (* AT %MW5000.5 *) (* S369 자동운전중 *)
    S369_M_자동_운전중 : BOOL; (* AT %MW5000.4 *) (* S369 자동운전중 *)
    S369_M_총괄_이상 : BOOL; (* AT %MW5009.0 *) (* S369_M_총괄_이상 *)
    전체_M_GATE_비상정지_정상 : BOOL; (* AT %MW308.4 *) (* 전체 M GATE 비상정지 정상 *)
    전체_M_GATE_자동기동 : BOOL; (* AT %MW308.1 *) (* 전체_M_자동_운전 *)
    전체_M_운전준비_보조 : BOOL; (* AT %MW308.5 *)
    전체_M_이상_리셋 : BOOL; (* AT %MW308.2 *) (* ALL공정 PB 이상리셋 *)
    전체_공정_M_총괄_비상정지_정상 : BOOL; (* AT %MW304.1 *)
END_VAR
VAR
    INST1 : FB494_Robot_Hyundai_HMMI_v1;
    INST2 : FB494_Robot_Hyundai_HMMI_v1;
    R361_1_M_RB_PROG_NO : INT;
    R369_1_M_RB_PROG_NO : INT;
    R369_2_M_RB_PROG_NO : INT;
    로보트제외 : BOOL;
END_VAR
VAR_EXTERNAL
    MCP_PBL_운전준비_ON : BOOL; (* AT %MW87630.0 *) (* MCP_PBL_운전준비_ON *)
    R361_1_I_RB_INPUT : ARRAY[0..3] OF WORD; (* AT %MW84010 *) (* R361_1_I_RB_INPUT *)
    R361_1_M_I_RB_1차_작업완료 : BOOL; (* AT %MW20011.2 *) (* R361_1_M_I_RB_1차_작업완료 *)
    R361_1_M_I_RB_2차_작업완료 : BOOL; (* AT %MW20011.3 *) (* R361_1_M_I_RB_2차_작업완료 *)
    R361_1_M_I_RB_3차_작업완료 : BOOL; (* AT %MW20011.4 *) (* R361_1_M_I_RB_3차_작업완료 *)
    R361_1_M_I_RB_4차_작업완료 : BOOL; (* AT %MW20011.5 *) (* R361_1_M_I_RB_4차_작업완료 *)
    R361_1_M_I_RB_5차_작업완료 : BOOL; (* AT %MW20011.6 *) (* R361_1_M_I_RB_5차_작업완료 *)
    R361_1_M_I_RB_6차_작업완료 : BOOL; (* AT %MW20011.7 *) (* R361_1_M_I_RB_6차_작업완료 *)
    R361_1_M_I_RB_7차_작업완료 : BOOL; (* AT %MW20011.8 *) (* R361_1_M_I_RB_7차_작업완료 *)
    R361_1_M_I_RB_PAUSE_보조 : BOOL; (* AT %MW20010.5 *) (* R361_1_M_I_RB_PAUSE_보조 *)
    R361_1_M_I_RB_PLC_RUN_CHK_이상 : BOOL; (* AT %MW20010.7 *) (* R361_1_M_I_RB_PLC_RUN_CHK_이상 *)
    R361_1_M_I_RB_간섭무_1 : BOOL; (* AT %MW20012.0 *) (* R361_1_M_I_RB_간섭무_1 *)
    R361_1_M_I_RB_간섭무_10 : BOOL; (* AT %MW20012.9 *) (* R361_1_M_I_RB_간섭무_10 *)
    R361_1_M_I_RB_간섭무_11 : BOOL; (* AT %MW20012.10 *) (* R361_1_M_I_RB_간섭무_11 *)
    R361_1_M_I_RB_간섭무_12 : BOOL; (* AT %MW20012.11 *) (* R361_1_M_I_RB_간섭무_12 *)
    R361_1_M_I_RB_간섭무_2 : BOOL; (* AT %MW20012.1 *) (* R361_1_M_I_RB_간섭무_2 *)
    R361_1_M_I_RB_간섭무_3 : BOOL; (* AT %MW20012.2 *) (* R361_1_M_I_RB_간섭무_3 *)
    R361_1_M_I_RB_간섭무_4 : BOOL; (* AT %MW20012.3 *) (* R361_1_M_I_RB_간섭무_4 *)
    R361_1_M_I_RB_간섭무_5 : BOOL; (* AT %MW20012.4 *) (* R361_1_M_I_RB_간섭무_5 *)
    R361_1_M_I_RB_간섭무_6 : BOOL; (* AT %MW20012.5 *) (* R361_1_M_I_RB_간섭무_6 *)
    R361_1_M_I_RB_간섭무_7 : BOOL; (* AT %MW20012.6 *) (* R361_1_M_I_RB_간섭무_7 *)
    R361_1_M_I_RB_간섭무_8 : BOOL; (* AT %MW20012.7 *) (* R361_1_M_I_RB_간섭무_8 *)
    R361_1_M_I_RB_간섭무_9 : BOOL; (* AT %MW20012.8 *) (* R361_1_M_I_RB_간섭무_9 *)
    R361_1_M_I_RB_비상정지 : BOOL; (* AT %MW20010.4 *) (* R361_1_M_I_RB_비상정지 *)
    R361_1_M_I_RB_운전준비 : BOOL; (* AT %MW20010.0 *) (* R361_1_M_I_RB_운전준비 *)
    R361_1_M_I_RB_원위치 : BOOL; (* AT %MW20010.3 *) (* R361_1_M_I_RB_원위치 *)
    R361_1_M_I_RB_이상 : BOOL; (* AT %MW20010.2 *) (* R361_1_M_I_RB_이상 *)
    R361_1_M_I_RB_자동 : BOOL; (* AT %MW20010.1 *) (* R361_1_M_I_RB_자동 *)
    R361_1_M_I_RB_최종작업완료 : BOOL; (* AT %MW20011.0 *) (* R361_1_M_I_RB_최종작업완료 *)
    R361_1_M_I_RB_프로그램_이상 : BOOL; (* AT %MW20010.6 *) (* R361_1_M_I_RB_프로그램_이상 *)
    R361_1_M_O_RB_1_CYCLE_SET : BOOL; (* AT %MW21010.3 *) (* R361_1_M_O_RB_1_CYCLE_SET *)
    R361_1_M_O_RB_1차_작업완료_리셋 : BOOL; (* AT %MW21012.0 *) (* R361_1_M_O_RB_1차_작업완료_리셋 *)
    R361_1_M_O_RB_2차_작업완료_리셋 : BOOL; (* AT %MW21012.1 *) (* R361_1_M_O_RB_2차_작업완료_리셋 *)
    R361_1_M_O_RB_2차_진입OK : BOOL; (* AT %MW21011.8 *) (* R361_1_M_O_RB_2차_진입OK *)
    R361_1_M_O_RB_3차_작업완료_리셋 : BOOL; (* AT %MW21012.2 *) (* R361_1_M_O_RB_3차_작업완료_리셋 *)
    R361_1_M_O_RB_3차_진입OK : BOOL; (* AT %MW21011.9 *) (* R361_1_M_O_RB_3차_진입OK *)
    R361_1_M_O_RB_4차_작업완료_리셋 : BOOL; (* AT %MW21012.3 *) (* R361_1_M_O_RB_4차_작업완료_리셋 *)
    R361_1_M_O_RB_4차_진입OK : BOOL; (* AT %MW21011.10 *) (* R361_1_M_O_RB_4차_진입OK *)
    R361_1_M_O_RB_5차_작업완료_리셋 : BOOL; (* AT %MW21012.4 *) (* R361_1_M_O_RB_5차_작업완료_리셋 *)
    R361_1_M_O_RB_5차_진입OK : BOOL; (* AT %MW21011.11 *) (* R361_1_M_O_RB_5차_진입OK *)
    R361_1_M_O_RB_6차_작업완료_리셋 : BOOL; (* AT %MW21012.5 *) (* R361_1_M_O_RB_6차_작업완료_리셋 *)
    R361_1_M_O_RB_6차_진입OK : BOOL; (* AT %MW21011.12 *) (* R361_1_M_O_RB_6차_진입OK *)
    R361_1_M_O_RB_7차_작업완료_리셋 : BOOL; (* AT %MW21012.6 *) (* R361_1_M_O_RB_7차_작업완료_리셋 *)
    R361_1_M_O_RB_7차_진입OK : BOOL; (* AT %MW21011.13 *) (* R361_1_M_O_RB_7차_진입OK *)
    R361_1_M_O_RB_ATD_OK : BOOL; (* AT %MW21010.6 *) (* R361_1_M_O_RB_ATD_OK *)
    R361_1_M_O_RB_PLT_10_진입OK : BOOL; (* AT %MW21013.10 *) (* R361_1_M_O_RB_PLT_10_진입OK *)
    R361_1_M_O_RB_PLT_11_진입OK : BOOL; (* AT %MW21013.11 *) (* R361_1_M_O_RB_PLT_11_진입OK *)
    R361_1_M_O_RB_PLT_12_진입OK : BOOL; (* AT %MW21013.12 *) (* R361_1_M_O_RB_PLT_12_진입OK *)
    R361_1_M_O_RB_PLT_1_진입OK : BOOL; (* AT %MW21013.1 *) (* R361_1_M_O_RB_PLT_1_진입OK *)
    R361_1_M_O_RB_PLT_2_진입OK : BOOL; (* AT %MW21013.2 *) (* R361_1_M_O_RB_PLT_2_진입OK *)
    R361_1_M_O_RB_PLT_3_진입OK : BOOL; (* AT %MW21013.3 *) (* R361_1_M_O_RB_PLT_3_진입OK *)
    R361_1_M_O_RB_PLT_4_진입OK : BOOL; (* AT %MW21013.4 *) (* R361_1_M_O_RB_PLT_4_진입OK *)
    R361_1_M_O_RB_PLT_5_진입OK : BOOL; (* AT %MW21013.5 *) (* R361_1_M_O_RB_PLT_5_진입OK *)
    R361_1_M_O_RB_PLT_6_진입OK : BOOL; (* AT %MW21013.6 *) (* R361_1_M_O_RB_PLT_6_진입OK *)
    R361_1_M_O_RB_PLT_7_진입OK : BOOL; (* AT %MW21013.7 *) (* R361_1_M_O_RB_PLT_7_진입OK *)
    R361_1_M_O_RB_PLT_8_진입OK : BOOL; (* AT %MW21013.8 *) (* R361_1_M_O_RB_PLT_8_진입OK *)
    R361_1_M_O_RB_PLT_9_진입OK : BOOL; (* AT %MW21013.9 *) (* R361_1_M_O_RB_PLT_9_진입OK *)
    R361_1_M_O_RB_PLT_카운터리셋_보조 : BOOL; (* AT %MW21010.10 *) (* R361_1_M_O_RB_PLT_카운터리셋_보조 *)
    R361_1_M_O_RB_RESTART_OK : BOOL; (* AT %MW21010.2 *) (* R361_1_M_O_RB_RESTART_OK *)
    R361_1_M_O_RB_START_OK : BOOL; (* AT %MW21010.0 *) (* R361_1_M_O_RB_START_OK *)
    R361_1_M_O_RB_TEST_MODE_5000회 : BOOL; (* AT %MW21010.12 *) (* R361_1_M_O_RB_TEST_MODE_5000회 *)
    R361_1_M_O_RB_TIP_교체_시작 : BOOL; (* AT %MW21010.7 *) (* R361_1_M_O_RB_TIP_교체_시작 *)
    R361_1_M_O_RB_TIP_교체_완료 : BOOL; (* AT %MW21010.8 *) (* R361_1_M_O_RB_TIP_교체_완료 *)
    R361_1_M_O_RB_VIP_MODE : BOOL; (* AT %MW21010.11 *) (* R361_1_M_O_RB_VIP_MODE *)
    R361_1_M_O_RB_냉각수_차단_요청 : BOOL; (* AT %MW21010.9 *) (* R361_1_M_O_RB_냉각수_차단_요청 *)
    R361_1_M_O_RB_진입OK_AX차종 : BOOL; (* AT %MW21011.0 *) (* R361_1_M_O_RB_진입OK_AX차종 *)
    R361_1_M_O_RB_진입OK_B차종 : BOOL; (* AT %MW21011.1 *) (* R361_1_M_O_RB_진입OK_B차종 *)
    R361_1_M_O_RB_진입OK_C차종 : BOOL; (* AT %MW21011.2 *) (* R361_1_M_O_RB_진입OK_C차종 *)
    R361_1_M_O_RB_진입OK_D차종 : BOOL; (* AT %MW21011.3 *) (* R361_1_M_O_RB_진입OK_D차종 *)
    R361_1_M_O_RB_진입OK_E차종 : BOOL; (* AT %MW21011.4 *) (* R361_1_M_O_RB_진입OK_E차종 *)
    R361_1_M_O_RB_진입OK_F차종 : BOOL; (* AT %MW21011.5 *) (* R361_1_M_O_RB_진입OK_F차종 *)
    R361_1_M_O_RB_진입OK_G차종 : BOOL; (* AT %MW21011.6 *) (* R361_1_M_O_RB_진입OK_G차종 *)
    R361_1_M_O_RB_진입OK_H차종 : BOOL; (* AT %MW21011.7 *) (* R361_1_M_O_RB_진입OK_H차종 *)
    R361_1_M_O_RB_최종_작업완료_리셋 : BOOL; (* AT %MW21010.5 *) (* R361_1_M_O_RB_최종_작업완료_리셋 *)
    R361_1_M_O_RB_프로그램_OK : BOOL; (* AT %MW21010.1 *) (* R361_1_M_O_RB_프로그램_OK *)
    R361_1_O_RB_OUTPUT : ARRAY[0..3] OF WORD; (* AT %MW94010 *) (* R361_1_O_RB_OUTPUT *)
    R363_1_M_O_RB_6차_작업완료_리셋 : BOOL; (* AT %MW21032.5 *) (* R363_1_M_O_RB_6차_작업완료_리셋 *)
    R363_1_M_O_RB_최종_작업완료_리셋 : BOOL; (* AT %MW21030.5 *) (* R363_1_M_O_RB_최종_작업완료_리셋 *)
    R369_1_I_RB_INPUT : ARRAY[0..3] OF WORD; (* AT %MW84080 *) (* R369_1_I_RB_INPUT *)
    R369_1_M_I_RB_1차_작업완료 : BOOL; (* AT %MW20081.2 *) (* R369_1_M_I_RB_1차_작업완료 *)
    R369_1_M_I_RB_2차_작업완료 : BOOL; (* AT %MW20081.3 *) (* R369_1_M_I_RB_2차_작업완료 *)
    R369_1_M_I_RB_3차_작업완료 : BOOL; (* AT %MW20081.4 *) (* R369_1_M_I_RB_3차_작업완료 *)
    R369_1_M_I_RB_4차_작업완료 : BOOL; (* AT %MW20081.5 *) (* R369_1_M_I_RB_4차_작업완료 *)
    R369_1_M_I_RB_5차_작업완료 : BOOL; (* AT %MW20081.6 *) (* R369_1_M_I_RB_5차_작업완료 *)
    R369_1_M_I_RB_6차_작업완료 : BOOL; (* AT %MW20081.7 *) (* R369_1_M_I_RB_6차_작업완료 *)
    R369_1_M_I_RB_7차_작업완료 : BOOL; (* AT %MW20081.8 *) (* R369_1_M_I_RB_7차_작업완료 *)
    R369_1_M_I_RB_PAUSE_보조 : BOOL; (* AT %MW20080.5 *) (* R369_1_M_I_RB_PAUSE_보조 *)
    R369_1_M_I_RB_PLC_RUN_CHK_이상 : BOOL; (* AT %MW20080.7 *) (* R369_1_M_I_RB_PLC_RUN_CHK_이상 *)
    R369_1_M_I_RB_간섭무_1 : BOOL; (* AT %MW20082.0 *) (* R369_1_M_I_RB_간섭무_1 *)
    R369_1_M_I_RB_간섭무_10 : BOOL; (* AT %MW20082.9 *) (* R369_1_M_I_RB_간섭무_10 *)
    R369_1_M_I_RB_간섭무_11 : BOOL; (* AT %MW20082.10 *) (* R369_1_M_I_RB_간섭무_11 *)
    R369_1_M_I_RB_간섭무_12 : BOOL; (* AT %MW20082.11 *) (* R369_1_M_I_RB_간섭무_12 *)
    R369_1_M_I_RB_간섭무_2 : BOOL; (* AT %MW20082.1 *) (* R369_1_M_I_RB_간섭무_2 *)
    R369_1_M_I_RB_간섭무_3 : BOOL; (* AT %MW20082.2 *) (* R369_1_M_I_RB_간섭무_3 *)
    R369_1_M_I_RB_간섭무_4 : BOOL; (* AT %MW20082.3 *) (* R369_1_M_I_RB_간섭무_4 *)
    R369_1_M_I_RB_간섭무_5 : BOOL; (* AT %MW20082.4 *) (* R369_1_M_I_RB_간섭무_5 *)
    R369_1_M_I_RB_간섭무_6 : BOOL; (* AT %MW20082.5 *) (* R369_1_M_I_RB_간섭무_6 *)
    R369_1_M_I_RB_간섭무_7 : BOOL; (* AT %MW20082.6 *) (* R369_1_M_I_RB_간섭무_7 *)
    R369_1_M_I_RB_간섭무_8 : BOOL; (* AT %MW20082.7 *) (* R369_1_M_I_RB_간섭무_8 *)
    R369_1_M_I_RB_간섭무_9 : BOOL; (* AT %MW20082.8 *) (* R369_1_M_I_RB_간섭무_9 *)
    R369_1_M_I_RB_비상정지 : BOOL; (* AT %MW20080.4 *) (* R369_1_M_I_RB_비상정지 *)
    R369_1_M_I_RB_운전준비 : BOOL; (* AT %MW20080.0 *) (* R369_1_M_I_RB_운전준비 *)
    R369_1_M_I_RB_원위치 : BOOL; (* AT %MW20080.3 *) (* R369_1_M_I_RB_원위치 *)
    R369_1_M_I_RB_이상 : BOOL; (* AT %MW20080.2 *) (* R369_1_M_I_RB_이상 *)
    R369_1_M_I_RB_자동 : BOOL; (* AT %MW20080.1 *) (* R369_1_M_I_RB_자동 *)
    R369_1_M_I_RB_최종작업완료 : BOOL; (* AT %MW20081.0 *) (* R369_1_M_I_RB_최종작업완료 *)
    R369_1_M_I_RB_프로그램_이상 : BOOL; (* AT %MW20080.6 *) (* R369_1_M_I_RB_프로그램_이상 *)
    R369_1_M_O_RB_1_CYCLE_SET : BOOL; (* AT %MW21080.3 *) (* R369_1_M_O_RB_1_CYCLE_SET *)
    R369_1_M_O_RB_1차_작업완료_리셋 : BOOL; (* AT %MW21082.0 *) (* R369_1_M_O_RB_1차_작업완료_리셋 *)
    R369_1_M_O_RB_2차_작업완료_리셋 : BOOL; (* AT %MW21082.1 *) (* R369_1_M_O_RB_2차_작업완료_리셋 *)
    R369_1_M_O_RB_2차_진입OK : BOOL; (* AT %MW21081.8 *) (* R369_1_M_O_RB_2차_진입OK *)
    R369_1_M_O_RB_3차_작업완료_리셋 : BOOL; (* AT %MW21082.2 *) (* R369_1_M_O_RB_3차_작업완료_리셋 *)
    R369_1_M_O_RB_3차_진입OK : BOOL; (* AT %MW21081.9 *) (* R369_1_M_O_RB_3차_진입OK *)
    R369_1_M_O_RB_4차_작업완료_리셋 : BOOL; (* AT %MW21082.3 *) (* R369_1_M_O_RB_4차_작업완료_리셋 *)
    R369_1_M_O_RB_4차_진입OK : BOOL; (* AT %MW21081.10 *) (* R369_1_M_O_RB_4차_진입OK *)
    R369_1_M_O_RB_5차_작업완료_리셋 : BOOL; (* AT %MW21082.4 *) (* R369_1_M_O_RB_5차_작업완료_리셋 *)
    R369_1_M_O_RB_5차_진입OK : BOOL; (* AT %MW21081.11 *) (* R369_1_M_O_RB_5차_진입OK *)
    R369_1_M_O_RB_6차_작업완료_리셋 : BOOL; (* AT %MW21082.5 *) (* R369_1_M_O_RB_6차_작업완료_리셋 *)
    R369_1_M_O_RB_6차_진입OK : BOOL; (* AT %MW21081.12 *) (* R369_1_M_O_RB_6차_진입OK *)
    R369_1_M_O_RB_7차_작업완료_리셋 : BOOL; (* AT %MW21082.6 *) (* R369_1_M_O_RB_7차_작업완료_리셋 *)
    R369_1_M_O_RB_7차_진입OK : BOOL; (* AT %MW21081.13 *) (* R369_1_M_O_RB_7차_진입OK *)
    R369_1_M_O_RB_ATD_OK : BOOL; (* AT %MW21080.6 *) (* R369_1_M_O_RB_ATD_OK *)
    R369_1_M_O_RB_PLT_10_진입OK : BOOL; (* AT %MW21083.10 *) (* R369_1_M_O_RB_PLT_10_진입OK *)
    R369_1_M_O_RB_PLT_11_진입OK : BOOL; (* AT %MW21083.11 *) (* R369_1_M_O_RB_PLT_11_진입OK *)
    R369_1_M_O_RB_PLT_12_진입OK : BOOL; (* AT %MW21083.12 *) (* R369_1_M_O_RB_PLT_12_진입OK *)
    R369_1_M_O_RB_PLT_1_진입OK : BOOL; (* AT %MW21083.1 *) (* R369_1_M_O_RB_PLT_1_진입OK *)
    R369_1_M_O_RB_PLT_2_진입OK : BOOL; (* AT %MW21083.2 *) (* R369_1_M_O_RB_PLT_2_진입OK *)
    R369_1_M_O_RB_PLT_3_진입OK : BOOL; (* AT %MW21083.3 *) (* R369_1_M_O_RB_PLT_3_진입OK *)
    R369_1_M_O_RB_PLT_4_진입OK : BOOL; (* AT %MW21083.4 *) (* R369_1_M_O_RB_PLT_4_진입OK *)
    R369_1_M_O_RB_PLT_5_진입OK : BOOL; (* AT %MW21083.5 *) (* R369_1_M_O_RB_PLT_5_진입OK *)
    R369_1_M_O_RB_PLT_6_진입OK : BOOL; (* AT %MW21083.6 *) (* R369_1_M_O_RB_PLT_6_진입OK *)
    R369_1_M_O_RB_PLT_7_진입OK : BOOL; (* AT %MW21083.7 *) (* R369_1_M_O_RB_PLT_7_진입OK *)
    R369_1_M_O_RB_PLT_8_진입OK : BOOL; (* AT %MW21083.8 *) (* R369_1_M_O_RB_PLT_8_진입OK *)
    R369_1_M_O_RB_PLT_9_진입OK : BOOL; (* AT %MW21083.9 *) (* R369_1_M_O_RB_PLT_9_진입OK *)
    R369_1_M_O_RB_PLT_카운터리셋_보조 : BOOL; (* AT %MW21080.10 *) (* R369_1_M_O_RB_PLT_카운터리셋_보조 *)
    R369_1_M_O_RB_PROG_NO : WORD; (* AT %MW21084 *)
    R369_1_M_O_RB_RESTART_OK : BOOL; (* AT %MW21080.2 *) (* R369_1_M_O_RB_RESTART_OK *)
    R369_1_M_O_RB_START_OK : BOOL; (* AT %MW21080.0 *) (* R369_1_M_O_RB_START_OK *)
    R369_1_M_O_RB_TEST_MODE_5000회 : BOOL; (* AT %MW21080.12 *) (* R369_1_M_O_RB_TEST_MODE_5000회 *)
    R369_1_M_O_RB_TIP_교체_시작 : BOOL; (* AT %MW21080.7 *) (* R369_1_M_O_RB_TIP_교체_시작 *)
    R369_1_M_O_RB_TIP_교체_완료 : BOOL; (* AT %MW21080.8 *) (* R369_1_M_O_RB_TIP_교체_완료 *)
    R369_1_M_O_RB_VIP_MODE : BOOL; (* AT %MW21080.11 *) (* R369_1_M_O_RB_VIP_MODE *)
    R369_1_M_O_RB_냉각수_차단_요청 : BOOL; (* AT %MW21080.9 *) (* R369_1_M_O_RB_냉각수_차단_요청 *)
    R369_1_M_O_RB_진입OK_AX차종 : BOOL; (* AT %MW21081.0 *) (* R369_1_M_O_RB_진입OK_AX차종 *)
    R369_1_M_O_RB_진입OK_B차종 : BOOL; (* AT %MW21081.1 *) (* R369_1_M_O_RB_진입OK_B차종 *)
    R369_1_M_O_RB_진입OK_C차종 : BOOL; (* AT %MW21081.2 *) (* R369_1_M_O_RB_진입OK_C차종 *)
    R369_1_M_O_RB_진입OK_D차종 : BOOL; (* AT %MW21081.3 *) (* R369_1_M_O_RB_진입OK_D차종 *)
    R369_1_M_O_RB_진입OK_E차종 : BOOL; (* AT %MW21081.4 *) (* R369_1_M_O_RB_진입OK_E차종 *)
    R369_1_M_O_RB_진입OK_F차종 : BOOL; (* AT %MW21081.5 *) (* R369_1_M_O_RB_진입OK_F차종 *)
    R369_1_M_O_RB_진입OK_G차종 : BOOL; (* AT %MW21081.6 *) (* R369_1_M_O_RB_진입OK_G차종 *)
    R369_1_M_O_RB_진입OK_H차종 : BOOL; (* AT %MW21081.7 *) (* R369_1_M_O_RB_진입OK_H차종 *)
    R369_1_M_O_RB_최종_작업완료_리셋 : BOOL; (* AT %MW21080.5 *) (* R369_1_M_O_RB_최종_작업완료_리셋 *)
    R369_1_M_O_RB_프로그램_OK : BOOL; (* AT %MW21080.1 *) (* R369_1_M_O_RB_프로그램_OK *)
    R369_1_O_RB_OUTPUT : ARRAY[0..3] OF WORD; (* AT %MW94080 *) (* R369_1_O_RB_OUTPUT *)
    R369_2_I_RB_INPUT : ARRAY[0..3] OF WORD; (* AT %MW84090 *) (* R369_2_I_RB_INPUT *)
    R369_2_M_I_RB_1차_작업완료 : BOOL; (* AT %MW20091.2 *) (* R369_2_M_I_RB_1차_작업완료 *)
    R369_2_M_I_RB_2차_작업완료 : BOOL; (* AT %MW20091.3 *) (* R369_2_M_I_RB_2차_작업완료 *)
    R369_2_M_I_RB_3차_작업완료 : BOOL; (* AT %MW20091.4 *) (* R369_2_M_I_RB_3차_작업완료 *)
    R369_2_M_I_RB_4차_작업완료 : BOOL; (* AT %MW20091.5 *) (* R369_2_M_I_RB_4차_작업완료 *)
    R369_2_M_I_RB_5차_작업완료 : BOOL; (* AT %MW20091.6 *) (* R369_2_M_I_RB_5차_작업완료 *)
    R369_2_M_I_RB_6차_작업완료 : BOOL; (* AT %MW20091.7 *) (* R369_2_M_I_RB_6차_작업완료 *)
    R369_2_M_I_RB_7차_작업완료 : BOOL; (* AT %MW20091.8 *) (* R369_2_M_I_RB_7차_작업완료 *)
    R369_2_M_I_RB_PAUSE_보조 : BOOL; (* AT %MW20090.5 *) (* R369_2_M_I_RB_PAUSE_보조 *)
    R369_2_M_I_RB_PLC_RUN_CHK_이상 : BOOL; (* AT %MW20090.7 *) (* R369_2_M_I_RB_PLC_RUN_CHK_이상 *)
    R369_2_M_I_RB_간섭무_1 : BOOL; (* AT %MW20092.0 *) (* R369_2_M_I_RB_간섭무_1 *)
    R369_2_M_I_RB_간섭무_10 : BOOL; (* AT %MW20092.9 *) (* R369_2_M_I_RB_간섭무_10 *)
    R369_2_M_I_RB_간섭무_11 : BOOL; (* AT %MW20092.10 *) (* R369_2_M_I_RB_간섭무_11 *)
    R369_2_M_I_RB_간섭무_12 : BOOL; (* AT %MW20092.11 *) (* R369_2_M_I_RB_간섭무_12 *)
    R369_2_M_I_RB_간섭무_2 : BOOL; (* AT %MW20092.1 *) (* R369_2_M_I_RB_간섭무_2 *)
    R369_2_M_I_RB_간섭무_3 : BOOL; (* AT %MW20092.2 *) (* R369_2_M_I_RB_간섭무_3 *)
    R369_2_M_I_RB_간섭무_4 : BOOL; (* AT %MW20092.3 *) (* R369_2_M_I_RB_간섭무_4 *)
    R369_2_M_I_RB_간섭무_5 : BOOL; (* AT %MW20092.4 *) (* R369_2_M_I_RB_간섭무_5 *)
    R369_2_M_I_RB_간섭무_6 : BOOL; (* AT %MW20092.5 *) (* R369_2_M_I_RB_간섭무_6 *)
    R369_2_M_I_RB_간섭무_7 : BOOL; (* AT %MW20092.6 *) (* R369_2_M_I_RB_간섭무_7 *)
    R369_2_M_I_RB_간섭무_8 : BOOL; (* AT %MW20092.7 *) (* R369_2_M_I_RB_간섭무_8 *)
    R369_2_M_I_RB_간섭무_9 : BOOL; (* AT %MW20092.8 *) (* R369_2_M_I_RB_간섭무_9 *)
    R369_2_M_I_RB_비상정지 : BOOL; (* AT %MW20090.4 *) (* R369_2_M_I_RB_비상정지 *)
    R369_2_M_I_RB_운전준비 : BOOL; (* AT %MW20090.0 *) (* R369_2_M_I_RB_운전준비 *)
    R369_2_M_I_RB_원위치 : BOOL; (* AT %MW20090.3 *) (* R369_2_M_I_RB_원위치 *)
    R369_2_M_I_RB_이상 : BOOL; (* AT %MW20090.2 *) (* R369_2_M_I_RB_이상 *)
    R369_2_M_I_RB_자동 : BOOL; (* AT %MW20090.1 *) (* R369_2_M_I_RB_자동 *)
    R369_2_M_I_RB_최종작업완료 : BOOL; (* AT %MW20091.0 *) (* R369_2_M_I_RB_최종작업완료 *)
    R369_2_M_I_RB_프로그램_이상 : BOOL; (* AT %MW20090.6 *) (* R369_2_M_I_RB_프로그램_이상 *)
    R369_2_M_O_RB_1_CYCLE_SET : BOOL; (* AT %MW21090.3 *) (* R369_2_M_O_RB_1_CYCLE_SET *)
    R369_2_M_O_RB_1차_작업완료_리셋 : BOOL; (* AT %MW21092.0 *) (* R369_2_M_O_RB_1차_작업완료_리셋 *)
    R369_2_M_O_RB_2차_작업완료_리셋 : BOOL; (* AT %MW21092.1 *) (* R369_2_M_O_RB_2차_작업완료_리셋 *)
    R369_2_M_O_RB_2차_진입OK : BOOL; (* AT %MW21091.8 *) (* R369_2_M_O_RB_2차_진입OK *)
    R369_2_M_O_RB_3차_작업완료_리셋 : BOOL; (* AT %MW21092.2 *) (* R369_2_M_O_RB_3차_작업완료_리셋 *)
    R369_2_M_O_RB_3차_진입OK : BOOL; (* AT %MW21091.9 *) (* R369_2_M_O_RB_3차_진입OK *)
    R369_2_M_O_RB_4차_작업완료_리셋 : BOOL; (* AT %MW21092.3 *) (* R369_2_M_O_RB_4차_작업완료_리셋 *)
    R369_2_M_O_RB_4차_진입OK : BOOL; (* AT %MW21091.10 *) (* R369_2_M_O_RB_4차_진입OK *)
    R369_2_M_O_RB_5차_작업완료_리셋 : BOOL; (* AT %MW21092.4 *) (* R369_2_M_O_RB_5차_작업완료_리셋 *)
    R369_2_M_O_RB_5차_진입OK : BOOL; (* AT %MW21091.11 *) (* R369_2_M_O_RB_5차_진입OK *)
    R369_2_M_O_RB_6차_작업완료_리셋 : BOOL; (* AT %MW21092.5 *) (* R369_2_M_O_RB_6차_작업완료_리셋 *)
    R369_2_M_O_RB_6차_진입OK : BOOL; (* AT %MW21091.12 *) (* R369_2_M_O_RB_6차_진입OK *)
    R369_2_M_O_RB_7차_작업완료_리셋 : BOOL; (* AT %MW21092.6 *) (* R369_2_M_O_RB_7차_작업완료_리셋 *)
    R369_2_M_O_RB_7차_진입OK : BOOL; (* AT %MW21091.13 *) (* R369_2_M_O_RB_7차_진입OK *)
    R369_2_M_O_RB_ATD_OK : BOOL; (* AT %MW21090.6 *) (* R369_2_M_O_RB_ATD_OK *)
    R369_2_M_O_RB_PLT_10_진입OK : BOOL; (* AT %MW21093.10 *) (* R369_2_M_O_RB_PLT_10_진입OK *)
    R369_2_M_O_RB_PLT_11_진입OK : BOOL; (* AT %MW21093.11 *) (* R369_2_M_O_RB_PLT_11_진입OK *)
    R369_2_M_O_RB_PLT_12_진입OK : BOOL; (* AT %MW21093.12 *) (* R369_2_M_O_RB_PLT_12_진입OK *)
    R369_2_M_O_RB_PLT_1_진입OK : BOOL; (* AT %MW21093.1 *) (* R369_2_M_O_RB_PLT_1_진입OK *)
    R369_2_M_O_RB_PLT_2_진입OK : BOOL; (* AT %MW21093.2 *) (* R369_2_M_O_RB_PLT_2_진입OK *)
    R369_2_M_O_RB_PLT_3_진입OK : BOOL; (* AT %MW21093.3 *) (* R369_2_M_O_RB_PLT_3_진입OK *)
    R369_2_M_O_RB_PLT_4_진입OK : BOOL; (* AT %MW21093.4 *) (* R369_2_M_O_RB_PLT_4_진입OK *)
    R369_2_M_O_RB_PLT_5_진입OK : BOOL; (* AT %MW21093.5 *) (* R369_2_M_O_RB_PLT_5_진입OK *)
    R369_2_M_O_RB_PLT_6_진입OK : BOOL; (* AT %MW21093.6 *) (* R369_2_M_O_RB_PLT_6_진입OK *)
    R369_2_M_O_RB_PLT_7_진입OK : BOOL; (* AT %MW21093.7 *) (* R369_2_M_O_RB_PLT_7_진입OK *)
    R369_2_M_O_RB_PLT_8_진입OK : BOOL; (* AT %MW21093.8 *) (* R369_2_M_O_RB_PLT_8_진입OK *)
    R369_2_M_O_RB_PLT_9_진입OK : BOOL; (* AT %MW21093.9 *) (* R369_2_M_O_RB_PLT_9_진입OK *)
    R369_2_M_O_RB_PLT_카운터리셋_보조 : BOOL; (* AT %MW21090.10 *) (* R369_2_M_O_RB_PLT_카운터리셋_보조 *)
    R369_2_M_O_RB_PROG_NO : WORD; (* AT %MW21094 *)
    R369_2_M_O_RB_RESTART_OK : BOOL; (* AT %MW21090.2 *) (* R369_2_M_O_RB_RESTART_OK *)
    R369_2_M_O_RB_START_OK : BOOL; (* AT %MW21090.0 *) (* R369_2_M_O_RB_START_OK *)
    R369_2_M_O_RB_TEST_MODE_5000회 : BOOL; (* AT %MW21090.12 *) (* R369_2_M_O_RB_TEST_MODE_5000회 *)
    R369_2_M_O_RB_TIP_교체_시작 : BOOL; (* AT %MW21090.7 *) (* R369_2_M_O_RB_TIP_교체_시작 *)
    R369_2_M_O_RB_TIP_교체_완료 : BOOL; (* AT %MW21090.8 *) (* R369_2_M_O_RB_TIP_교체_완료 *)
    R369_2_M_O_RB_VIP_MODE : BOOL; (* AT %MW21090.11 *) (* R369_2_M_O_RB_VIP_MODE *)
    R369_2_M_O_RB_냉각수_차단_요청 : BOOL; (* AT %MW21090.9 *) (* R369_2_M_O_RB_냉각수_차단_요청 *)
    R369_2_M_O_RB_진입OK_AX차종 : BOOL; (* AT %MW21091.0 *) (* R369_2_M_O_RB_진입OK_AX차종 *)
    R369_2_M_O_RB_진입OK_B차종 : BOOL; (* AT %MW21091.1 *) (* R369_2_M_O_RB_진입OK_B차종 *)
    R369_2_M_O_RB_진입OK_C차종 : BOOL; (* AT %MW21091.2 *) (* R369_2_M_O_RB_진입OK_C차종 *)
    R369_2_M_O_RB_진입OK_D차종 : BOOL; (* AT %MW21091.3 *) (* R369_2_M_O_RB_진입OK_D차종 *)
    R369_2_M_O_RB_진입OK_E차종 : BOOL; (* AT %MW21091.4 *) (* R369_2_M_O_RB_진입OK_E차종 *)
    R369_2_M_O_RB_진입OK_F차종 : BOOL; (* AT %MW21091.5 *) (* R369_2_M_O_RB_진입OK_F차종 *)
    R369_2_M_O_RB_진입OK_G차종 : BOOL; (* AT %MW21091.6 *) (* R369_2_M_O_RB_진입OK_G차종 *)
    R369_2_M_O_RB_진입OK_H차종 : BOOL; (* AT %MW21091.7 *) (* R369_2_M_O_RB_진입OK_H차종 *)
    R369_2_M_O_RB_최종_작업완료_리셋 : BOOL; (* AT %MW21090.5 *) (* R369_2_M_O_RB_최종_작업완료_리셋 *)
    R369_2_M_O_RB_프로그램_OK : BOOL; (* AT %MW21090.1 *) (* R369_2_M_O_RB_프로그램_OK *)
    R369_2_O_RB_OUTPUT : ARRAY[0..3] OF WORD; (* AT %MW94090 *) (* R369_2_O_RB_OUTPUT *)
END_VAR
(* ladder body could not be read *)
END_PROGRAM

PROGRAM S369_1_이상 (* task: 스캔 프로그램 *)
VAR
    INST10 : TON;
    INST11 : TON;
    INST12 : TON;
    INST13 : TON;
    INST14 : TON;
    INST15 : TON;
    INST16 : TON;
    INST17 : TON;
    INST18 : TON;
    INST19 : TON;
    INST20 : TON;
    INST21 : TON;
    INST22 : TON;
    INST23 : TON;
    INST24 : TON;
    INST25 : TON;
    INST26 : TON;
    INST27 : TON;
    INST28 : TON;
    INST29 : TON;
    INST8 : TON;
    INST9 : TON;
END_VAR
VAR_EXTERNAL
    R368_1_M_I_RB_이상 : BOOL; (* AT %MW20070.2 *) (* R368_1_M_I_RB_이상 *)
    R368_1_M_I_RB_프로그램_이상 : BOOL; (* AT %MW20070.6 *) (* R368_1_M_I_RB_프로그램_이상 *)
    R369_1_M_I_RB_이상 : BOOL; (* AT %MW20080.2 *) (* R369_1_M_I_RB_이상 *)
    R369_1_M_I_RB_프로그램_이상 : BOOL; (* AT %MW20080.6 *) (* R369_1_M_I_RB_프로그램_이상 *)
    R369_2_M_I_RB_이상 : BOOL; (* AT %MW20090.2 *) (* R369_2_M_I_RB_이상 *)
    R369_2_M_I_RB_프로그램_이상 : BOOL; (* AT %MW20090.6 *) (* R369_2_M_I_RB_프로그램_이상 *)
    S369_1_6_40_PLC_BOX_CP_TRIP : BOOL; (* AT %MW86402.15 *) (* S369_1_6_40_PLC_BOX_CP_TRIP *)
    _0004_EB07_CFG_ER : BOOL; (* AT %MW184037.0 *) (* EB 구성 에러 *)
    _0004_EB07_DEER : BOOL; (* AT %MW184037.1 *) (* EB 운전 중 탈락 *)
    _0004_EB08_CFG_ER : BOOL; (* AT %MW184039.8 *) (* EB 구성 에러 *)
    _0004_EB08_DEER : BOOL; (* AT %MW184039.9 *) (* EB 운전 중 탈락 *)
    _0004_EB09_CFG_ER : BOOL; (* AT %MW184042.0 *) (* EB 구성 에러 *)
    _0004_EB09_DEER : BOOL; (* AT %MW184042.1 *) (* EB 운전 중 탈락 *)
    _0006_EB30_CFG_ER : BOOL; (* AT %MW186046.0 *) (* EB 구성 에러 *)
    _0006_EB30_DEER : BOOL; (* AT %MW186046.1 *) (* EB 운전 중 탈락 *)
    _0006_EB30_IO_DEER : BOOL; (* AT %MW186047.2 *) (* EB IO 탈락 에러 *)
    _0006_EB30_IO_TYER : BOOL; (* AT %MW186047.1 *) (* EB IO 타입 에러 *)
    _0006_EB40_CFG_ER : BOOL; (* AT %MW186058.0 *) (* EB 구성 에러 *)
    _0006_EB40_DEER : BOOL; (* AT %MW186058.1 *) (* EB 운전 중 탈락 *)
    _0006_EB40_IO_DEER : BOOL; (* AT %MW186059.2 *) (* EB IO 탈락 에러 *)
    _0006_EB40_IO_TYER : BOOL; (* AT %MW186059.1 *) (* EB IO 타입 에러 *)
END_VAR
VAR_EXTERNAL RETAIN
    R369_1_M_NODE_4_08_통신_이상 : BOOL; (* AT %MW4524.8 *)
    R369_2_M_NODE_4_09_통신_이상 : BOOL; (* AT %MW4524.9 *)
    S369_1_M_NODE_6_40_통신_이상 : BOOL; (* AT %MW4524.0 *)
    S369_1_M_R369_1_안착완료 : BOOL; (* AT %MW4501.1 *)
    S369_1_M_ROOF_제품감지_무 : BOOL; (* AT %MW4501.6 *)
    S369_1_M_ROOF_제품감지_유 : BOOL; (* AT %MW4501.5 *)
    S369_1_M_ROOF_제품감지_이상 : BOOL; (* AT %MW4514.0 *)
    S369_1_M_공정_불간섭 : BOOL; (* AT %MW4504.1 *) (* S369_1_M_공정_불간섭 *)
    S369_1_M_공정_제품감지_무 : BOOL; (* AT %MW4501.4 *) (* S369_1_M_공정_제품감지_무 *)
    S369_1_M_공정_차종_유 : BOOL; (* AT %MW4502.0 *) (* S369_1_M_공정_차종_유 *)
    S369_1_M_썬루프_제품감지_유 : BOOL; (* AT %MW4501.7 *)
    S369_1_M_썬루프_제품감지_이상 : BOOL; (* AT %MW4514.1 *)
    S369_1_M_자동_운전중 : BOOL; (* AT %MW4500.4 *) (* S369-1 자동운전중 *)
    S369_1_M_차종6_썬루프 : BOOL; (* AT %MW10223.4 *) (* S369 1 M 차종6 썬루프 *)
    S369_1_M_차종6_일반루프 : BOOL; (* AT %MW10223.3 *) (* S369 1 M 차종6 일반루프 *)
    S369_1_M_총괄_CP_이상 : BOOL; (* AT %MW4509.7 *) (* S369-1 CP OFF 이상 *)
    S369_1_M_총괄_CT_이상 : BOOL; (* AT %MW4510.4 *) (* S369-1 TACK TIME 이상 *)
    S369_1_M_총괄_EOCR_이상 : BOOL; (* AT %MW4509.8 *) (* S369_1_M_총괄_EOCR_이상 *)
    S369_1_M_총괄_INV_이상 : BOOL; (* AT %MW4509.9 *) (* S369_1_M_총괄_INV_이상 *)
    S369_1_M_총괄_LS_이상 : BOOL; (* AT %MW4509.15 *) (* S369-1 LS 이상 *)
    S369_1_M_총괄_MATCH_이상 : BOOL; (* AT %MW4510.0 *) (* S369-1 매트SW 이상 *)
    S369_1_M_총괄_MC_이상 : BOOL; (* AT %MW4509.13 *) (* S369_1_M_총괄_MC_이상 *)
    S369_1_M_총괄_NFB_이상 : BOOL; (* AT %MW4509.11 *) (* S369_1_M_총괄_NFB_이상 *)
    S369_1_M_총괄_ROBOT_이상 : BOOL; (* AT %MW4510.1 *) (* S369-1 ROBOT 이상 *)
    S369_1_M_총괄_SAFETY_이상 : BOOL; (* AT %MW4509.2 *) (* S369_1_M_총괄_SAFETY_이상 *)
    S369_1_M_총괄_공기압_이상 : BOOL; (* AT %MW4509.3 *) (* S36-1 공기압 이상 *)
    S369_1_M_총괄_사양_이상 : BOOL; (* AT %MW4509.6 *) (* S369-1 사양 이상 *)
    S369_1_M_총괄_오버런_이상 : BOOL; (* AT %MW4509.12 *) (* S369_1_M_총괄_오버런_이상 *)
    S369_1_M_총괄_용접타점수_이상 : BOOL; (* AT %MW4510.2 *) (* S369-1 용접타점수 이상 *)
    S369_1_M_총괄_이상 : BOOL; (* AT %MW4509.0 *) (* S369_1_M_총괄_이상 *)
    S369_1_M_총괄_제품감지_이상 : BOOL; (* AT %MW4509.4 *) (* S369-1 제품감지 이상 *)
    S369_1_M_총괄_차종_이상 : BOOL; (* AT %MW4509.5 *) (* S369-1 차종 이상 *)
    S369_1_M_총괄_통신_이상 : BOOL; (* AT %MW4509.14 *) (* S369-1 통신이상 *)
    전체_M_이상_리셋 : BOOL; (* AT %MW308.2 *) (* ALL공정 PB 이상리셋 *)
END_VAR

